// TIA Portal V18 program export: 2 tag tables, 0 data types, 2 data blocks, 5 code blocks (in call order from the OBs), 1 instance data blocks

VAR_GLOBAL   // PLC tag table "Default tag table"
   System_Byte AT %MB101 : Byte;
   FirstScan AT %M101.0 : Bool;
   DiagStatusUpdate AT %M101.1 : Bool;
   AlwaysTRUE AT %M101.2 : Bool;
   AlwaysFALSE AT %M101.3 : Bool;
   Clock_Byte AT %MB100 : Byte;
   Clock_10Hz AT %M100.0 : Bool;
   Clock_5Hz AT %M100.1 : Bool;
   "Clock_2.5Hz" AT %M100.2 : Bool;
   Clock_2Hz AT %M100.3 : Bool;
   "Clock_1.25Hz" AT %M100.4 : Bool;
   Clock_1Hz AT %M100.5 : Bool;
   "Clock_0.625Hz" AT %M100.6 : Bool;
   "Clock_0.5Hz" AT %M100.7 : Bool;
END_VAR

VAR_GLOBAL   // PLC tag table "PLC_Tags"
   FT3210_Bon3 AT %ID132 : Real;   // Cảm biến lưu lượng nước dosing vào Bồn 3
   FT3210_Bon3_HMI AT %MD764 : Real;   // Giá trị mô phỏng/HMI song song cho Cảm biến lưu lượng nước dosing vào Bồn 3
   FT3210_Bon3_Use_HMI AT %M421.0 : Bool;   // Chọn chế độ mô phỏng HMI cho Cảm biến lưu lượng nước dosing vào Bồn 3
   FT3210_Bon3_Sim_Req AT %M323.2 : Bool;   // Yêu cầu mô phỏng cảm biến cho Cảm biến lưu lượng nước dosing vào Bồn 3
   FT3210_Bon3_Sim_Active AT %M323.3 : Bool;   // Mô phỏng cảm biến đang hoạt động cho Cảm biến lưu lượng nước dosing vào Bồn 3
   FT3210_Bon3_Eff AT %MD768 : Real;   // Giá trị thực tế/mô phỏng hiệu dụng cho Cảm biến lưu lượng nước dosing vào Bồn 3
   FQ3210_Bon3 AT %ID136 : Real;   // Bộ đếm lưu lượng tích lũy Bồn 3
   FQ3210_Bon3_HMI AT %MD772 : Real;   // Giá trị mô phỏng/HMI song song cho Bộ đếm lưu lượng tích lũy Bồn 3
   FQ3210_Bon3_Use_HMI AT %M421.1 : Bool;   // Chọn chế độ mô phỏng HMI cho Bộ đếm lưu lượng tích lũy Bồn 3
   FQ3210_Bon3_Sim_Req AT %M323.4 : Bool;   // Yêu cầu mô phỏng cảm biến cho Bộ đếm lưu lượng tích lũy Bồn 3
   FQ3210_Bon3_Sim_Active AT %M323.5 : Bool;   // Mô phỏng cảm biến đang hoạt động cho Bộ đếm lưu lượng tích lũy Bồn 3
   FQ3210_Bon3_Eff AT %MD776 : Real;   // Giá trị thực tế/mô phỏng hiệu dụng cho Bộ đếm lưu lượng tích lũy Bồn 3
   LT3213_Bon3 AT %ID140 : Real;   // Cảm biến mức liên tục Bồn 3
   LT3213_Bon3_HMI AT %MD780 : Real;   // Giá trị mô phỏng/HMI song song cho Cảm biến mức liên tục Bồn 3
   LT3213_Bon3_Use_HMI AT %M421.2 : Bool;   // Chọn chế độ mô phỏng HMI cho Cảm biến mức liên tục Bồn 3
   LT3213_Bon3_Sim_Req AT %M323.6 : Bool;   // Yêu cầu mô phỏng cảm biến cho Cảm biến mức liên tục Bồn 3
   LT3213_Bon3_Sim_Active AT %M323.7 : Bool;   // Mô phỏng cảm biến đang hoạt động cho Cảm biến mức liên tục Bồn 3
   LT3213_Bon3_Eff AT %MD784 : Real;   // Giá trị thực tế/mô phỏng hiệu dụng cho Cảm biến mức liên tục Bồn 3
   TT3214_Bon3 AT %ID144 : Real;   // Cảm biến nhiệt độ Bồn 3
   TT3214_Bon3_HMI AT %MD788 : Real;   // Giá trị mô phỏng/HMI song song cho Cảm biến nhiệt độ Bồn 3
   TT3214_Bon3_Use_HMI AT %M421.3 : Bool;   // Chọn chế độ mô phỏng HMI cho Cảm biến nhiệt độ Bồn 3
   TT3214_Bon3_Sim_Req AT %M324.0 : Bool;   // Yêu cầu mô phỏng cảm biến cho Cảm biến nhiệt độ Bồn 3
   TT3214_Bon3_Sim_Active AT %M324.1 : Bool;   // Mô phỏng cảm biến đang hoạt động cho Cảm biến nhiệt độ Bồn 3
   TT3214_Bon3_Eff AT %MD792 : Real;   // Giá trị thực tế/mô phỏng hiệu dụng cho Cảm biến nhiệt độ Bồn 3
   FT3215_Bon4 AT %ID148 : Real;   // Cảm biến lưu lượng nước dosing vào Bồn 4
   FT3215_Bon4_HMI AT %MD796 : Real;   // Giá trị mô phỏng/HMI song song cho Cảm biến lưu lượng nước dosing vào Bồn 4
   FT3215_Bon4_Use_HMI AT %M421.4 : Bool;   // Chọn chế độ mô phỏng HMI cho Cảm biến lưu lượng nước dosing vào Bồn 4
   FT3215_Bon4_Sim_Req AT %M324.2 : Bool;   // Yêu cầu mô phỏng cảm biến cho Cảm biến lưu lượng nước dosing vào Bồn 4
   FT3215_Bon4_Sim_Active AT %M324.3 : Bool;   // Mô phỏng cảm biến đang hoạt động cho Cảm biến lưu lượng nước dosing vào Bồn 4
   FT3215_Bon4_Eff AT %MD800 : Real;   // Giá trị thực tế/mô phỏng hiệu dụng cho Cảm biến lưu lượng nước dosing vào Bồn 4
   FQ3215_Bon4 AT %ID152 : Real;   // Bộ đếm lưu lượng tích lũy Bồn 4
   FQ3215_Bon4_HMI AT %MD804 : Real;   // Giá trị mô phỏng/HMI song song cho Bộ đếm lưu lượng tích lũy Bồn 4
   FQ3215_Bon4_Use_HMI AT %M421.5 : Bool;   // Chọn chế độ mô phỏng HMI cho Bộ đếm lưu lượng tích lũy Bồn 4
   FQ3215_Bon4_Sim_Req AT %M324.4 : Bool;   // Yêu cầu mô phỏng cảm biến cho Bộ đếm lưu lượng tích lũy Bồn 4
   FQ3215_Bon4_Sim_Active AT %M324.5 : Bool;   // Mô phỏng cảm biến đang hoạt động cho Bộ đếm lưu lượng tích lũy Bồn 4
   FQ3215_Bon4_Eff AT %MD808 : Real;   // Giá trị thực tế/mô phỏng hiệu dụng cho Bộ đếm lưu lượng tích lũy Bồn 4
   LS3217_Bon4_Cao AT %I0.5 : Bool;   // Cảm biến mức cao Bồn 4
   LS3217_Bon4_Cao_HMI AT %M110.5 : Bool;   // Tín hiệu mô phỏng/HMI song song cho Cảm biến mức cao Bồn 4
   LS3217_Bon4_Cao_HMI_Gated AT %M324.6 : Bool;   // Tín hiệu HMI đã qua xử lý chế độ cho Cảm biến mức cao Bồn 4
   LS3217_Bon4_Cao_Eff AT %M324.7 : Bool;   // Tín hiệu thực tế/mô phỏng hiệu dụng cho Cảm biến mức cao Bồn 4
   LT3218_Bon4 AT %ID156 : Real;   // Cảm biến mức liên tục Bồn 4
   LT3218_Bon4_HMI AT %MD812 : Real;   // Giá trị mô phỏng/HMI song song cho Cảm biến mức liên tục Bồn 4
   LT3218_Bon4_Use_HMI AT %M421.6 : Bool;   // Chọn chế độ mô phỏng HMI cho Cảm biến mức liên tục Bồn 4
   LT3218_Bon4_Sim_Req AT %M325.0 : Bool;   // Yêu cầu mô phỏng cảm biến cho Cảm biến mức liên tục Bồn 4
   LT3218_Bon4_Sim_Active AT %M325.1 : Bool;   // Mô phỏng cảm biến đang hoạt động cho Cảm biến mức liên tục Bồn 4
   LT3218_Bon4_Eff AT %MD816 : Real;   // Giá trị thực tế/mô phỏng hiệu dụng cho Cảm biến mức liên tục Bồn 4
   TT3219_Bon4 AT %ID160 : Real;   // Cảm biến nhiệt độ Bồn 4
   TT3219_Bon4_HMI AT %MD820 : Real;   // Giá trị mô phỏng/HMI song song cho Cảm biến nhiệt độ Bồn 4
   TT3219_Bon4_Use_HMI AT %M421.7 : Bool;   // Chọn chế độ mô phỏng HMI cho Cảm biến nhiệt độ Bồn 4
   TT3219_Bon4_Sim_Req AT %M325.2 : Bool;   // Yêu cầu mô phỏng cảm biến cho Cảm biến nhiệt độ Bồn 4
   TT3219_Bon4_Sim_Active AT %M325.3 : Bool;   // Mô phỏng cảm biến đang hoạt động cho Cảm biến nhiệt độ Bồn 4
   TT3219_Bon4_Eff AT %MD824 : Real;   // Giá trị thực tế/mô phỏng hiệu dụng cho Cảm biến nhiệt độ Bồn 4
   V3240_Nuoc_Bon3 AT %Q1.4 : Bool;   // Van on/off cấp nước Bồn 3
   V3240_Nuoc_Bon3_M AT %M221.4 : Bool;   // Tag gương phản hồi HMI cho Van on/off cấp nước Bồn 3
   CV3211_Nuoc_Bon3 AT %QD116 : Real;   // Van tuyến tính cấp nước Bồn 3
   CV3211_Nuoc_Bon3_M AT %MD1216 : Real;   // Tag gương phản hồi HMI cho Van tuyến tính cấp nước Bồn 3
   AGTR3262_Khuay_Bon3 AT %Q1.5 : Bool;   // Động cơ khuấy Bồn 3
   AGTR3262_Khuay_Bon3_M AT %M221.5 : Bool;   // Tag gương phản hồi HMI cho Động cơ khuấy Bồn 3
   AGTR3262_Toc_Do_AO AT %QD120 : Real;   // Tín hiệu tốc độ khuấy Bồn 3
   AGTR3262_Toc_Do_AO_M AT %MD1220 : Real;   // Tag gương phản hồi HMI cho Tín hiệu tốc độ khuấy Bồn 3
   V3242_Xa_Bon3 AT %Q1.6 : Bool;   // Van xả đáy Bồn 3 số 1
   V3242_Xa_Bon3_M AT %M221.6 : Bool;   // Tag gương phản hồi HMI cho Van xả đáy Bồn 3 số 1
   V3243_Xa_Bon3 AT %Q1.7 : Bool;   // Van xả đáy Bồn 3 số 2
   V3243_Xa_Bon3_M AT %M221.7 : Bool;   // Tag gương phản hồi HMI cho Van xả đáy Bồn 3 số 2
   V3244_Xa_Bon3 AT %Q2.0 : Bool;   // Van xả đáy Bồn 3 số 3
   V3244_Xa_Bon3_M AT %M222.0 : Bool;   // Tag gương phản hồi HMI cho Van xả đáy Bồn 3 số 3
   V3245_Nuoc_Bon4 AT %Q2.1 : Bool;   // Van on/off cấp nước Bồn 4
   V3245_Nuoc_Bon4_M AT %M222.1 : Bool;   // Tag gương phản hồi HMI cho Van on/off cấp nước Bồn 4
   CV3216_Hoi_Bon4 AT %QD124 : Real;   // Van tuyến tính gia nhiệt mô phỏng Bồn 4
   CV3216_Hoi_Bon4_M AT %MD1224 : Real;   // Tag gương phản hồi HMI cho Van tuyến tính gia nhiệt mô phỏng Bồn 4
   AGTR3263_Khuay_Bon4 AT %Q2.2 : Bool;   // Động cơ khuấy Bồn 4
   AGTR3263_Khuay_Bon4_M AT %M222.2 : Bool;   // Tag gương phản hồi HMI cho Động cơ khuấy Bồn 4
   AGTR3263_Dao_Chieu AT %Q2.3 : Bool;   // Lệnh đảo chiều động cơ khuấy Bồn 4
   AGTR3263_Dao_Chieu_M AT %M222.3 : Bool;   // Tag gương phản hồi HMI cho Lệnh đảo chiều động cơ khuấy Bồn 4
   AGTR3263_Toc_Do_AO AT %QD128 : Real;   // Tốc độ đặt động cơ khuấy Bồn 4
   AGTR3263_Toc_Do_AO_M AT %MD1228 : Real;   // Tag gương phản hồi HMI cho Tốc độ đặt động cơ khuấy Bồn 4
   V3247_Xa_Bon4 AT %Q2.4 : Bool;   // Van xả đáy Bồn 4 số 1
   V3247_Xa_Bon4_M AT %M222.4 : Bool;   // Tag gương phản hồi HMI cho Van xả đáy Bồn 4 số 1
   V3248_Xa_Bon4 AT %Q2.5 : Bool;   // Van xả đáy Bồn 4 số 2
   V3248_Xa_Bon4_M AT %M222.5 : Bool;   // Tag gương phản hồi HMI cho Van xả đáy Bồn 4 số 2
   V3249_Xa_Bon4 AT %Q2.6 : Bool;   // Van xả đáy Bồn 4 số 3
   V3249_Xa_Bon4_M AT %M222.6 : Bool;   // Tag gương phản hồi HMI cho Van xả đáy Bồn 4 số 3
   Pump3265_Chuyen_Nhanh2 AT %Q2.7 : Bool;   // Bơm chuyển dung dịch Nhánh 2 xuống bồn chứa
   Pump3265_Chuyen_Nhanh2_M AT %M222.7 : Bool;   // Tag gương phản hồi HMI cho Bơm chuyển dung dịch Nhánh 2 xuống bồn chứa
   HMI_Operator_Login AT %M422.7 : Bool;   // Đăng nhập quyền Operator
   HMI_Engineer_Login AT %M423.0 : Bool;   // Đăng nhập quyền Engineer
   HMI_Admin_Login AT %M423.1 : Bool;   // Đăng nhập quyền Admin
   HMI_Che_Do_Manual AT %M423.2 : Bool;   // Cho phép điều khiển tay từng thiết bị
   HMI_Ack_Alarm AT %M423.3 : Bool;   // Xác nhận cảnh báo
   HMI_Reset_Alarm AT %M423.4 : Bool;   // Reset alarm bằng HMI
   Gia_Lap_Mat_Ket_Noi_HMI AT %M423.5 : Bool;   // Nút giả lập mất kết nối PLC
   HMI_User_Level AT %MW520 : Int;   // Mức quyền hiện tại: 1 Operator, 2 Engineer, 3 Admin
   HMI_Cho_Phep_Sua_Thong_So AT %M327.6 : Bool;   // Cờ cho phép sửa công thức và PID
   HMI_Alarm_Status AT %MW522 : Int;   // Mã cảnh báo tổng hợp cho WinCC TextList
   HMI_AnToan_Status AT %MW524 : Int;   // Mã chẩn đoán an toàn ưu tiên
   PLC2_Auto_Enable AT %M328.5 : Bool;   // Cho phép chạy Auto Nhánh 2 Bồn 3-4
   PLC2_EStop_Latch AT %M328.6 : Bool;   // Chốt dừng khẩn HMI/SCADA Nhánh 2 Bồn 3-4
   PLC2_Loi_Tong AT %M328.7 : Bool;   // Lỗi tổng khóa Auto Nhánh 2 Bồn 3-4
   PLC2_Loi_Dry_Run AT %M329.0 : Bool;   // Lỗi chạy khô bơm Nhánh 2 Bồn 3-4
   PLC2_Loi_Dosing AT %M329.1 : Bool;   // Lỗi quá thời gian dosing Nhánh 2 Bồn 3-4
   PLC2_Loi_Truyen_Thong AT %M329.2 : Bool;   // Lỗi truyền thông mô phỏng Nhánh 2 Bồn 3-4
   PLC2_State AT %MW528 : Int;   // Mã bước chu trình Nhánh 2 Bồn 3-4
   PLC2_Step_Bon3_Dosing AT %M331.0 : Bool;   // Bồn 3 đang dosing nước
   PLC2_Step_Bon3_Tip AT %M331.1 : Bool;   // Bồn 3 đang mô phỏng tip cốt tương đậu đậm đặc
   PLC2_Step_Bon3_Khuay AT %M331.2 : Bool;   // Bồn 3 đang khuấy ban đầu
   PLC2_Step_Bon3_Xa AT %M331.3 : Bool;   // Bồn 3 đang xả sang Bồn 4
   PLC2_Step_Bon4_Dosing AT %M331.4 : Bool;   // Bồn 4 đang dosing bổ sung
   PLC2_Step_Bon4_Tip AT %M331.5 : Bool;   // Bồn 4 đang tip phụ gia
   PLC2_Step_Bon4_Khuay_Thuan AT %M331.6 : Bool;   // Bồn 4 khuấy chiều thuận
   PLC2_Step_Bon4_Khuay_Nghich AT %M331.7 : Bool;   // Bồn 4 khuấy chiều ngược
   PLC2_Step_Bon4_PID_Mo_Phong AT %M332.0 : Bool;   // Bồn 4 chạy PID mô phỏng
   PLC2_Step_Bon4_Thanh_Trung AT %M332.1 : Bool;   // Bồn 4 giữ thời gian thanh trùng
   PLC2_Xa_Bon3_Xong AT %M332.2 : Bool;   // Bồn 3 đã xả hết
   PLC2_Xa_Bon4_Xong AT %M332.3 : Bool;   // Bồn 4 đã xả hết
   PLC2_Me_Nhanh2_Hoan_Thanh AT %M333.3 : Bool;   // Cờ hoàn thành Nhánh 2 gửi sang PLC1
   PLC2_Me_Nhanh2_Hoan_Thanh_M AT %M224.6 : Bool;   // Tag gương phản hồi HMI cho cờ hoàn thành Nhánh 2 gửi sang PLC1
   Pump3265_Chuyen_Nhanh2_Cmd_Nhan AT %M333.7 : Bool;   // Nhận lệnh chạy bơm chuyển Nhánh 2 từ PLC1
   Pump3265_Chuyen_Nhanh2_Cmd_Nhan_HMI AT %M111.1 : Bool;   // Tín hiệu mô phỏng/HMI song song cho lệnh chạy bơm chuyển Nhánh 2 từ PLC1
   Nut_Khoi_Dong_Nhan AT %M334.1 : Bool;   // nút khởi động nhận từ PLC1
   Nut_Khoi_Dong_Nhan_HMI AT %M111.2 : Bool;   // Tín hiệu mô phỏng/HMI song song cho nút khởi động nhận từ PLC1
   Nut_Khoi_Dong_Nhan_HMI_Gated AT %M334.2 : Bool;   // Tín hiệu HMI đã qua xử lý chế độ cho nút khởi động nhận từ PLC1
   Nut_Khoi_Dong_Nhan_Eff AT %M334.3 : Bool;   // Tín hiệu thực tế/mô phỏng hiệu dụng cho nút khởi động nhận từ PLC1
   Nut_Dung_Nhan AT %M334.4 : Bool;   // nút dừng nhận từ PLC1
   Nut_Dung_Nhan_HMI AT %M111.3 : Bool;   // Tín hiệu mô phỏng/HMI song song cho nút dừng nhận từ PLC1
   Nut_Dung_Nhan_HMI_Gated AT %M334.5 : Bool;   // Tín hiệu HMI đã qua xử lý chế độ cho nút dừng nhận từ PLC1
   Nut_Dung_Nhan_Eff AT %M334.6 : Bool;   // Tín hiệu thực tế/mô phỏng hiệu dụng cho nút dừng nhận từ PLC1
   Nut_Reset_Nhan AT %M334.7 : Bool;   // nút reset nhận từ PLC1
   Nut_Reset_Nhan_HMI AT %M111.4 : Bool;   // Tín hiệu mô phỏng/HMI song song cho nút reset nhận từ PLC1
   Nut_Reset_Nhan_HMI_Gated AT %M335.0 : Bool;   // Tín hiệu HMI đã qua xử lý chế độ cho nút reset nhận từ PLC1
   Nut_Reset_Nhan_Eff AT %M335.1 : Bool;   // Tín hiệu thực tế/mô phỏng hiệu dụng cho nút reset nhận từ PLC1
   Nut_EStop_Nhan AT %M335.2 : Bool;   // nút dừng khẩn nhận từ PLC1
   Nut_EStop_Nhan_HMI AT %M111.5 : Bool;   // Tín hiệu mô phỏng/HMI song song cho nút dừng khẩn nhận từ PLC1
   Nut_EStop_Nhan_HMI_Gated AT %M335.3 : Bool;   // Tín hiệu HMI đã qua xử lý chế độ cho nút dừng khẩn nhận từ PLC1
   Nut_EStop_Nhan_Eff AT %M335.4 : Bool;   // Tín hiệu thực tế/mô phỏng hiệu dụng cho nút dừng khẩn nhận từ PLC1
   Clock_1Hz AT %M100.5 : Bool;   // Clock 1Hz system memory bit
   FirstScan AT %M101.0 : Bool;   // First Scan system memory bit
   PLC2_Last_CmdSeq AT %MW80 : Int;   // Last processed command sequence
   PLC2_CmdSeq_New AT %M82.0 : Bool;   // New command sequence received
   MB_TCP_Server_Error AT %M82.1 : Bool;   // Modbus TCP Server Error
   MB_TCP_Server_Status AT %MW84 : Word;   // Modbus TCP Server Status
   MB_TCP_Server_NDR AT %M82.2 : Bool;   // Modbus TCP Server New Data Received
   MB_TCP_Server_DR AT %M82.3 : Bool;   // Modbus TCP Server Data Read
   PLC1_Tip_Bon1_Xong_HMI AT %M423.6 : Bool;   // Nút mô phỏng tip Bồn 1 đã hoàn tất
   PLC1_Khuay_Bon1_Xong_HMI AT %M423.7 : Bool;   // Nút mô phỏng hết thời gian khuấy Bồn 1
   PLC1_Tip_Bon2_Xong_HMI AT %M424.0 : Bool;   // Nút mô phỏng tip Bồn 2 đã hoàn tất
   PLC1_Khuay_Thuan_Bon2_Xong_HMI AT %M424.1 : Bool;   // Nút mô phỏng hết thời gian khuấy thuận Bồn 2
   PLC1_Khuay_Nghich_Bon2_Xong_HMI AT %M424.2 : Bool;   // Nút mô phỏng hết thời gian khuấy ngược Bồn 2
   PLC1_Thanh_Trung_Bon2_Xong_HMI AT %M424.3 : Bool;   // Nút mô phỏng hết thời gian thanh trùng Bồn 2
   PLC2_Tip_Bon3_Xong_HMI AT %M424.4 : Bool;   // Nút mô phỏng tip Bồn 3 đã hoàn tất
   PLC2_Khuay_Bon3_Xong_HMI AT %M424.5 : Bool;   // Nút mô phỏng hết thời gian khuấy Bồn 3
   PLC2_Tip_Bon4_Xong_HMI AT %M424.6 : Bool;   // Nút mô phỏng tip Bồn 4 đã hoàn tất
   PLC2_Khuay_Thuan_Bon4_Xong_HMI AT %M424.7 : Bool;   // Nút mô phỏng hết thời gian khuấy thuận Bồn 4
   PLC2_Khuay_Nghich_Bon4_Xong_HMI AT %M425.0 : Bool;   // Nút mô phỏng hết thời gian khuấy ngược Bồn 4
   PLC2_Thanh_Trung_Bon4_Xong_HMI AT %M425.1 : Bool;   // Nút mô phỏng hết thời gian thanh trùng Bồn 4
   BonChua_Nhan_Dich_Xong_HMI AT %M425.2 : Bool;   // Nút mô phỏng nhận dịch vào Bồn chứa 01 xong
   BonChua_Chuyen_Bon2_Xong_HMI AT %M425.3 : Bool;   // Nút mô phỏng chuyển sang Bồn chứa 02 xong
   HMI_SP_PLC1_Nuoc_Bon1 AT %MD896 : Real;   // Lượng nước dosing Bồn 1
   HMI_SP_PLC1_Nuoc_Bon2 AT %MD900 : Real;   // Lượng nước dosing bổ sung Bồn 2
   HMI_SP_PLC1_Toc_Do_Bon1 AT %MD904 : Real;   // Tốc độ khuấy Bồn 1
   HMI_SP_PLC1_Toc_Do_Bon2_Main AT %MD908 : Real;   // Tốc độ khuấy chính Bồn 2
   HMI_SP_PLC1_Nhiet_Do_Bon2 AT %MD912 : Real;   // Setpoint nhiệt/PID Bồn 2
   HMI_SP_PLC2_Nuoc_Bon3 AT %MD916 : Real;   // Lượng nước dosing Bồn 3
   HMI_SP_PLC2_Nuoc_Bon4 AT %MD920 : Real;   // Lượng nước dosing bổ sung Bồn 4
   HMI_SP_PLC2_Toc_Do_Bon3 AT %MD924 : Real;   // Tốc độ khuấy Bồn 3
   HMI_SP_PLC2_Toc_Do_Bon4_Main AT %MD928 : Real;   // Tốc độ khuấy chính Bồn 4
   HMI_SP_PLC2_Nhiet_Do_Bon4 AT %MD932 : Real;   // Setpoint nhiệt/PID mô phỏng Bồn 4
   HMI_SP_BonChua1_Nhiet_Giai_Nhiet AT %MD936 : Real;   // Nhiệt độ giải nhiệt đích Bồn chứa 01
   HMI_SP_Loc_Ap_Suat_Max AT %MD940 : Real;   // Ngưỡng áp suất cao trước màng lọc
   HMI_SP_Time_Khuay_Bon1 AT %MD944 : Time;   // Thời gian khuấy Bồn 1
   HMI_SP_Time_Khuay_Bon3 AT %MD948 : Time;   // Thời gian khuấy Bồn 3
   HMI_SP_Time_Fwd AT %MD952 : Time;   // Thời gian khuấy chiều thuận
   HMI_SP_Time_Rev AT %MD956 : Time;   // Thời gian khuấy chiều ngược
   HMI_SP_Time_Sterilize AT %MD960 : Time;   // Thời gian giữ nhiệt thanh trùng
   PLC1_Khuay_Bon1_Xong AT %M336.2 : Bool;   // Trạng thái tự động xong khuấy Bồn 1
   PLC1_Khuay_Thuan_Bon2_Xong AT %M336.3 : Bool;   // Trạng thái tự động xong khuấy thuận Bồn 2
   PLC1_Khuay_Nghich_Bon2_Xong AT %M336.4 : Bool;   // Trạng thái tự động xong khuấy ngược Bồn 2
   PLC1_Thanh_Trung_Bon2_Xong AT %M336.5 : Bool;   // Trạng thái tự động xong thanh trùng Bồn 2
   PLC2_Khuay_Bon3_Xong AT %M336.6 : Bool;   // Trạng thái tự động xong khuấy Bồn 3
   PLC2_Khuay_Thuan_Bon4_Xong AT %M336.7 : Bool;   // Trạng thái tự động xong khuấy thuận Bồn 4
   PLC2_Khuay_Nghich_Bon4_Xong AT %M337.0 : Bool;   // Trạng thái tự động xong khuấy ngược Bồn 4
   PLC2_Thanh_Trung_Bon4_Xong AT %M337.1 : Bool;   // Trạng thái tự động xong thanh trùng Bồn 4
   PLC1_Tip_Bon1_Auto_Done AT %M337.2 : Bool;   // Trạng thái tự động xong tip Bồn 1
   PLC1_Tip_Bon2_Auto_Done AT %M337.3 : Bool;   // Trạng thái tự động xong tip Bồn 2
   PLC2_Tip_Bon3_Auto_Done AT %M337.4 : Bool;   // Trạng thái tự động xong tip Bồn 3
   PLC2_Tip_Bon4_Auto_Done AT %M337.5 : Bool;   // Trạng thái tự động xong tip Bồn 4
   PLC1_Start_Edge_Old AT %M337.6 : Bool;   // Cờ nhớ cạnh lên nút Start PLC1
   PLC1_Start_Edge_Edge AT %M337.7 : Bool;   // Xung cạnh lên nút Start PLC1
   PLC2_Start_Edge_Old AT %M338.0 : Bool;   // Cờ nhớ cạnh lên nút Start PLC2
   PLC2_Start_Edge_Edge AT %M338.1 : Bool;   // Xung cạnh lên nút Start PLC2
   PID_Bon2_Enable AT %M338.2 : Bool;   // Cho phép PID Bồn 2
   PID_Bon2_ManualEnable AT %M338.3 : Bool;   // Chế độ manual PID Bồn 2
   PID_Bon2_Error AT %M338.4 : Bool;   // Lỗi khối PID Bồn 2
   PID_Bon4_Enable AT %M338.5 : Bool;   // Cho phép PID mô phỏng Bồn 4
   PID_Bon4_ManualEnable AT %M338.6 : Bool;   // Chế độ manual PID Bồn 4
   PID_Bon4_Error AT %M338.7 : Bool;   // Lỗi khối PID Bồn 4
   PID_Bon2_ErrorBits AT %MD964 : DWord;   // Mã lỗi DWORD PID Bồn 2
   PID_Bon4_ErrorBits AT %MD968 : DWord;   // Mã lỗi DWORD PID Bồn 4
   PID_Bon2_SP AT %MD972 : Real;   // Setpoint đưa vào PID Bồn 2
   PID_Bon2_Err AT %MD976 : Real;   // Sai lệch PID Bồn 2 = SP - PV
   PID_Bon2_CV AT %MD980 : Real;   // Giá trị điều khiển PID Bồn 2
   PID_Bon2_ManualValue AT %MD984 : Real;   // Giá trị manual PID Bồn 2
   PID_Bon4_SP AT %MD988 : Real;   // Setpoint đưa vào PID mô phỏng Bồn 4
   PID_Bon4_Err AT %MD992 : Real;   // Sai lệch PID mô phỏng Bồn 4 = SP - PV
   PID_Bon4_CV AT %MD996 : Real;   // Giá trị điều khiển PID mô phỏng Bồn 4
   PID_Bon4_ManualValue AT %MD1000 : Real;   // Giá trị manual PID Bồn 4
   TT3219_Bon4_Sim AT %MD1004 : Real;   // Nhiệt độ mô phỏng nội bộ cho PID Bồn 4
   PID_Bon2_Temp_Inc AT %MD1008 : Real;   // Mức tăng nhiệt mô phỏng Bồn 2
   PID_Bon4_Tang_Nhiet_Buoc AT %MD1012 : Real;   // Mức tăng nhiệt mô phỏng mỗi chu kỳ OB31
   TT3219_Bon4_Target AT %MD1016 : Real;   // Nhiệt độ đích mô phỏng bồn 4
   TT3219_Bon4_Sim_Pure AT %MD1020 : Real;   // Nhiệt độ mô phỏng chưa có nhiễu bồn 4
   PID_Bon4_Temp_Val_1 AT %MD1024 : Real;   // Biến tạm mô phỏng nhiệt độ 1
   PID_Bon4_Temp_Val_2 AT %MD1028 : Real;   // Biến tạm mô phỏng nhiệt độ 2
   PID_Bon4_Sim_Counter AT %MD1032 : Real;   // Đồng hồ chu kỳ mô phỏng
   PID_Bon4_Sim_Angle AT %MD1036 : Real;   // Góc lượng giác nhiễu
   PID_Bon4_Sim_Sin AT %MD1040 : Real;   // Giá trị hình sin nhiễu
   PID_Bon4_Sim_Noise AT %MD1044 : Real;   // Giá trị nhiễu nhiệt độ
   PLC1_Tip_Bon1_Timer AT %MD1048 : Real;   // Bộ đếm thời gian mô phỏng tip bồn 1
   PLC1_Tip_Bon2_Timer AT %MD1052 : Real;   // Bộ đếm thời gian mô phỏng tip bồn 2
   PLC2_Tip_Bon3_Timer AT %MD1056 : Real;   // Bộ đếm thời gian mô phỏng tip bồn 3
   PLC2_Tip_Bon4_Timer AT %MD1060 : Real;   // Bộ đếm thời gian mô phỏng tip bồn 4
   PID_Bon4_State AT %MW536 : Int;   // Trạng thái khối PID Bồn 4
   PLC2_Stop_Active AT %M339.1 : Bool;   // Tín hiệu dừng active PLC2
   AGTR3263_Khuay_Active AT %M339.4 : Bool;   // Trạng thái khuấy Bồn 4 active
   AGTR3263_Should_Run AT %M339.5 : Bool;   // Yêu cầu chạy động cơ Bồn 4
   HMI_Use_Sim_Input_PLC2 AT %M339.7 : Bool;   // Cho phép sử dụng đầu vào mô phỏng PLC2
   Pump3265_Chuyen_Nhanh2_Cmd_Nhan_Eff AT %M340.2 : Bool;   // Lệnh chạy bơm chuyển Nhánh 2 nhận được hiệu dụng
   Pump3265_Chuyen_Nhanh2_Cmd_Nhan_HMI_Gated AT %M340.4 : Bool;   // Lệnh chạy bơm chuyển Nhánh 2 HMI gated
   PLC2_SP_Valid AT %M340.6 : Bool;   // Setpoint PLC2 hợp lệ
   PLC2_Loi_Setpoint AT %M341.1 : Bool;   // Lỗi Setpoint PLC2
   Init_Defaults_Done_PLC2 AT %M341.4 : Bool;   // Khởi tạo Setpoint mặc định PLC2 hoàn tất
   Init_Trigger_PLC2 AT %M341.7 : Bool;   // Cờ kích hoạt nạp recipe mặc định PLC2
   HMI_Load_Default_Recipe AT %M342.1 : Bool;   // Yêu cầu nạp lại Recipe mặc định từ HMI
   PLC2_Load_Default_Cmd_Nhan AT %M342.3 : Bool;   // Nhận lệnh nạp recipe mặc định từ PLC1
   PLC2_Load_Default_Cmd_Nhan_HMI AT %M111.6 : Bool;   // Tín hiệu mô phỏng/HMI cho nhận lệnh nạp recipe
   PLC2_Load_Default_Cmd_Nhan_HMI_Gated AT %M342.4 : Bool;   // Tín hiệu nhận lệnh nạp recipe HMI gated
   PLC2_Load_Default_Cmd_Nhan_Eff AT %M342.5 : Bool;   // Tín hiệu nhận lệnh nạp recipe hiệu dụng
   PLC2_Load_Default_Done AT %M342.6 : Bool;   // Báo nạp recipe mặc định xong gửi sang PLC1
   PLC2_Load_Default_Done_M AT %M225.1 : Bool;   // Tag gương phản hồi HMI cho báo nạp recipe xong PLC2
   HMI_Sim_Mode AT %M343.2 : Bool;   // Cho phép toàn bộ tín hiệu mô phỏng HMI tác động vào input hiệu dụng
   HMI_Run_Enable AT %M343.3 : Bool;   // Cho phép vận hành từ HMI ở chế độ thật
   System_Mode_Real AT %M343.4 : Bool;   // Hệ thống đang hoạt động ở chế độ thực tế
   System_Mode_Sim AT %M343.5 : Bool;   // Hệ thống đang hoạt động ở chế độ mô phỏng
   HMI_Sim_Active_Warning AT %M343.6 : Bool;   // Cảnh báo chế độ mô phỏng HMI đang hoạt động
   PID_Bon4_Kp_HMI AT %MD1072 : Real;   // HMI parameter for Kp PID Bồn 4
   PID_Bon4_Ti_HMI AT %MD1076 : Real;   // HMI parameter for Ti PID Bồn 4
   Clock_1Hz_Last AT %M344.1 : Bool;   // Trạng thái Clock 1Hz chu kỳ trước
   Clock_1Hz_Edge AT %M344.2 : Bool;   // Xung cạnh lên của Clock 1Hz
   PLC1_Heartbeat_Last AT %MW538 : Int;   // Heartbeat PLC1 chu kỳ trước
   PLC1_Heartbeat_Changed AT %M344.3 : Bool;   // Cờ heartbeat PLC1 thay đổi
   PLC2_Heartbeat_Timeout AT %M344.4 : Bool;   // Lỗi timeout heartbeat PLC1
END_VAR

DATA_BLOCK "DB_Modbus_Holding_Register_DB"   // DB20
TITLE = DB_Modbus_Holding_Register_DB
{ S7_Optimized_Access := 'FALSE' }
VERSION : 0.1
// DB communication via Modbus TCP
// stored: AutoNumber false, DBAccessibleFromOPCUA true, IsOnlyStoredInLoadMemory false, IsWriteProtectedInAS false
   VAR
      CmdSeq : Int;
      Cmd_Start : Bool;
      Cmd_Stop : Bool;
      Cmd_Reset : Bool;
      Cmd_EStop : Bool;
      Cmd_Pump_Branch2_To_SubTanks : Bool;
      Cmd_Load_Recipe : Bool;
      Heartbeat_Client : Int;
      AckSeq : Int;
      Done_Branch2 : Bool;
      Done_Recipe : Bool;
      Alarm : Bool;
      State : Int;
      PID_Bon4_SP : Real;
      PID_Bon4_PV : Real;
      PID_Bon4_CV : Real;
      Done_Discharge2 : Bool;
      Heartbeat_Server : Int;
   END_VAR
BEGIN
END_DATA_BLOCK

DATA_BLOCK "Timers_PLC2"   // DB1
TITLE = Timers_PLC2
{ S7_Optimized_Access := 'TRUE' }
VERSION : 0.1
// Global DB containing all timers and PID instances
// stored: AutoNumber true, DBAccessibleFromOPCUA true, IsOnlyStoredInLoadMemory false, IsRetainMemResEnabled false, IsWriteProtectedInAS false, MemoryReserve 100
   VAR
      Timer_Dosing_Bon3 : IEC_TIMER;
      Timer_Tip_Bon3 : IEC_TIMER;
      Timer_Dosing_Bon4 : IEC_TIMER;
      Timer_Tip_Bon4 : IEC_TIMER;
      Timer_Khuay_Bon3 : IEC_TIMER;
      Timer_Khuay_Thuan_Bon4 : IEC_TIMER;
      Timer_Khuay_Nghich_Bon4 : IEC_TIMER;
      Timer_Thanh_Trung_Bon4 : IEC_TIMER;
      Timer_DryRun_Bon4 : IEC_TIMER;
      Timer_Heartbeat_PLC2 : IEC_TIMER;
   END_VAR
BEGIN
END_DATA_BLOCK

ORGANIZATION_BLOCK "Main"   // OB1, LAD, ProgramCycle
TITLE = "Main Program Sweep (Cycle)"
{ S7_Optimized_Access := 'TRUE' }
VERSION : 0.1
// stored: AutoNumber true, IsIECCheckEnabled false, SetENOAutomatically false
   VAR_INPUT
      Initial_Call : Bool;   // Initial call of this OB
      Remanence : Bool;   // =True, if remanent data are available
   END_VAR
BEGIN

REGION Network 1: Clock 1Hz Edge Detection
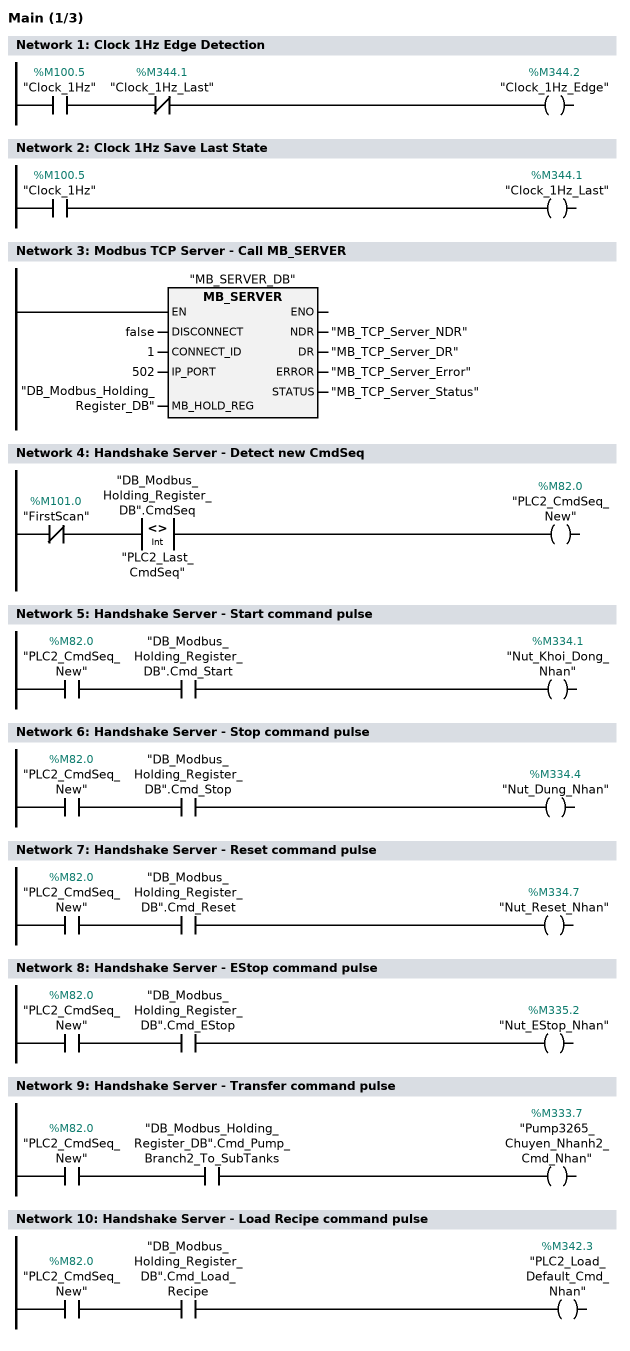
   RUNG wire#powerrail
      Contact( "Clock_1Hz" )
      I_Contact( "Clock_1Hz_Last" )
      Coil( "Clock_1Hz_Edge" )
   END_RUNG
   // the same network as SCL:
   "Clock_1Hz_Edge" := "Clock_1Hz" AND NOT "Clock_1Hz_Last";
END_REGION

REGION Network 2: Clock 1Hz Save Last State
   RUNG wire#powerrail
      Contact( "Clock_1Hz" )
      Coil( "Clock_1Hz_Last" )
   END_RUNG
   // the same network as SCL:
   "Clock_1Hz_Last" := "Clock_1Hz";
END_REGION

REGION Network 3: Modbus TCP Server - Call MB_SERVER
   RUNG wire#powerrail
      { S7_Templates := "[card1200 := 1, card1500 := 0]" } "MB_SERVER_DB".MB_SERVER(DISCONNECT := false, CONNECT_ID := 1, IP_PORT := 502, MB_HOLD_REG := "DB_Modbus_Holding_Register_DB", NDR => "MB_TCP_Server_NDR", DR => "MB_TCP_Server_DR", ERROR => "MB_TCP_Server_Error", STATUS => "MB_TCP_Server_Status")
   END_RUNG
   // the same network as SCL:
   "MB_SERVER_DB"(DISCONNECT := false,   // MB_SERVER
                  CONNECT_ID := 1,
                  IP_PORT := 502,
                  MB_HOLD_REG := "DB_Modbus_Holding_Register_DB",
                  NDR => "MB_TCP_Server_NDR",
                  DR => "MB_TCP_Server_DR",
                  ERROR => "MB_TCP_Server_Error",
                  STATUS => "MB_TCP_Server_Status");
END_REGION

REGION Network 4: Handshake Server - Detect new CmdSeq
   RUNG wire#powerrail
      I_Contact( "FirstScan" )
      { S7_Templates := "SrcType := Int" } NE_Contact(in1 := "DB_Modbus_Holding_Register_DB".CmdSeq, in2 := "PLC2_Last_CmdSeq")
      Coil( "PLC2_CmdSeq_New" )
   END_RUNG
   // the same network as SCL:
   "PLC2_CmdSeq_New" := NOT "FirstScan" AND ("DB_Modbus_Holding_Register_DB".CmdSeq <> "PLC2_Last_CmdSeq");
END_REGION

REGION Network 5: Handshake Server - Start command pulse
   RUNG wire#powerrail
      Contact( "PLC2_CmdSeq_New" )
      Contact( "DB_Modbus_Holding_Register_DB".Cmd_Start )
      Coil( "Nut_Khoi_Dong_Nhan" )
   END_RUNG
   // the same network as SCL:
   "Nut_Khoi_Dong_Nhan" := "PLC2_CmdSeq_New" AND "DB_Modbus_Holding_Register_DB".Cmd_Start;
END_REGION

REGION Network 6: Handshake Server - Stop command pulse
   RUNG wire#powerrail
      Contact( "PLC2_CmdSeq_New" )
      Contact( "DB_Modbus_Holding_Register_DB".Cmd_Stop )
      Coil( "Nut_Dung_Nhan" )
   END_RUNG
   // the same network as SCL:
   "Nut_Dung_Nhan" := "PLC2_CmdSeq_New" AND "DB_Modbus_Holding_Register_DB".Cmd_Stop;
END_REGION

REGION Network 7: Handshake Server - Reset command pulse
   RUNG wire#powerrail
      Contact( "PLC2_CmdSeq_New" )
      Contact( "DB_Modbus_Holding_Register_DB".Cmd_Reset )
      Coil( "Nut_Reset_Nhan" )
   END_RUNG
   // the same network as SCL:
   "Nut_Reset_Nhan" := "PLC2_CmdSeq_New" AND "DB_Modbus_Holding_Register_DB".Cmd_Reset;
END_REGION

REGION Network 8: Handshake Server - EStop command pulse
   RUNG wire#powerrail
      Contact( "PLC2_CmdSeq_New" )
      Contact( "DB_Modbus_Holding_Register_DB".Cmd_EStop )
      Coil( "Nut_EStop_Nhan" )
   END_RUNG
   // the same network as SCL:
   "Nut_EStop_Nhan" := "PLC2_CmdSeq_New" AND "DB_Modbus_Holding_Register_DB".Cmd_EStop;
END_REGION

REGION Network 9: Handshake Server - Transfer command pulse
   RUNG wire#powerrail
      Contact( "PLC2_CmdSeq_New" )
      Contact( "DB_Modbus_Holding_Register_DB".Cmd_Pump_Branch2_To_SubTanks )
      Coil( "Pump3265_Chuyen_Nhanh2_Cmd_Nhan" )
   END_RUNG
   // the same network as SCL:
   "Pump3265_Chuyen_Nhanh2_Cmd_Nhan" := "PLC2_CmdSeq_New" AND "DB_Modbus_Holding_Register_DB".Cmd_Pump_Branch2_To_SubTanks;
END_REGION

REGION Network 10: Handshake Server - Load Recipe command pulse
   RUNG wire#powerrail
      Contact( "PLC2_CmdSeq_New" )
      Contact( "DB_Modbus_Holding_Register_DB".Cmd_Load_Recipe )
      Coil( "PLC2_Load_Default_Cmd_Nhan" )
   END_RUNG
   // the same network as SCL:
   "PLC2_Load_Default_Cmd_Nhan" := "PLC2_CmdSeq_New" AND "DB_Modbus_Holding_Register_DB".Cmd_Load_Recipe;
END_REGION

REGION Network 11: PLC2 - Gọi logic khởi tạo recipe mặc định PLC2
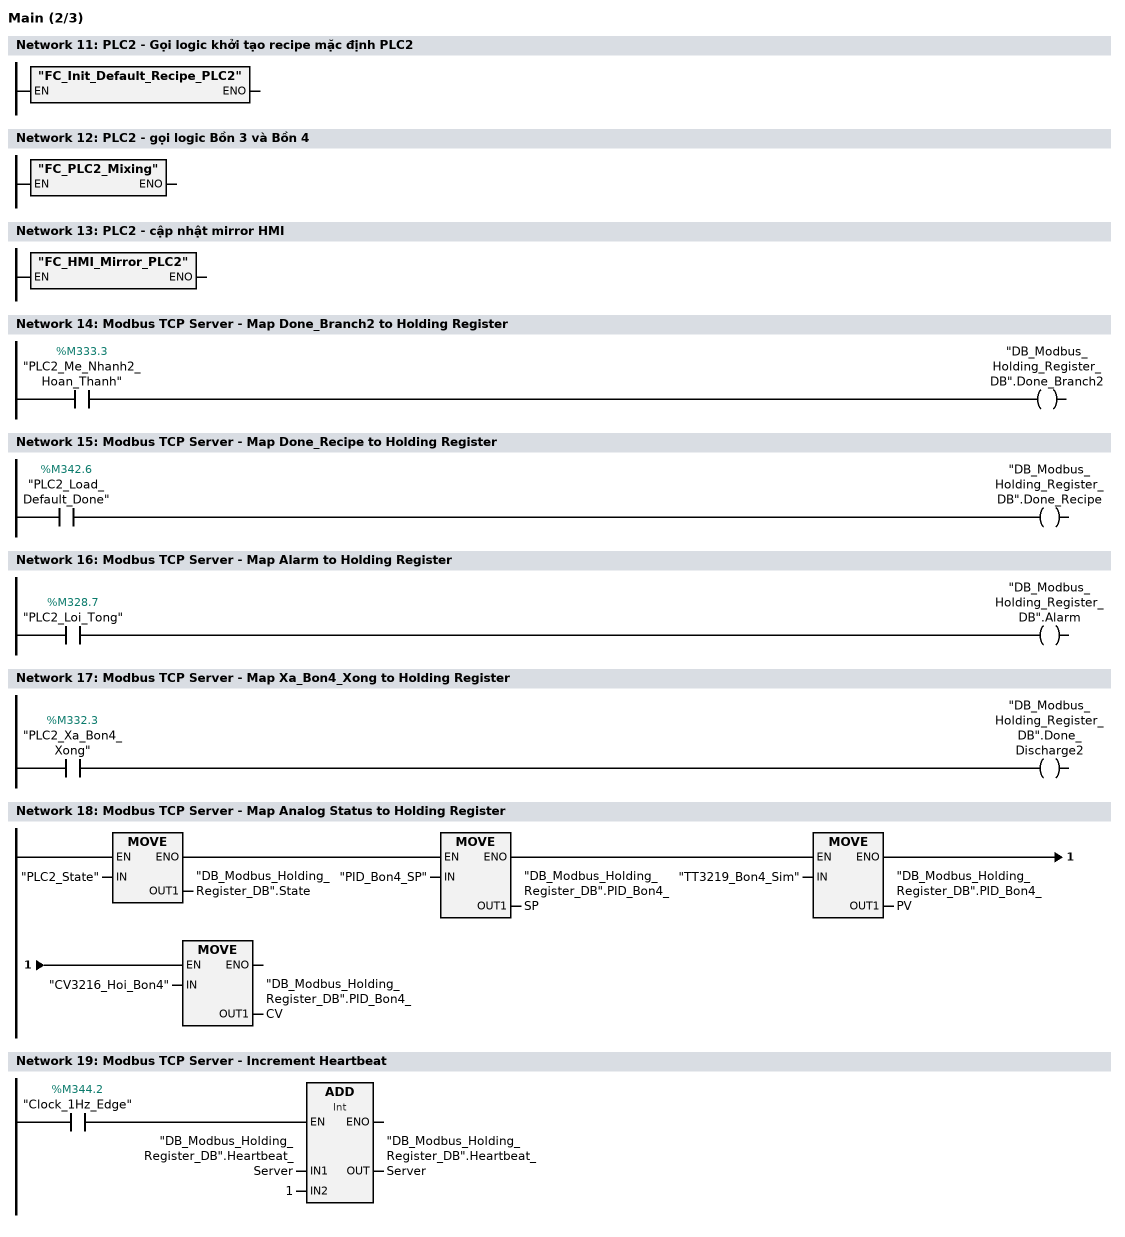
   RUNG wire#powerrail
      "FC_Init_Default_Recipe_PLC2"()
   END_RUNG
   // the same network as SCL:
   "FC_Init_Default_Recipe_PLC2"();
END_REGION

REGION Network 12: PLC2 - gọi logic Bồn 3 và Bồn 4
   RUNG wire#powerrail
      "FC_PLC2_Mixing"()
   END_RUNG
   // the same network as SCL:
   "FC_PLC2_Mixing"();
END_REGION

REGION Network 13: PLC2 - cập nhật mirror HMI
   RUNG wire#powerrail
      "FC_HMI_Mirror_PLC2"()
   END_RUNG
   // the same network as SCL:
   "FC_HMI_Mirror_PLC2"();
END_REGION

REGION Network 14: Modbus TCP Server - Map Done_Branch2 to Holding Register
   RUNG wire#powerrail
      Contact( "PLC2_Me_Nhanh2_Hoan_Thanh" )
      Coil( "DB_Modbus_Holding_Register_DB".Done_Branch2 )
   END_RUNG
   // the same network as SCL:
   "DB_Modbus_Holding_Register_DB".Done_Branch2 := "PLC2_Me_Nhanh2_Hoan_Thanh";
END_REGION

REGION Network 15: Modbus TCP Server - Map Done_Recipe to Holding Register
   RUNG wire#powerrail
      Contact( "PLC2_Load_Default_Done" )
      Coil( "DB_Modbus_Holding_Register_DB".Done_Recipe )
   END_RUNG
   // the same network as SCL:
   "DB_Modbus_Holding_Register_DB".Done_Recipe := "PLC2_Load_Default_Done";
END_REGION

REGION Network 16: Modbus TCP Server - Map Alarm to Holding Register
   RUNG wire#powerrail
      Contact( "PLC2_Loi_Tong" )
      Coil( "DB_Modbus_Holding_Register_DB".Alarm )
   END_RUNG
   // the same network as SCL:
   "DB_Modbus_Holding_Register_DB".Alarm := "PLC2_Loi_Tong";
END_REGION

REGION Network 17: Modbus TCP Server - Map Xa_Bon4_Xong to Holding Register
   RUNG wire#powerrail
      Contact( "PLC2_Xa_Bon4_Xong" )
      Coil( "DB_Modbus_Holding_Register_DB".Done_Discharge2 )
   END_RUNG
   // the same network as SCL:
   "DB_Modbus_Holding_Register_DB".Done_Discharge2 := "PLC2_Xa_Bon4_Xong";
END_REGION

REGION Network 18: Modbus TCP Server - Map Analog Status to Holding Register
   RUNG wire#powerrail
      { S7_GenerateENO := "TRUE" } Move(in := "PLC2_State", out1 => "DB_Modbus_Holding_Register_DB".State)
      { S7_GenerateENO := "TRUE" } Move(in := "PID_Bon4_SP", out1 => "DB_Modbus_Holding_Register_DB".PID_Bon4_SP)
      { S7_GenerateENO := "TRUE" } Move(in := "TT3219_Bon4_Sim", out1 => "DB_Modbus_Holding_Register_DB".PID_Bon4_PV)
      { S7_GenerateENO := "TRUE" } Move(in := "CV3216_Hoi_Bon4", out1 => "DB_Modbus_Holding_Register_DB".PID_Bon4_CV)
   END_RUNG
   // the same network as SCL:
   // ENO of a box is taken as its EN; it also drops when the box reports an error
   "DB_Modbus_Holding_Register_DB".State := "PLC2_State";
   "DB_Modbus_Holding_Register_DB".PID_Bon4_SP := "PID_Bon4_SP";
   "DB_Modbus_Holding_Register_DB".PID_Bon4_PV := "TT3219_Bon4_Sim";
   "DB_Modbus_Holding_Register_DB".PID_Bon4_CV := "CV3216_Hoi_Bon4";
END_REGION

REGION Network 19: Modbus TCP Server - Increment Heartbeat
   RUNG wire#powerrail
      Contact( "Clock_1Hz_Edge" )
      { S7_Templates := "SrcType := Int"; S7_GenerateENO := "TRUE" } Add(in1 := "DB_Modbus_Holding_Register_DB".Heartbeat_Server, in2 := 1, out => "DB_Modbus_Holding_Register_DB".Heartbeat_Server)
   END_RUNG
   // the same network as SCL:
   IF "Clock_1Hz_Edge" THEN
       "DB_Modbus_Holding_Register_DB".Heartbeat_Server := "DB_Modbus_Holding_Register_DB".Heartbeat_Server + 1;
   END_IF;
END_REGION

REGION Network 20: Modbus TCP Server - Monitor Heartbeat Change
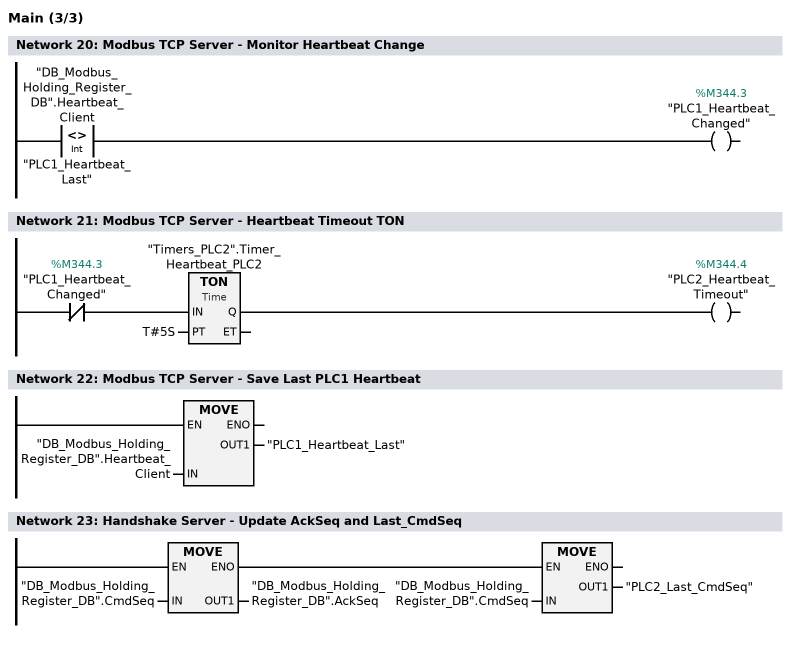
   RUNG wire#powerrail
      { S7_Templates := "SrcType := Int" } NE_Contact(in1 := "DB_Modbus_Holding_Register_DB".Heartbeat_Client, in2 := "PLC1_Heartbeat_Last")
      Coil( "PLC1_Heartbeat_Changed" )
   END_RUNG
   // the same network as SCL:
   "PLC1_Heartbeat_Changed" := "DB_Modbus_Holding_Register_DB".Heartbeat_Client <> "PLC1_Heartbeat_Last";
END_REGION

REGION Network 21: Modbus TCP Server - Heartbeat Timeout TON
   RUNG wire#powerrail
      I_Contact( "PLC1_Heartbeat_Changed" )
      { S7_Templates := "time_type := Time" } "Timers_PLC2".Timer_Heartbeat_PLC2.TON(pt := T#5S, et =>)
      Coil( "PLC2_Heartbeat_Timeout" )
   END_RUNG
   // the same network as SCL:
   "Timers_PLC2".Timer_Heartbeat_PLC2.TON(IN := NOT "PLC1_Heartbeat_Changed", PT := T#5S);
   "PLC2_Heartbeat_Timeout" := "Timers_PLC2".Timer_Heartbeat_PLC2.Q;
END_REGION

REGION Network 22: Modbus TCP Server - Save Last PLC1 Heartbeat
   RUNG wire#powerrail
      { S7_GenerateENO := "TRUE" } Move(in := "DB_Modbus_Holding_Register_DB".Heartbeat_Client, out1 => "PLC1_Heartbeat_Last")
   END_RUNG
   // the same network as SCL:
   "PLC1_Heartbeat_Last" := "DB_Modbus_Holding_Register_DB".Heartbeat_Client;
END_REGION

REGION Network 23: Handshake Server - Update AckSeq and Last_CmdSeq
   RUNG wire#powerrail
      { S7_GenerateENO := "TRUE" } Move(in := "DB_Modbus_Holding_Register_DB".CmdSeq, out1 => "DB_Modbus_Holding_Register_DB".AckSeq)
      { S7_GenerateENO := "TRUE" } Move(in := "DB_Modbus_Holding_Register_DB".CmdSeq, out1 => "PLC2_Last_CmdSeq")
   END_RUNG
   // the same network as SCL:
   // ENO of a box is taken as its EN; it also drops when the box reports an error
   "DB_Modbus_Holding_Register_DB".AckSeq := "DB_Modbus_Holding_Register_DB".CmdSeq;
   "PLC2_Last_CmdSeq" := "DB_Modbus_Holding_Register_DB".CmdSeq;
END_REGION
END_ORGANIZATION_BLOCK

FUNCTION "FC_Init_Default_Recipe_PLC2" : Void   // FC51, LAD
{ S7_Optimized_Access := 'TRUE' }
VERSION : 0.1
// stored: AutoNumber true, IsIECCheckEnabled false, SetENOAutomatically false, UDAEnableTagReadback false
BEGIN

REGION Network 1: Kích hoạt nạp recipe mặc định lần đầu scan PLC2
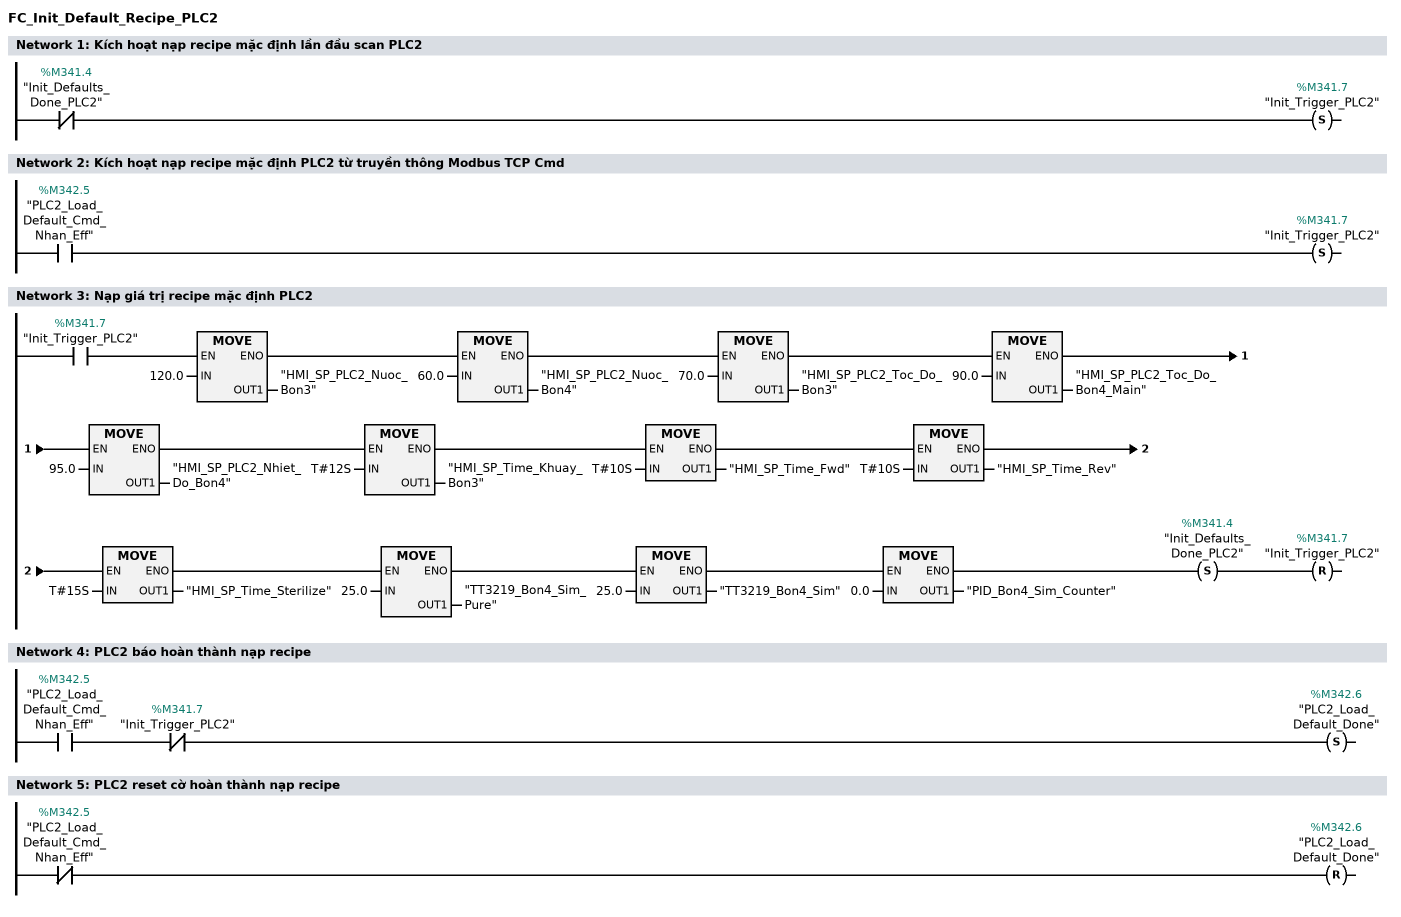
   RUNG wire#powerrail
      I_Contact( "Init_Defaults_Done_PLC2" )
      S_Coil( "Init_Trigger_PLC2" )
   END_RUNG
   // the same network as SCL:
   IF NOT "Init_Defaults_Done_PLC2" THEN "Init_Trigger_PLC2" := TRUE; END_IF;
END_REGION

REGION Network 2: Kích hoạt nạp recipe mặc định PLC2 từ truyền thông Modbus TCP Cmd
   RUNG wire#powerrail
      Contact( "PLC2_Load_Default_Cmd_Nhan_Eff" )
      S_Coil( "Init_Trigger_PLC2" )
   END_RUNG
   // the same network as SCL:
   IF "PLC2_Load_Default_Cmd_Nhan_Eff" THEN "Init_Trigger_PLC2" := TRUE; END_IF;
END_REGION

REGION Network 3: Nạp giá trị recipe mặc định PLC2
   RUNG wire#powerrail
      Contact( "Init_Trigger_PLC2" )
      { S7_GenerateENO := "TRUE" } Move(in := 120.0, out1 => "HMI_SP_PLC2_Nuoc_Bon3")
      { S7_GenerateENO := "TRUE" } Move(in := 60.0, out1 => "HMI_SP_PLC2_Nuoc_Bon4")
      { S7_GenerateENO := "TRUE" } Move(in := 70.0, out1 => "HMI_SP_PLC2_Toc_Do_Bon3")
      { S7_GenerateENO := "TRUE" } Move(in := 90.0, out1 => "HMI_SP_PLC2_Toc_Do_Bon4_Main")
      { S7_GenerateENO := "TRUE" } Move(in := 95.0, out1 => "HMI_SP_PLC2_Nhiet_Do_Bon4")
      { S7_GenerateENO := "TRUE" } Move(in := T#12S, out1 => "HMI_SP_Time_Khuay_Bon3")
      { S7_GenerateENO := "TRUE" } Move(in := T#10S, out1 => "HMI_SP_Time_Fwd")
      { S7_GenerateENO := "TRUE" } Move(in := T#10S, out1 => "HMI_SP_Time_Rev")
      { S7_GenerateENO := "TRUE" } Move(in := T#15S, out1 => "HMI_SP_Time_Sterilize")
      { S7_GenerateENO := "TRUE" } Move(in := 25.0, out1 => "TT3219_Bon4_Sim_Pure")
      { S7_GenerateENO := "TRUE" } Move(in := 25.0, out1 => "TT3219_Bon4_Sim")
      { S7_GenerateENO := "TRUE" } Move(in := 0.0, out1 => "PID_Bon4_Sim_Counter")
      S_Coil( "Init_Defaults_Done_PLC2" )
      R_Coil( "Init_Trigger_PLC2" )
   END_RUNG
   // the same network as SCL:
   // ENO of a box is taken as its EN; it also drops when the box reports an error
   IF "Init_Trigger_PLC2" THEN
       "HMI_SP_PLC2_Nuoc_Bon3" := 120.0;
       "HMI_SP_PLC2_Nuoc_Bon4" := 60.0;
       "HMI_SP_PLC2_Toc_Do_Bon3" := 70.0;
       "HMI_SP_PLC2_Toc_Do_Bon4_Main" := 90.0;
       "HMI_SP_PLC2_Nhiet_Do_Bon4" := 95.0;
       "HMI_SP_Time_Khuay_Bon3" := T#12S;
       "HMI_SP_Time_Fwd" := T#10S;
       "HMI_SP_Time_Rev" := T#10S;
       "HMI_SP_Time_Sterilize" := T#15S;
       "TT3219_Bon4_Sim_Pure" := 25.0;
       "TT3219_Bon4_Sim" := 25.0;
       "PID_Bon4_Sim_Counter" := 0.0;
       "Init_Defaults_Done_PLC2" := TRUE;
       "Init_Trigger_PLC2" := FALSE;
   END_IF;
END_REGION

REGION Network 4: PLC2 báo hoàn thành nạp recipe
   RUNG wire#powerrail
      Contact( "PLC2_Load_Default_Cmd_Nhan_Eff" )
      I_Contact( "Init_Trigger_PLC2" )
      S_Coil( "PLC2_Load_Default_Done" )
   END_RUNG
   // the same network as SCL:
   IF "PLC2_Load_Default_Cmd_Nhan_Eff" AND NOT "Init_Trigger_PLC2" THEN
       "PLC2_Load_Default_Done" := TRUE;
   END_IF;
END_REGION

REGION Network 5: PLC2 reset cờ hoàn thành nạp recipe
   RUNG wire#powerrail
      I_Contact( "PLC2_Load_Default_Cmd_Nhan_Eff" )
      R_Coil( "PLC2_Load_Default_Done" )
   END_RUNG
   // the same network as SCL:
   IF NOT "PLC2_Load_Default_Cmd_Nhan_Eff" THEN "PLC2_Load_Default_Done" := FALSE; END_IF;
END_REGION
END_FUNCTION

FUNCTION "FC_PLC2_Mixing" : Void   // FC20, LAD
{ S7_Optimized_Access := 'TRUE' }
VERSION : 0.1
// stored: AutoNumber true, IsIECCheckEnabled false, SetENOAutomatically false, UDAEnableTagReadback false
   VAR_TEMP   // added for the SCL form of the ladder/FBD networks
      _w1 : Bool;
   END_VAR
BEGIN

REGION Network 1: Khóa nút nhấn Start HMI qua Run Enable PLC2
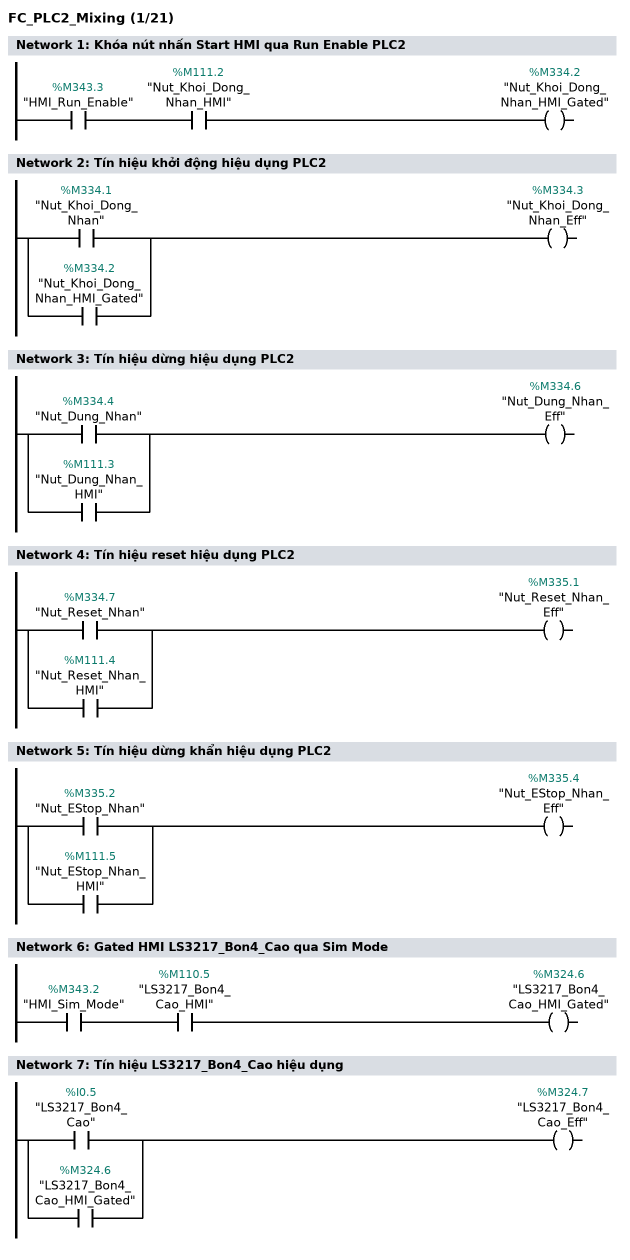
   RUNG wire#powerrail
      Contact( "HMI_Run_Enable" )
      Contact( "Nut_Khoi_Dong_Nhan_HMI" )
      Coil( "Nut_Khoi_Dong_Nhan_HMI_Gated" )
   END_RUNG
   // the same network as SCL:
   "Nut_Khoi_Dong_Nhan_HMI_Gated" := "HMI_Run_Enable" AND "Nut_Khoi_Dong_Nhan_HMI";
END_REGION

REGION Network 2: Tín hiệu khởi động hiệu dụng PLC2
   RUNG wire#powerrail
      Contact( "Nut_Khoi_Dong_Nhan" )
      wire#w1
      Coil( "Nut_Khoi_Dong_Nhan_Eff" )
   END_RUNG
   RUNG wire#powerrail
      Contact( "Nut_Khoi_Dong_Nhan_HMI_Gated" )
   END_RUNG wire#w1
   // the same network as SCL:
   "Nut_Khoi_Dong_Nhan_Eff" := "Nut_Khoi_Dong_Nhan" OR "Nut_Khoi_Dong_Nhan_HMI_Gated";
END_REGION

REGION Network 3: Tín hiệu dừng hiệu dụng PLC2
   RUNG wire#powerrail
      Contact( "Nut_Dung_Nhan" )
      wire#w1
      Coil( "Nut_Dung_Nhan_Eff" )
   END_RUNG
   RUNG wire#powerrail
      Contact( "Nut_Dung_Nhan_HMI" )
   END_RUNG wire#w1
   // the same network as SCL:
   "Nut_Dung_Nhan_Eff" := "Nut_Dung_Nhan" OR "Nut_Dung_Nhan_HMI";
END_REGION

REGION Network 4: Tín hiệu reset hiệu dụng PLC2
   RUNG wire#powerrail
      Contact( "Nut_Reset_Nhan" )
      wire#w1
      Coil( "Nut_Reset_Nhan_Eff" )
   END_RUNG
   RUNG wire#powerrail
      Contact( "Nut_Reset_Nhan_HMI" )
   END_RUNG wire#w1
   // the same network as SCL:
   "Nut_Reset_Nhan_Eff" := "Nut_Reset_Nhan" OR "Nut_Reset_Nhan_HMI";
END_REGION

REGION Network 5: Tín hiệu dừng khẩn hiệu dụng PLC2
   RUNG wire#powerrail
      Contact( "Nut_EStop_Nhan" )
      wire#w1
      Coil( "Nut_EStop_Nhan_Eff" )
   END_RUNG
   RUNG wire#powerrail
      Contact( "Nut_EStop_Nhan_HMI" )
   END_RUNG wire#w1
   // the same network as SCL:
   "Nut_EStop_Nhan_Eff" := "Nut_EStop_Nhan" OR "Nut_EStop_Nhan_HMI";
END_REGION

REGION Network 6: Gated HMI LS3217_Bon4_Cao qua Sim Mode
   RUNG wire#powerrail
      Contact( "HMI_Sim_Mode" )
      Contact( "LS3217_Bon4_Cao_HMI" )
      Coil( "LS3217_Bon4_Cao_HMI_Gated" )
   END_RUNG
   // the same network as SCL:
   "LS3217_Bon4_Cao_HMI_Gated" := "HMI_Sim_Mode" AND "LS3217_Bon4_Cao_HMI";
END_REGION

REGION Network 7: Tín hiệu LS3217_Bon4_Cao hiệu dụng
   RUNG wire#powerrail
      Contact( "LS3217_Bon4_Cao" )
      wire#w1
      Coil( "LS3217_Bon4_Cao_Eff" )
   END_RUNG
   RUNG wire#powerrail
      Contact( "LS3217_Bon4_Cao_HMI_Gated" )
   END_RUNG wire#w1
   // the same network as SCL:
   "LS3217_Bon4_Cao_Eff" := "LS3217_Bon4_Cao" OR "LS3217_Bon4_Cao_HMI_Gated";
END_REGION

REGION Network 8: Gated HMI Pump3265_Chuyen_Nhanh2_Cmd_Nhan qua Sim Mode
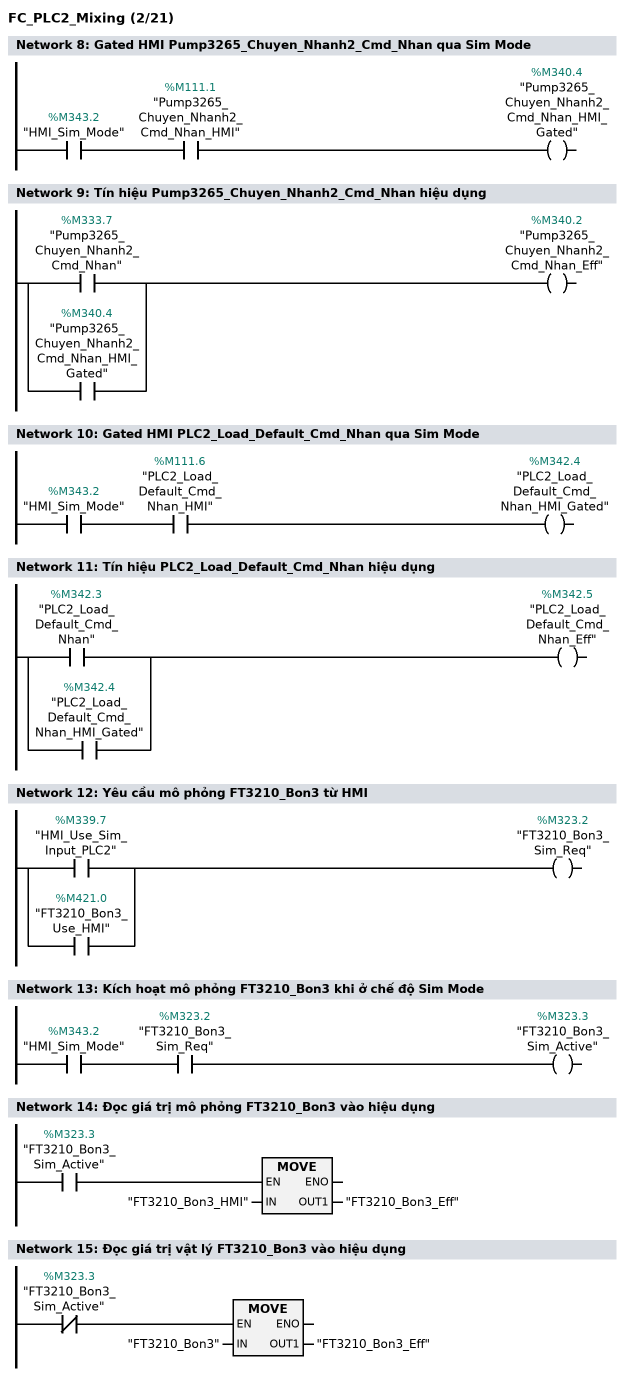
   RUNG wire#powerrail
      Contact( "HMI_Sim_Mode" )
      Contact( "Pump3265_Chuyen_Nhanh2_Cmd_Nhan_HMI" )
      Coil( "Pump3265_Chuyen_Nhanh2_Cmd_Nhan_HMI_Gated" )
   END_RUNG
   // the same network as SCL:
   "Pump3265_Chuyen_Nhanh2_Cmd_Nhan_HMI_Gated" := "HMI_Sim_Mode" AND "Pump3265_Chuyen_Nhanh2_Cmd_Nhan_HMI";
END_REGION

REGION Network 9: Tín hiệu Pump3265_Chuyen_Nhanh2_Cmd_Nhan hiệu dụng
   RUNG wire#powerrail
      Contact( "Pump3265_Chuyen_Nhanh2_Cmd_Nhan" )
      wire#w1
      Coil( "Pump3265_Chuyen_Nhanh2_Cmd_Nhan_Eff" )
   END_RUNG
   RUNG wire#powerrail
      Contact( "Pump3265_Chuyen_Nhanh2_Cmd_Nhan_HMI_Gated" )
   END_RUNG wire#w1
   // the same network as SCL:
   "Pump3265_Chuyen_Nhanh2_Cmd_Nhan_Eff" := "Pump3265_Chuyen_Nhanh2_Cmd_Nhan" OR "Pump3265_Chuyen_Nhanh2_Cmd_Nhan_HMI_Gated";
END_REGION

REGION Network 10: Gated HMI PLC2_Load_Default_Cmd_Nhan qua Sim Mode
   RUNG wire#powerrail
      Contact( "HMI_Sim_Mode" )
      Contact( "PLC2_Load_Default_Cmd_Nhan_HMI" )
      Coil( "PLC2_Load_Default_Cmd_Nhan_HMI_Gated" )
   END_RUNG
   // the same network as SCL:
   "PLC2_Load_Default_Cmd_Nhan_HMI_Gated" := "HMI_Sim_Mode" AND "PLC2_Load_Default_Cmd_Nhan_HMI";
END_REGION

REGION Network 11: Tín hiệu PLC2_Load_Default_Cmd_Nhan hiệu dụng
   RUNG wire#powerrail
      Contact( "PLC2_Load_Default_Cmd_Nhan" )
      wire#w1
      Coil( "PLC2_Load_Default_Cmd_Nhan_Eff" )
   END_RUNG
   RUNG wire#powerrail
      Contact( "PLC2_Load_Default_Cmd_Nhan_HMI_Gated" )
   END_RUNG wire#w1
   // the same network as SCL:
   "PLC2_Load_Default_Cmd_Nhan_Eff" := "PLC2_Load_Default_Cmd_Nhan" OR "PLC2_Load_Default_Cmd_Nhan_HMI_Gated";
END_REGION

REGION Network 12: Yêu cầu mô phỏng FT3210_Bon3 từ HMI
   RUNG wire#powerrail
      Contact( "HMI_Use_Sim_Input_PLC2" )
      wire#w1
      Coil( "FT3210_Bon3_Sim_Req" )
   END_RUNG
   RUNG wire#powerrail
      Contact( "FT3210_Bon3_Use_HMI" )
   END_RUNG wire#w1
   // the same network as SCL:
   "FT3210_Bon3_Sim_Req" := "HMI_Use_Sim_Input_PLC2" OR "FT3210_Bon3_Use_HMI";
END_REGION

REGION Network 13: Kích hoạt mô phỏng FT3210_Bon3 khi ở chế độ Sim Mode
   RUNG wire#powerrail
      Contact( "HMI_Sim_Mode" )
      Contact( "FT3210_Bon3_Sim_Req" )
      Coil( "FT3210_Bon3_Sim_Active" )
   END_RUNG
   // the same network as SCL:
   "FT3210_Bon3_Sim_Active" := "HMI_Sim_Mode" AND "FT3210_Bon3_Sim_Req";
END_REGION

REGION Network 14: Đọc giá trị mô phỏng FT3210_Bon3 vào hiệu dụng
   RUNG wire#powerrail
      Contact( "FT3210_Bon3_Sim_Active" )
      { S7_GenerateENO := "TRUE" } Move(in := "FT3210_Bon3_HMI", out1 => "FT3210_Bon3_Eff")
   END_RUNG
   // the same network as SCL:
   IF "FT3210_Bon3_Sim_Active" THEN "FT3210_Bon3_Eff" := "FT3210_Bon3_HMI"; END_IF;
END_REGION

REGION Network 15: Đọc giá trị vật lý FT3210_Bon3 vào hiệu dụng
   RUNG wire#powerrail
      I_Contact( "FT3210_Bon3_Sim_Active" )
      { S7_GenerateENO := "TRUE" } Move(in := "FT3210_Bon3", out1 => "FT3210_Bon3_Eff")
   END_RUNG
   // the same network as SCL:
   IF NOT "FT3210_Bon3_Sim_Active" THEN "FT3210_Bon3_Eff" := "FT3210_Bon3"; END_IF;
END_REGION

REGION Network 16: Yêu cầu mô phỏng FQ3210_Bon3 từ HMI
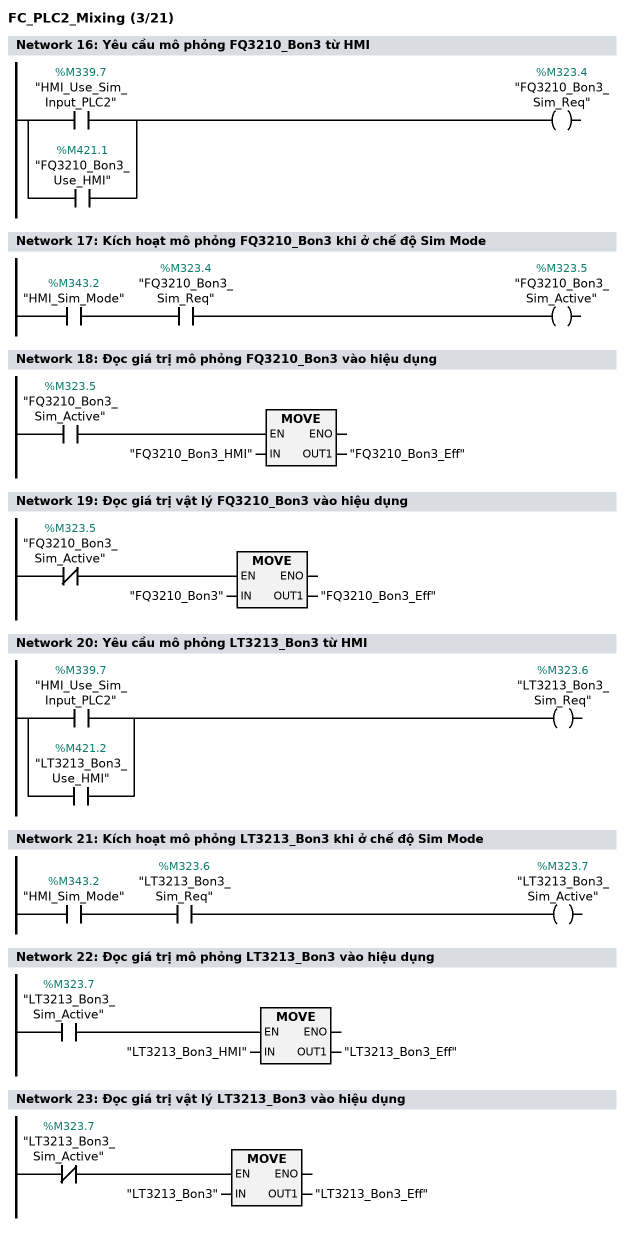
   RUNG wire#powerrail
      Contact( "HMI_Use_Sim_Input_PLC2" )
      wire#w1
      Coil( "FQ3210_Bon3_Sim_Req" )
   END_RUNG
   RUNG wire#powerrail
      Contact( "FQ3210_Bon3_Use_HMI" )
   END_RUNG wire#w1
   // the same network as SCL:
   "FQ3210_Bon3_Sim_Req" := "HMI_Use_Sim_Input_PLC2" OR "FQ3210_Bon3_Use_HMI";
END_REGION

REGION Network 17: Kích hoạt mô phỏng FQ3210_Bon3 khi ở chế độ Sim Mode
   RUNG wire#powerrail
      Contact( "HMI_Sim_Mode" )
      Contact( "FQ3210_Bon3_Sim_Req" )
      Coil( "FQ3210_Bon3_Sim_Active" )
   END_RUNG
   // the same network as SCL:
   "FQ3210_Bon3_Sim_Active" := "HMI_Sim_Mode" AND "FQ3210_Bon3_Sim_Req";
END_REGION

REGION Network 18: Đọc giá trị mô phỏng FQ3210_Bon3 vào hiệu dụng
   RUNG wire#powerrail
      Contact( "FQ3210_Bon3_Sim_Active" )
      { S7_GenerateENO := "TRUE" } Move(in := "FQ3210_Bon3_HMI", out1 => "FQ3210_Bon3_Eff")
   END_RUNG
   // the same network as SCL:
   IF "FQ3210_Bon3_Sim_Active" THEN "FQ3210_Bon3_Eff" := "FQ3210_Bon3_HMI"; END_IF;
END_REGION

REGION Network 19: Đọc giá trị vật lý FQ3210_Bon3 vào hiệu dụng
   RUNG wire#powerrail
      I_Contact( "FQ3210_Bon3_Sim_Active" )
      { S7_GenerateENO := "TRUE" } Move(in := "FQ3210_Bon3", out1 => "FQ3210_Bon3_Eff")
   END_RUNG
   // the same network as SCL:
   IF NOT "FQ3210_Bon3_Sim_Active" THEN "FQ3210_Bon3_Eff" := "FQ3210_Bon3"; END_IF;
END_REGION

REGION Network 20: Yêu cầu mô phỏng LT3213_Bon3 từ HMI
   RUNG wire#powerrail
      Contact( "HMI_Use_Sim_Input_PLC2" )
      wire#w1
      Coil( "LT3213_Bon3_Sim_Req" )
   END_RUNG
   RUNG wire#powerrail
      Contact( "LT3213_Bon3_Use_HMI" )
   END_RUNG wire#w1
   // the same network as SCL:
   "LT3213_Bon3_Sim_Req" := "HMI_Use_Sim_Input_PLC2" OR "LT3213_Bon3_Use_HMI";
END_REGION

REGION Network 21: Kích hoạt mô phỏng LT3213_Bon3 khi ở chế độ Sim Mode
   RUNG wire#powerrail
      Contact( "HMI_Sim_Mode" )
      Contact( "LT3213_Bon3_Sim_Req" )
      Coil( "LT3213_Bon3_Sim_Active" )
   END_RUNG
   // the same network as SCL:
   "LT3213_Bon3_Sim_Active" := "HMI_Sim_Mode" AND "LT3213_Bon3_Sim_Req";
END_REGION

REGION Network 22: Đọc giá trị mô phỏng LT3213_Bon3 vào hiệu dụng
   RUNG wire#powerrail
      Contact( "LT3213_Bon3_Sim_Active" )
      { S7_GenerateENO := "TRUE" } Move(in := "LT3213_Bon3_HMI", out1 => "LT3213_Bon3_Eff")
   END_RUNG
   // the same network as SCL:
   IF "LT3213_Bon3_Sim_Active" THEN "LT3213_Bon3_Eff" := "LT3213_Bon3_HMI"; END_IF;
END_REGION

REGION Network 23: Đọc giá trị vật lý LT3213_Bon3 vào hiệu dụng
   RUNG wire#powerrail
      I_Contact( "LT3213_Bon3_Sim_Active" )
      { S7_GenerateENO := "TRUE" } Move(in := "LT3213_Bon3", out1 => "LT3213_Bon3_Eff")
   END_RUNG
   // the same network as SCL:
   IF NOT "LT3213_Bon3_Sim_Active" THEN "LT3213_Bon3_Eff" := "LT3213_Bon3"; END_IF;
END_REGION

REGION Network 24: Yêu cầu mô phỏng TT3214_Bon3 từ HMI
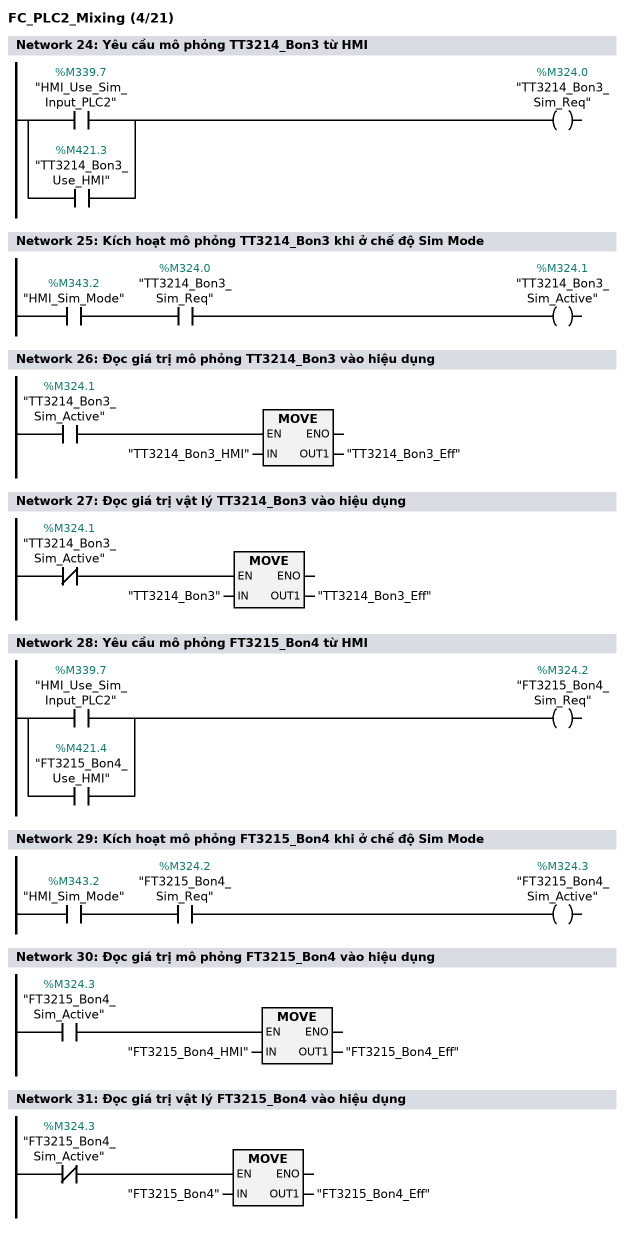
   RUNG wire#powerrail
      Contact( "HMI_Use_Sim_Input_PLC2" )
      wire#w1
      Coil( "TT3214_Bon3_Sim_Req" )
   END_RUNG
   RUNG wire#powerrail
      Contact( "TT3214_Bon3_Use_HMI" )
   END_RUNG wire#w1
   // the same network as SCL:
   "TT3214_Bon3_Sim_Req" := "HMI_Use_Sim_Input_PLC2" OR "TT3214_Bon3_Use_HMI";
END_REGION

REGION Network 25: Kích hoạt mô phỏng TT3214_Bon3 khi ở chế độ Sim Mode
   RUNG wire#powerrail
      Contact( "HMI_Sim_Mode" )
      Contact( "TT3214_Bon3_Sim_Req" )
      Coil( "TT3214_Bon3_Sim_Active" )
   END_RUNG
   // the same network as SCL:
   "TT3214_Bon3_Sim_Active" := "HMI_Sim_Mode" AND "TT3214_Bon3_Sim_Req";
END_REGION

REGION Network 26: Đọc giá trị mô phỏng TT3214_Bon3 vào hiệu dụng
   RUNG wire#powerrail
      Contact( "TT3214_Bon3_Sim_Active" )
      { S7_GenerateENO := "TRUE" } Move(in := "TT3214_Bon3_HMI", out1 => "TT3214_Bon3_Eff")
   END_RUNG
   // the same network as SCL:
   IF "TT3214_Bon3_Sim_Active" THEN "TT3214_Bon3_Eff" := "TT3214_Bon3_HMI"; END_IF;
END_REGION

REGION Network 27: Đọc giá trị vật lý TT3214_Bon3 vào hiệu dụng
   RUNG wire#powerrail
      I_Contact( "TT3214_Bon3_Sim_Active" )
      { S7_GenerateENO := "TRUE" } Move(in := "TT3214_Bon3", out1 => "TT3214_Bon3_Eff")
   END_RUNG
   // the same network as SCL:
   IF NOT "TT3214_Bon3_Sim_Active" THEN "TT3214_Bon3_Eff" := "TT3214_Bon3"; END_IF;
END_REGION

REGION Network 28: Yêu cầu mô phỏng FT3215_Bon4 từ HMI
   RUNG wire#powerrail
      Contact( "HMI_Use_Sim_Input_PLC2" )
      wire#w1
      Coil( "FT3215_Bon4_Sim_Req" )
   END_RUNG
   RUNG wire#powerrail
      Contact( "FT3215_Bon4_Use_HMI" )
   END_RUNG wire#w1
   // the same network as SCL:
   "FT3215_Bon4_Sim_Req" := "HMI_Use_Sim_Input_PLC2" OR "FT3215_Bon4_Use_HMI";
END_REGION

REGION Network 29: Kích hoạt mô phỏng FT3215_Bon4 khi ở chế độ Sim Mode
   RUNG wire#powerrail
      Contact( "HMI_Sim_Mode" )
      Contact( "FT3215_Bon4_Sim_Req" )
      Coil( "FT3215_Bon4_Sim_Active" )
   END_RUNG
   // the same network as SCL:
   "FT3215_Bon4_Sim_Active" := "HMI_Sim_Mode" AND "FT3215_Bon4_Sim_Req";
END_REGION

REGION Network 30: Đọc giá trị mô phỏng FT3215_Bon4 vào hiệu dụng
   RUNG wire#powerrail
      Contact( "FT3215_Bon4_Sim_Active" )
      { S7_GenerateENO := "TRUE" } Move(in := "FT3215_Bon4_HMI", out1 => "FT3215_Bon4_Eff")
   END_RUNG
   // the same network as SCL:
   IF "FT3215_Bon4_Sim_Active" THEN "FT3215_Bon4_Eff" := "FT3215_Bon4_HMI"; END_IF;
END_REGION

REGION Network 31: Đọc giá trị vật lý FT3215_Bon4 vào hiệu dụng
   RUNG wire#powerrail
      I_Contact( "FT3215_Bon4_Sim_Active" )
      { S7_GenerateENO := "TRUE" } Move(in := "FT3215_Bon4", out1 => "FT3215_Bon4_Eff")
   END_RUNG
   // the same network as SCL:
   IF NOT "FT3215_Bon4_Sim_Active" THEN "FT3215_Bon4_Eff" := "FT3215_Bon4"; END_IF;
END_REGION

REGION Network 32: Yêu cầu mô phỏng FQ3215_Bon4 từ HMI
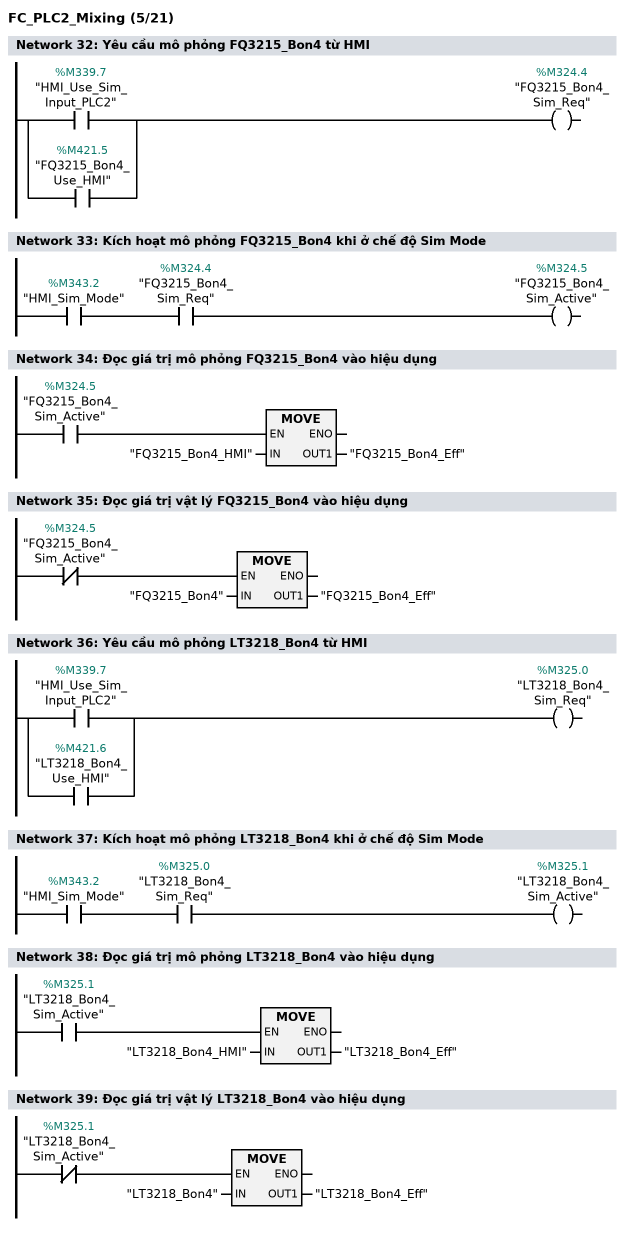
   RUNG wire#powerrail
      Contact( "HMI_Use_Sim_Input_PLC2" )
      wire#w1
      Coil( "FQ3215_Bon4_Sim_Req" )
   END_RUNG
   RUNG wire#powerrail
      Contact( "FQ3215_Bon4_Use_HMI" )
   END_RUNG wire#w1
   // the same network as SCL:
   "FQ3215_Bon4_Sim_Req" := "HMI_Use_Sim_Input_PLC2" OR "FQ3215_Bon4_Use_HMI";
END_REGION

REGION Network 33: Kích hoạt mô phỏng FQ3215_Bon4 khi ở chế độ Sim Mode
   RUNG wire#powerrail
      Contact( "HMI_Sim_Mode" )
      Contact( "FQ3215_Bon4_Sim_Req" )
      Coil( "FQ3215_Bon4_Sim_Active" )
   END_RUNG
   // the same network as SCL:
   "FQ3215_Bon4_Sim_Active" := "HMI_Sim_Mode" AND "FQ3215_Bon4_Sim_Req";
END_REGION

REGION Network 34: Đọc giá trị mô phỏng FQ3215_Bon4 vào hiệu dụng
   RUNG wire#powerrail
      Contact( "FQ3215_Bon4_Sim_Active" )
      { S7_GenerateENO := "TRUE" } Move(in := "FQ3215_Bon4_HMI", out1 => "FQ3215_Bon4_Eff")
   END_RUNG
   // the same network as SCL:
   IF "FQ3215_Bon4_Sim_Active" THEN "FQ3215_Bon4_Eff" := "FQ3215_Bon4_HMI"; END_IF;
END_REGION

REGION Network 35: Đọc giá trị vật lý FQ3215_Bon4 vào hiệu dụng
   RUNG wire#powerrail
      I_Contact( "FQ3215_Bon4_Sim_Active" )
      { S7_GenerateENO := "TRUE" } Move(in := "FQ3215_Bon4", out1 => "FQ3215_Bon4_Eff")
   END_RUNG
   // the same network as SCL:
   IF NOT "FQ3215_Bon4_Sim_Active" THEN "FQ3215_Bon4_Eff" := "FQ3215_Bon4"; END_IF;
END_REGION

REGION Network 36: Yêu cầu mô phỏng LT3218_Bon4 từ HMI
   RUNG wire#powerrail
      Contact( "HMI_Use_Sim_Input_PLC2" )
      wire#w1
      Coil( "LT3218_Bon4_Sim_Req" )
   END_RUNG
   RUNG wire#powerrail
      Contact( "LT3218_Bon4_Use_HMI" )
   END_RUNG wire#w1
   // the same network as SCL:
   "LT3218_Bon4_Sim_Req" := "HMI_Use_Sim_Input_PLC2" OR "LT3218_Bon4_Use_HMI";
END_REGION

REGION Network 37: Kích hoạt mô phỏng LT3218_Bon4 khi ở chế độ Sim Mode
   RUNG wire#powerrail
      Contact( "HMI_Sim_Mode" )
      Contact( "LT3218_Bon4_Sim_Req" )
      Coil( "LT3218_Bon4_Sim_Active" )
   END_RUNG
   // the same network as SCL:
   "LT3218_Bon4_Sim_Active" := "HMI_Sim_Mode" AND "LT3218_Bon4_Sim_Req";
END_REGION

REGION Network 38: Đọc giá trị mô phỏng LT3218_Bon4 vào hiệu dụng
   RUNG wire#powerrail
      Contact( "LT3218_Bon4_Sim_Active" )
      { S7_GenerateENO := "TRUE" } Move(in := "LT3218_Bon4_HMI", out1 => "LT3218_Bon4_Eff")
   END_RUNG
   // the same network as SCL:
   IF "LT3218_Bon4_Sim_Active" THEN "LT3218_Bon4_Eff" := "LT3218_Bon4_HMI"; END_IF;
END_REGION

REGION Network 39: Đọc giá trị vật lý LT3218_Bon4 vào hiệu dụng
   RUNG wire#powerrail
      I_Contact( "LT3218_Bon4_Sim_Active" )
      { S7_GenerateENO := "TRUE" } Move(in := "LT3218_Bon4", out1 => "LT3218_Bon4_Eff")
   END_RUNG
   // the same network as SCL:
   IF NOT "LT3218_Bon4_Sim_Active" THEN "LT3218_Bon4_Eff" := "LT3218_Bon4"; END_IF;
END_REGION

REGION Network 40: Yêu cầu mô phỏng TT3219_Bon4 từ HMI
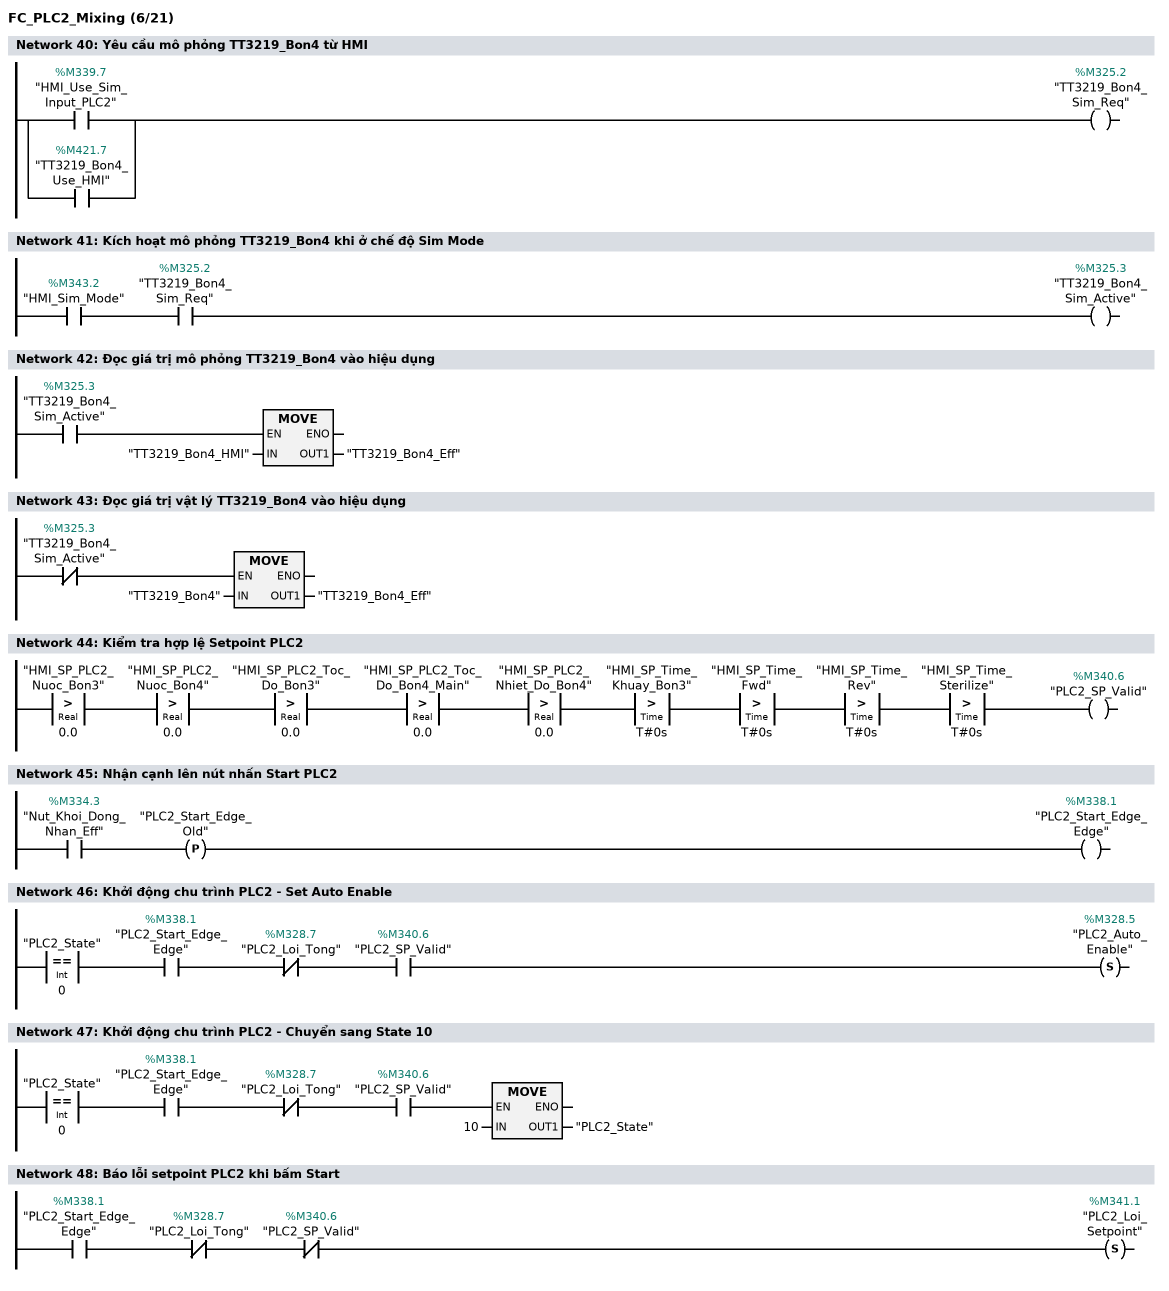
   RUNG wire#powerrail
      Contact( "HMI_Use_Sim_Input_PLC2" )
      wire#w1
      Coil( "TT3219_Bon4_Sim_Req" )
   END_RUNG
   RUNG wire#powerrail
      Contact( "TT3219_Bon4_Use_HMI" )
   END_RUNG wire#w1
   // the same network as SCL:
   "TT3219_Bon4_Sim_Req" := "HMI_Use_Sim_Input_PLC2" OR "TT3219_Bon4_Use_HMI";
END_REGION

REGION Network 41: Kích hoạt mô phỏng TT3219_Bon4 khi ở chế độ Sim Mode
   RUNG wire#powerrail
      Contact( "HMI_Sim_Mode" )
      Contact( "TT3219_Bon4_Sim_Req" )
      Coil( "TT3219_Bon4_Sim_Active" )
   END_RUNG
   // the same network as SCL:
   "TT3219_Bon4_Sim_Active" := "HMI_Sim_Mode" AND "TT3219_Bon4_Sim_Req";
END_REGION

REGION Network 42: Đọc giá trị mô phỏng TT3219_Bon4 vào hiệu dụng
   RUNG wire#powerrail
      Contact( "TT3219_Bon4_Sim_Active" )
      { S7_GenerateENO := "TRUE" } Move(in := "TT3219_Bon4_HMI", out1 => "TT3219_Bon4_Eff")
   END_RUNG
   // the same network as SCL:
   IF "TT3219_Bon4_Sim_Active" THEN "TT3219_Bon4_Eff" := "TT3219_Bon4_HMI"; END_IF;
END_REGION

REGION Network 43: Đọc giá trị vật lý TT3219_Bon4 vào hiệu dụng
   RUNG wire#powerrail
      I_Contact( "TT3219_Bon4_Sim_Active" )
      { S7_GenerateENO := "TRUE" } Move(in := "TT3219_Bon4", out1 => "TT3219_Bon4_Eff")
   END_RUNG
   // the same network as SCL:
   IF NOT "TT3219_Bon4_Sim_Active" THEN "TT3219_Bon4_Eff" := "TT3219_Bon4"; END_IF;
END_REGION

REGION Network 44: Kiểm tra hợp lệ Setpoint PLC2
   RUNG wire#powerrail
      { S7_Templates := "SrcType := Real" } GT_Contact(in1 := "HMI_SP_PLC2_Nuoc_Bon3", in2 := 0.0)
      { S7_Templates := "SrcType := Real" } GT_Contact(in1 := "HMI_SP_PLC2_Nuoc_Bon4", in2 := 0.0)
      { S7_Templates := "SrcType := Real" } GT_Contact(in1 := "HMI_SP_PLC2_Toc_Do_Bon3", in2 := 0.0)
      { S7_Templates := "SrcType := Real" } GT_Contact(in1 := "HMI_SP_PLC2_Toc_Do_Bon4_Main", in2 := 0.0)
      { S7_Templates := "SrcType := Real" } GT_Contact(in1 := "HMI_SP_PLC2_Nhiet_Do_Bon4", in2 := 0.0)
      { S7_Templates := "SrcType := Time" } GT_Contact(in1 := "HMI_SP_Time_Khuay_Bon3", in2 := T#0s)
      { S7_Templates := "SrcType := Time" } GT_Contact(in1 := "HMI_SP_Time_Fwd", in2 := T#0s)
      { S7_Templates := "SrcType := Time" } GT_Contact(in1 := "HMI_SP_Time_Rev", in2 := T#0s)
      { S7_Templates := "SrcType := Time" } GT_Contact(in1 := "HMI_SP_Time_Sterilize", in2 := T#0s)
      Coil( "PLC2_SP_Valid" )
   END_RUNG
   // the same network as SCL:
   "PLC2_SP_Valid" := ("HMI_SP_PLC2_Nuoc_Bon3" > 0.0) AND ("HMI_SP_PLC2_Nuoc_Bon4" > 0.0) AND ("HMI_SP_PLC2_Toc_Do_Bon3" > 0.0) AND ("HMI_SP_PLC2_Toc_Do_Bon4_Main" > 0.0) AND ("HMI_SP_PLC2_Nhiet_Do_Bon4" > 0.0) AND ("HMI_SP_Time_Khuay_Bon3" > T#0s) AND ("HMI_SP_Time_Fwd" > T#0s) AND ("HMI_SP_Time_Rev" > T#0s) AND ("HMI_SP_Time_Sterilize" > T#0s);
END_REGION

REGION Network 45: Nhận cạnh lên nút nhấn Start PLC2
   RUNG wire#powerrail
      Contact( "Nut_Khoi_Dong_Nhan_Eff" )
      P_Trig( "PLC2_Start_Edge_Old" )
      Coil( "PLC2_Start_Edge_Edge" )
   END_RUNG
   // the same network as SCL:
   #_w1 := "Nut_Khoi_Dong_Nhan_Eff" AND NOT "PLC2_Start_Edge_Old";   // rising edge
   "PLC2_Start_Edge_Old" := "Nut_Khoi_Dong_Nhan_Eff";
   "PLC2_Start_Edge_Edge" := #_w1;
END_REGION

REGION Network 46: Khởi động chu trình PLC2 - Set Auto Enable
   RUNG wire#powerrail
      { S7_Templates := "SrcType := Int" } EQ_Contact(in1 := "PLC2_State", in2 := 0)
      Contact( "PLC2_Start_Edge_Edge" )
      I_Contact( "PLC2_Loi_Tong" )
      Contact( "PLC2_SP_Valid" )
      S_Coil( "PLC2_Auto_Enable" )
   END_RUNG
   // the same network as SCL:
   IF ("PLC2_State" = 0) AND "PLC2_Start_Edge_Edge" AND NOT "PLC2_Loi_Tong" AND "PLC2_SP_Valid" THEN
       "PLC2_Auto_Enable" := TRUE;
   END_IF;
END_REGION

REGION Network 47: Khởi động chu trình PLC2 - Chuyển sang State 10
   RUNG wire#powerrail
      { S7_Templates := "SrcType := Int" } EQ_Contact(in1 := "PLC2_State", in2 := 0)
      Contact( "PLC2_Start_Edge_Edge" )
      I_Contact( "PLC2_Loi_Tong" )
      Contact( "PLC2_SP_Valid" )
      { S7_GenerateENO := "TRUE" } Move(in := 10, out1 => "PLC2_State")
   END_RUNG
   // the same network as SCL:
   IF ("PLC2_State" = 0) AND "PLC2_Start_Edge_Edge" AND NOT "PLC2_Loi_Tong" AND "PLC2_SP_Valid" THEN
       "PLC2_State" := 10;
   END_IF;
END_REGION

REGION Network 48: Báo lỗi setpoint PLC2 khi bấm Start
   RUNG wire#powerrail
      Contact( "PLC2_Start_Edge_Edge" )
      I_Contact( "PLC2_Loi_Tong" )
      I_Contact( "PLC2_SP_Valid" )
      S_Coil( "PLC2_Loi_Setpoint" )
   END_RUNG
   // the same network as SCL:
   IF "PLC2_Start_Edge_Edge" AND NOT "PLC2_Loi_Tong" AND NOT "PLC2_SP_Valid" THEN
       "PLC2_Loi_Setpoint" := TRUE;
   END_IF;
END_REGION

REGION Network 49: Stop PLC2 từ HMI dùng chung
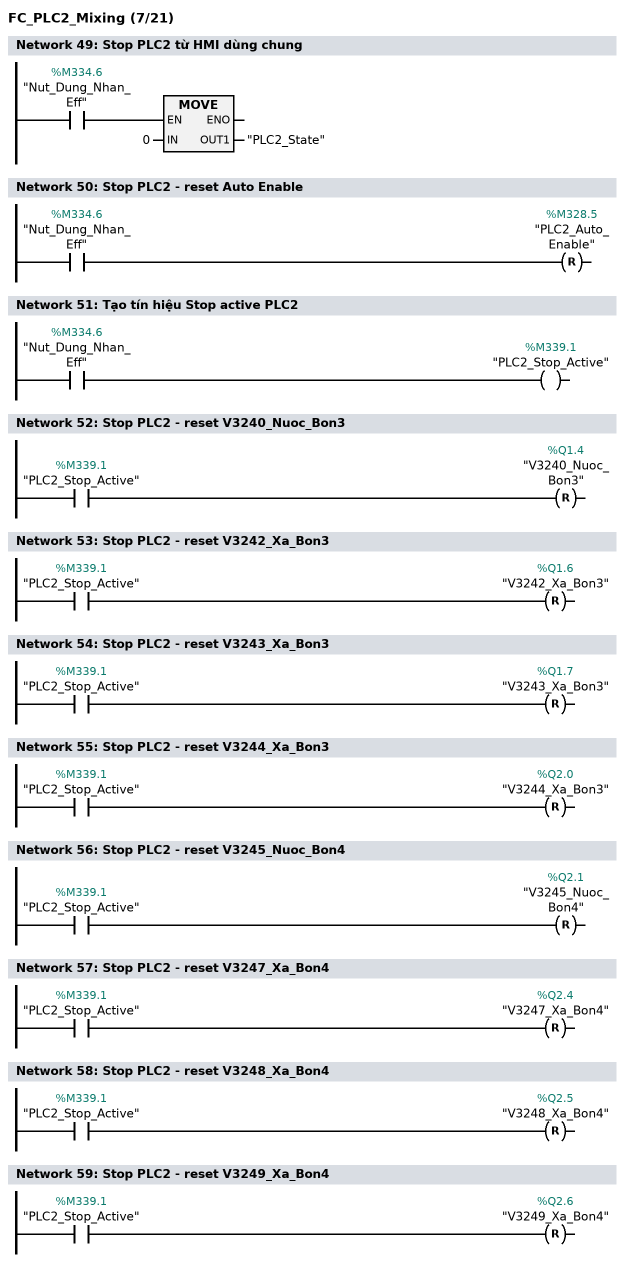
   RUNG wire#powerrail
      Contact( "Nut_Dung_Nhan_Eff" )
      { S7_GenerateENO := "TRUE" } Move(in := 0, out1 => "PLC2_State")
   END_RUNG
   // the same network as SCL:
   IF "Nut_Dung_Nhan_Eff" THEN "PLC2_State" := 0; END_IF;
END_REGION

REGION Network 50: Stop PLC2 - reset Auto Enable
   RUNG wire#powerrail
      Contact( "Nut_Dung_Nhan_Eff" )
      R_Coil( "PLC2_Auto_Enable" )
   END_RUNG
   // the same network as SCL:
   IF "Nut_Dung_Nhan_Eff" THEN "PLC2_Auto_Enable" := FALSE; END_IF;
END_REGION

REGION Network 51: Tạo tín hiệu Stop active PLC2
   RUNG wire#powerrail
      Contact( "Nut_Dung_Nhan_Eff" )
      Coil( "PLC2_Stop_Active" )
   END_RUNG
   // the same network as SCL:
   "PLC2_Stop_Active" := "Nut_Dung_Nhan_Eff";
END_REGION

REGION Network 52: Stop PLC2 - reset V3240_Nuoc_Bon3
   RUNG wire#powerrail
      Contact( "PLC2_Stop_Active" )
      R_Coil( "V3240_Nuoc_Bon3" )
   END_RUNG
   // the same network as SCL:
   IF "PLC2_Stop_Active" THEN "V3240_Nuoc_Bon3" := FALSE; END_IF;
END_REGION

REGION Network 53: Stop PLC2 - reset V3242_Xa_Bon3
   RUNG wire#powerrail
      Contact( "PLC2_Stop_Active" )
      R_Coil( "V3242_Xa_Bon3" )
   END_RUNG
   // the same network as SCL:
   IF "PLC2_Stop_Active" THEN "V3242_Xa_Bon3" := FALSE; END_IF;
END_REGION

REGION Network 54: Stop PLC2 - reset V3243_Xa_Bon3
   RUNG wire#powerrail
      Contact( "PLC2_Stop_Active" )
      R_Coil( "V3243_Xa_Bon3" )
   END_RUNG
   // the same network as SCL:
   IF "PLC2_Stop_Active" THEN "V3243_Xa_Bon3" := FALSE; END_IF;
END_REGION

REGION Network 55: Stop PLC2 - reset V3244_Xa_Bon3
   RUNG wire#powerrail
      Contact( "PLC2_Stop_Active" )
      R_Coil( "V3244_Xa_Bon3" )
   END_RUNG
   // the same network as SCL:
   IF "PLC2_Stop_Active" THEN "V3244_Xa_Bon3" := FALSE; END_IF;
END_REGION

REGION Network 56: Stop PLC2 - reset V3245_Nuoc_Bon4
   RUNG wire#powerrail
      Contact( "PLC2_Stop_Active" )
      R_Coil( "V3245_Nuoc_Bon4" )
   END_RUNG
   // the same network as SCL:
   IF "PLC2_Stop_Active" THEN "V3245_Nuoc_Bon4" := FALSE; END_IF;
END_REGION

REGION Network 57: Stop PLC2 - reset V3247_Xa_Bon4
   RUNG wire#powerrail
      Contact( "PLC2_Stop_Active" )
      R_Coil( "V3247_Xa_Bon4" )
   END_RUNG
   // the same network as SCL:
   IF "PLC2_Stop_Active" THEN "V3247_Xa_Bon4" := FALSE; END_IF;
END_REGION

REGION Network 58: Stop PLC2 - reset V3248_Xa_Bon4
   RUNG wire#powerrail
      Contact( "PLC2_Stop_Active" )
      R_Coil( "V3248_Xa_Bon4" )
   END_RUNG
   // the same network as SCL:
   IF "PLC2_Stop_Active" THEN "V3248_Xa_Bon4" := FALSE; END_IF;
END_REGION

REGION Network 59: Stop PLC2 - reset V3249_Xa_Bon4
   RUNG wire#powerrail
      Contact( "PLC2_Stop_Active" )
      R_Coil( "V3249_Xa_Bon4" )
   END_RUNG
   // the same network as SCL:
   IF "PLC2_Stop_Active" THEN "V3249_Xa_Bon4" := FALSE; END_IF;
END_REGION

REGION Network 60: Stop PLC2 - reset PID Enable
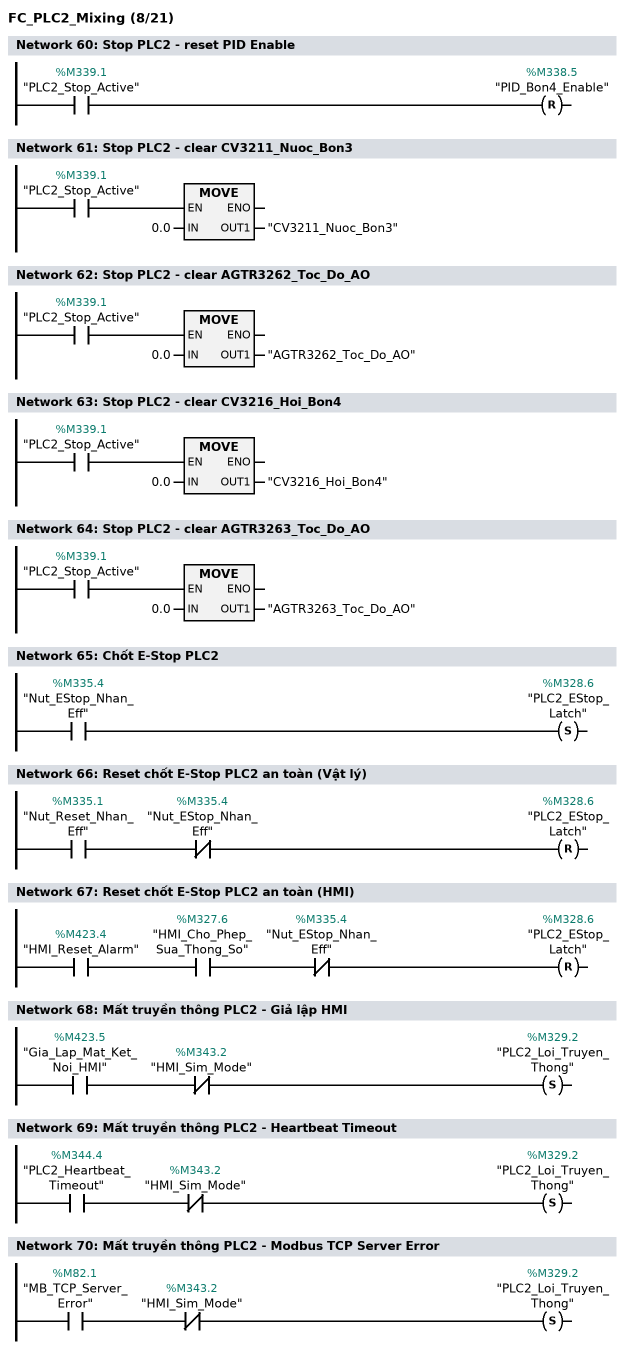
   RUNG wire#powerrail
      Contact( "PLC2_Stop_Active" )
      R_Coil( "PID_Bon4_Enable" )
   END_RUNG
   // the same network as SCL:
   IF "PLC2_Stop_Active" THEN "PID_Bon4_Enable" := FALSE; END_IF;
END_REGION

REGION Network 61: Stop PLC2 - clear CV3211_Nuoc_Bon3
   RUNG wire#powerrail
      Contact( "PLC2_Stop_Active" )
      { S7_GenerateENO := "TRUE" } Move(in := 0.0, out1 => "CV3211_Nuoc_Bon3")
   END_RUNG
   // the same network as SCL:
   IF "PLC2_Stop_Active" THEN "CV3211_Nuoc_Bon3" := 0.0; END_IF;
END_REGION

REGION Network 62: Stop PLC2 - clear AGTR3262_Toc_Do_AO
   RUNG wire#powerrail
      Contact( "PLC2_Stop_Active" )
      { S7_GenerateENO := "TRUE" } Move(in := 0.0, out1 => "AGTR3262_Toc_Do_AO")
   END_RUNG
   // the same network as SCL:
   IF "PLC2_Stop_Active" THEN "AGTR3262_Toc_Do_AO" := 0.0; END_IF;
END_REGION

REGION Network 63: Stop PLC2 - clear CV3216_Hoi_Bon4
   RUNG wire#powerrail
      Contact( "PLC2_Stop_Active" )
      { S7_GenerateENO := "TRUE" } Move(in := 0.0, out1 => "CV3216_Hoi_Bon4")
   END_RUNG
   // the same network as SCL:
   IF "PLC2_Stop_Active" THEN "CV3216_Hoi_Bon4" := 0.0; END_IF;
END_REGION

REGION Network 64: Stop PLC2 - clear AGTR3263_Toc_Do_AO
   RUNG wire#powerrail
      Contact( "PLC2_Stop_Active" )
      { S7_GenerateENO := "TRUE" } Move(in := 0.0, out1 => "AGTR3263_Toc_Do_AO")
   END_RUNG
   // the same network as SCL:
   IF "PLC2_Stop_Active" THEN "AGTR3263_Toc_Do_AO" := 0.0; END_IF;
END_REGION

REGION Network 65: Chốt E-Stop PLC2
   RUNG wire#powerrail
      Contact( "Nut_EStop_Nhan_Eff" )
      S_Coil( "PLC2_EStop_Latch" )
   END_RUNG
   // the same network as SCL:
   IF "Nut_EStop_Nhan_Eff" THEN "PLC2_EStop_Latch" := TRUE; END_IF;
END_REGION

REGION Network 66: Reset chốt E-Stop PLC2 an toàn (Vật lý)
   RUNG wire#powerrail
      Contact( "Nut_Reset_Nhan_Eff" )
      I_Contact( "Nut_EStop_Nhan_Eff" )
      R_Coil( "PLC2_EStop_Latch" )
   END_RUNG
   // the same network as SCL:
   IF "Nut_Reset_Nhan_Eff" AND NOT "Nut_EStop_Nhan_Eff" THEN "PLC2_EStop_Latch" := FALSE; END_IF;
END_REGION

REGION Network 67: Reset chốt E-Stop PLC2 an toàn (HMI)
   RUNG wire#powerrail
      Contact( "HMI_Reset_Alarm" )
      Contact( "HMI_Cho_Phep_Sua_Thong_So" )
      I_Contact( "Nut_EStop_Nhan_Eff" )
      R_Coil( "PLC2_EStop_Latch" )
   END_RUNG
   // the same network as SCL:
   IF "HMI_Reset_Alarm" AND "HMI_Cho_Phep_Sua_Thong_So" AND NOT "Nut_EStop_Nhan_Eff" THEN
       "PLC2_EStop_Latch" := FALSE;
   END_IF;
END_REGION

REGION Network 68: Mất truyền thông PLC2 - Giả lập HMI
   RUNG wire#powerrail
      Contact( "Gia_Lap_Mat_Ket_Noi_HMI" )
      I_Contact( "HMI_Sim_Mode" )
      S_Coil( "PLC2_Loi_Truyen_Thong" )
   END_RUNG
   // the same network as SCL:
   IF "Gia_Lap_Mat_Ket_Noi_HMI" AND NOT "HMI_Sim_Mode" THEN "PLC2_Loi_Truyen_Thong" := TRUE; END_IF;
END_REGION

REGION Network 69: Mất truyền thông PLC2 - Heartbeat Timeout
   RUNG wire#powerrail
      Contact( "PLC2_Heartbeat_Timeout" )
      I_Contact( "HMI_Sim_Mode" )
      S_Coil( "PLC2_Loi_Truyen_Thong" )
   END_RUNG
   // the same network as SCL:
   IF "PLC2_Heartbeat_Timeout" AND NOT "HMI_Sim_Mode" THEN "PLC2_Loi_Truyen_Thong" := TRUE; END_IF;
END_REGION

REGION Network 70: Mất truyền thông PLC2 - Modbus TCP Server Error
   RUNG wire#powerrail
      Contact( "MB_TCP_Server_Error" )
      I_Contact( "HMI_Sim_Mode" )
      S_Coil( "PLC2_Loi_Truyen_Thong" )
   END_RUNG
   // the same network as SCL:
   IF "MB_TCP_Server_Error" AND NOT "HMI_Sim_Mode" THEN "PLC2_Loi_Truyen_Thong" := TRUE; END_IF;
END_REGION

REGION Network 71: Dry Run bơm Nhánh 2
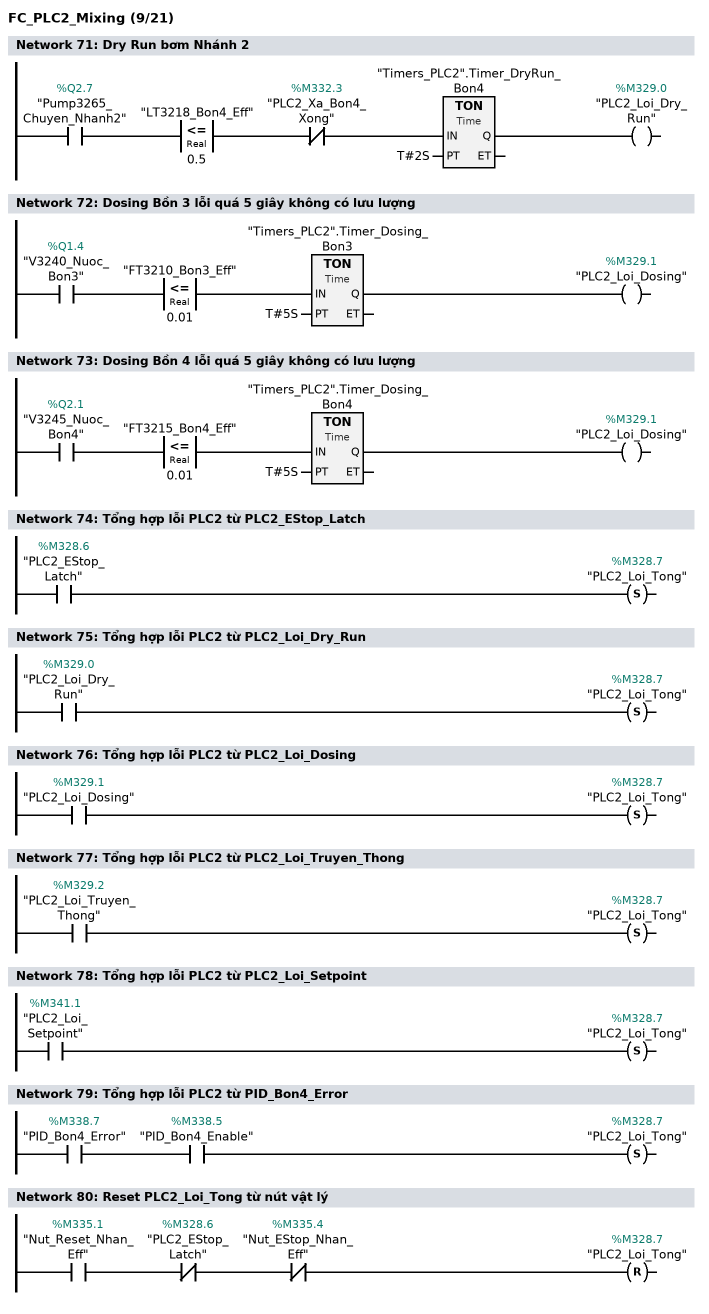
   RUNG wire#powerrail
      Contact( "Pump3265_Chuyen_Nhanh2" )
      { S7_Templates := "SrcType := Real" } LE_Contact(in1 := "LT3218_Bon4_Eff", in2 := 0.5)
      I_Contact( "PLC2_Xa_Bon4_Xong" )
      { S7_Templates := "time_type := Time" } "Timers_PLC2".Timer_DryRun_Bon4.TON(pt := T#2S, et =>)
      Coil( "PLC2_Loi_Dry_Run" )
   END_RUNG
   // the same network as SCL:
   "Timers_PLC2".Timer_DryRun_Bon4.TON(IN := "Pump3265_Chuyen_Nhanh2" AND ("LT3218_Bon4_Eff" <= 0.5) AND NOT "PLC2_Xa_Bon4_Xong",
                           PT := T#2S);
   "PLC2_Loi_Dry_Run" := "Timers_PLC2".Timer_DryRun_Bon4.Q;
END_REGION

REGION Network 72: Dosing Bồn 3 lỗi quá 5 giây không có lưu lượng
   RUNG wire#powerrail
      Contact( "V3240_Nuoc_Bon3" )
      { S7_Templates := "SrcType := Real" } LE_Contact(in1 := "FT3210_Bon3_Eff", in2 := 0.01)
      { S7_Templates := "time_type := Time" } "Timers_PLC2".Timer_Dosing_Bon3.TON(pt := T#5S, et =>)
      Coil( "PLC2_Loi_Dosing" )
   END_RUNG
   // the same network as SCL:
   "Timers_PLC2".Timer_Dosing_Bon3.TON(IN := "V3240_Nuoc_Bon3" AND ("FT3210_Bon3_Eff" <= 0.01), PT := T#5S);
   "PLC2_Loi_Dosing" := "Timers_PLC2".Timer_Dosing_Bon3.Q;
END_REGION

REGION Network 73: Dosing Bồn 4 lỗi quá 5 giây không có lưu lượng
   RUNG wire#powerrail
      Contact( "V3245_Nuoc_Bon4" )
      { S7_Templates := "SrcType := Real" } LE_Contact(in1 := "FT3215_Bon4_Eff", in2 := 0.01)
      { S7_Templates := "time_type := Time" } "Timers_PLC2".Timer_Dosing_Bon4.TON(pt := T#5S, et =>)
      Coil( "PLC2_Loi_Dosing" )
   END_RUNG
   // the same network as SCL:
   "Timers_PLC2".Timer_Dosing_Bon4.TON(IN := "V3245_Nuoc_Bon4" AND ("FT3215_Bon4_Eff" <= 0.01), PT := T#5S);
   "PLC2_Loi_Dosing" := "Timers_PLC2".Timer_Dosing_Bon4.Q;
END_REGION

REGION Network 74: Tổng hợp lỗi PLC2 từ PLC2_EStop_Latch
   RUNG wire#powerrail
      Contact( "PLC2_EStop_Latch" )
      S_Coil( "PLC2_Loi_Tong" )
   END_RUNG
   // the same network as SCL:
   IF "PLC2_EStop_Latch" THEN "PLC2_Loi_Tong" := TRUE; END_IF;
END_REGION

REGION Network 75: Tổng hợp lỗi PLC2 từ PLC2_Loi_Dry_Run
   RUNG wire#powerrail
      Contact( "PLC2_Loi_Dry_Run" )
      S_Coil( "PLC2_Loi_Tong" )
   END_RUNG
   // the same network as SCL:
   IF "PLC2_Loi_Dry_Run" THEN "PLC2_Loi_Tong" := TRUE; END_IF;
END_REGION

REGION Network 76: Tổng hợp lỗi PLC2 từ PLC2_Loi_Dosing
   RUNG wire#powerrail
      Contact( "PLC2_Loi_Dosing" )
      S_Coil( "PLC2_Loi_Tong" )
   END_RUNG
   // the same network as SCL:
   IF "PLC2_Loi_Dosing" THEN "PLC2_Loi_Tong" := TRUE; END_IF;
END_REGION

REGION Network 77: Tổng hợp lỗi PLC2 từ PLC2_Loi_Truyen_Thong
   RUNG wire#powerrail
      Contact( "PLC2_Loi_Truyen_Thong" )
      S_Coil( "PLC2_Loi_Tong" )
   END_RUNG
   // the same network as SCL:
   IF "PLC2_Loi_Truyen_Thong" THEN "PLC2_Loi_Tong" := TRUE; END_IF;
END_REGION

REGION Network 78: Tổng hợp lỗi PLC2 từ PLC2_Loi_Setpoint
   RUNG wire#powerrail
      Contact( "PLC2_Loi_Setpoint" )
      S_Coil( "PLC2_Loi_Tong" )
   END_RUNG
   // the same network as SCL:
   IF "PLC2_Loi_Setpoint" THEN "PLC2_Loi_Tong" := TRUE; END_IF;
END_REGION

REGION Network 79: Tổng hợp lỗi PLC2 từ PID_Bon4_Error
   RUNG wire#powerrail
      Contact( "PID_Bon4_Error" )
      Contact( "PID_Bon4_Enable" )
      S_Coil( "PLC2_Loi_Tong" )
   END_RUNG
   // the same network as SCL:
   IF "PID_Bon4_Error" AND "PID_Bon4_Enable" THEN "PLC2_Loi_Tong" := TRUE; END_IF;
END_REGION

REGION Network 80: Reset PLC2_Loi_Tong từ nút vật lý
   RUNG wire#powerrail
      Contact( "Nut_Reset_Nhan_Eff" )
      I_Contact( "PLC2_EStop_Latch" )
      I_Contact( "Nut_EStop_Nhan_Eff" )
      R_Coil( "PLC2_Loi_Tong" )
   END_RUNG
   // the same network as SCL:
   IF "Nut_Reset_Nhan_Eff" AND NOT "PLC2_EStop_Latch" AND NOT "Nut_EStop_Nhan_Eff" THEN
       "PLC2_Loi_Tong" := FALSE;
   END_IF;
END_REGION

REGION Network 81: Reset PLC2_Loi_Dry_Run từ nút vật lý
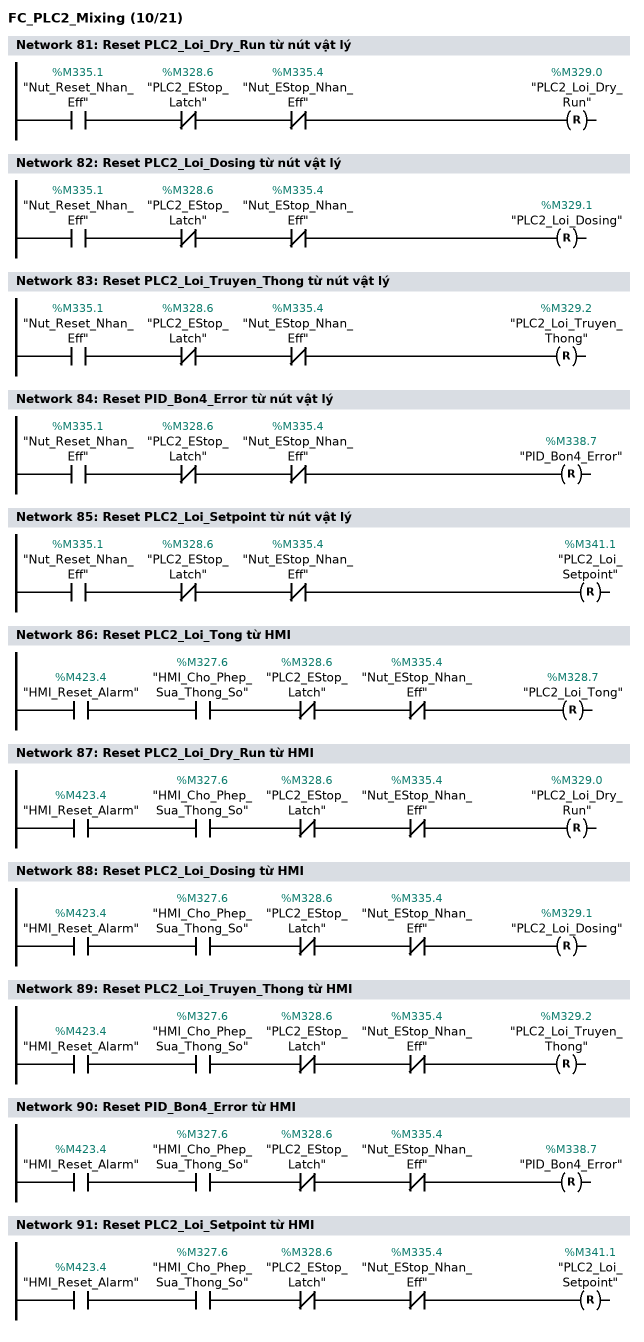
   RUNG wire#powerrail
      Contact( "Nut_Reset_Nhan_Eff" )
      I_Contact( "PLC2_EStop_Latch" )
      I_Contact( "Nut_EStop_Nhan_Eff" )
      R_Coil( "PLC2_Loi_Dry_Run" )
   END_RUNG
   // the same network as SCL:
   IF "Nut_Reset_Nhan_Eff" AND NOT "PLC2_EStop_Latch" AND NOT "Nut_EStop_Nhan_Eff" THEN
       "PLC2_Loi_Dry_Run" := FALSE;
   END_IF;
END_REGION

REGION Network 82: Reset PLC2_Loi_Dosing từ nút vật lý
   RUNG wire#powerrail
      Contact( "Nut_Reset_Nhan_Eff" )
      I_Contact( "PLC2_EStop_Latch" )
      I_Contact( "Nut_EStop_Nhan_Eff" )
      R_Coil( "PLC2_Loi_Dosing" )
   END_RUNG
   // the same network as SCL:
   IF "Nut_Reset_Nhan_Eff" AND NOT "PLC2_EStop_Latch" AND NOT "Nut_EStop_Nhan_Eff" THEN
       "PLC2_Loi_Dosing" := FALSE;
   END_IF;
END_REGION

REGION Network 83: Reset PLC2_Loi_Truyen_Thong từ nút vật lý
   RUNG wire#powerrail
      Contact( "Nut_Reset_Nhan_Eff" )
      I_Contact( "PLC2_EStop_Latch" )
      I_Contact( "Nut_EStop_Nhan_Eff" )
      R_Coil( "PLC2_Loi_Truyen_Thong" )
   END_RUNG
   // the same network as SCL:
   IF "Nut_Reset_Nhan_Eff" AND NOT "PLC2_EStop_Latch" AND NOT "Nut_EStop_Nhan_Eff" THEN
       "PLC2_Loi_Truyen_Thong" := FALSE;
   END_IF;
END_REGION

REGION Network 84: Reset PID_Bon4_Error từ nút vật lý
   RUNG wire#powerrail
      Contact( "Nut_Reset_Nhan_Eff" )
      I_Contact( "PLC2_EStop_Latch" )
      I_Contact( "Nut_EStop_Nhan_Eff" )
      R_Coil( "PID_Bon4_Error" )
   END_RUNG
   // the same network as SCL:
   IF "Nut_Reset_Nhan_Eff" AND NOT "PLC2_EStop_Latch" AND NOT "Nut_EStop_Nhan_Eff" THEN
       "PID_Bon4_Error" := FALSE;
   END_IF;
END_REGION

REGION Network 85: Reset PLC2_Loi_Setpoint từ nút vật lý
   RUNG wire#powerrail
      Contact( "Nut_Reset_Nhan_Eff" )
      I_Contact( "PLC2_EStop_Latch" )
      I_Contact( "Nut_EStop_Nhan_Eff" )
      R_Coil( "PLC2_Loi_Setpoint" )
   END_RUNG
   // the same network as SCL:
   IF "Nut_Reset_Nhan_Eff" AND NOT "PLC2_EStop_Latch" AND NOT "Nut_EStop_Nhan_Eff" THEN
       "PLC2_Loi_Setpoint" := FALSE;
   END_IF;
END_REGION

REGION Network 86: Reset PLC2_Loi_Tong từ HMI
   RUNG wire#powerrail
      Contact( "HMI_Reset_Alarm" )
      Contact( "HMI_Cho_Phep_Sua_Thong_So" )
      I_Contact( "PLC2_EStop_Latch" )
      I_Contact( "Nut_EStop_Nhan_Eff" )
      R_Coil( "PLC2_Loi_Tong" )
   END_RUNG
   // the same network as SCL:
   IF "HMI_Reset_Alarm" AND "HMI_Cho_Phep_Sua_Thong_So" AND NOT "PLC2_EStop_Latch" AND NOT "Nut_EStop_Nhan_Eff" THEN
       "PLC2_Loi_Tong" := FALSE;
   END_IF;
END_REGION

REGION Network 87: Reset PLC2_Loi_Dry_Run từ HMI
   RUNG wire#powerrail
      Contact( "HMI_Reset_Alarm" )
      Contact( "HMI_Cho_Phep_Sua_Thong_So" )
      I_Contact( "PLC2_EStop_Latch" )
      I_Contact( "Nut_EStop_Nhan_Eff" )
      R_Coil( "PLC2_Loi_Dry_Run" )
   END_RUNG
   // the same network as SCL:
   IF "HMI_Reset_Alarm" AND "HMI_Cho_Phep_Sua_Thong_So" AND NOT "PLC2_EStop_Latch" AND NOT "Nut_EStop_Nhan_Eff" THEN
       "PLC2_Loi_Dry_Run" := FALSE;
   END_IF;
END_REGION

REGION Network 88: Reset PLC2_Loi_Dosing từ HMI
   RUNG wire#powerrail
      Contact( "HMI_Reset_Alarm" )
      Contact( "HMI_Cho_Phep_Sua_Thong_So" )
      I_Contact( "PLC2_EStop_Latch" )
      I_Contact( "Nut_EStop_Nhan_Eff" )
      R_Coil( "PLC2_Loi_Dosing" )
   END_RUNG
   // the same network as SCL:
   IF "HMI_Reset_Alarm" AND "HMI_Cho_Phep_Sua_Thong_So" AND NOT "PLC2_EStop_Latch" AND NOT "Nut_EStop_Nhan_Eff" THEN
       "PLC2_Loi_Dosing" := FALSE;
   END_IF;
END_REGION

REGION Network 89: Reset PLC2_Loi_Truyen_Thong từ HMI
   RUNG wire#powerrail
      Contact( "HMI_Reset_Alarm" )
      Contact( "HMI_Cho_Phep_Sua_Thong_So" )
      I_Contact( "PLC2_EStop_Latch" )
      I_Contact( "Nut_EStop_Nhan_Eff" )
      R_Coil( "PLC2_Loi_Truyen_Thong" )
   END_RUNG
   // the same network as SCL:
   IF "HMI_Reset_Alarm" AND "HMI_Cho_Phep_Sua_Thong_So" AND NOT "PLC2_EStop_Latch" AND NOT "Nut_EStop_Nhan_Eff" THEN
       "PLC2_Loi_Truyen_Thong" := FALSE;
   END_IF;
END_REGION

REGION Network 90: Reset PID_Bon4_Error từ HMI
   RUNG wire#powerrail
      Contact( "HMI_Reset_Alarm" )
      Contact( "HMI_Cho_Phep_Sua_Thong_So" )
      I_Contact( "PLC2_EStop_Latch" )
      I_Contact( "Nut_EStop_Nhan_Eff" )
      R_Coil( "PID_Bon4_Error" )
   END_RUNG
   // the same network as SCL:
   IF "HMI_Reset_Alarm" AND "HMI_Cho_Phep_Sua_Thong_So" AND NOT "PLC2_EStop_Latch" AND NOT "Nut_EStop_Nhan_Eff" THEN
       "PID_Bon4_Error" := FALSE;
   END_IF;
END_REGION

REGION Network 91: Reset PLC2_Loi_Setpoint từ HMI
   RUNG wire#powerrail
      Contact( "HMI_Reset_Alarm" )
      Contact( "HMI_Cho_Phep_Sua_Thong_So" )
      I_Contact( "PLC2_EStop_Latch" )
      I_Contact( "Nut_EStop_Nhan_Eff" )
      R_Coil( "PLC2_Loi_Setpoint" )
   END_RUNG
   // the same network as SCL:
   IF "HMI_Reset_Alarm" AND "HMI_Cho_Phep_Sua_Thong_So" AND NOT "PLC2_EStop_Latch" AND NOT "Nut_EStop_Nhan_Eff" THEN
       "PLC2_Loi_Setpoint" := FALSE;
   END_IF;
END_REGION

REGION Network 92: Lỗi PLC2 - Dừng State về 0
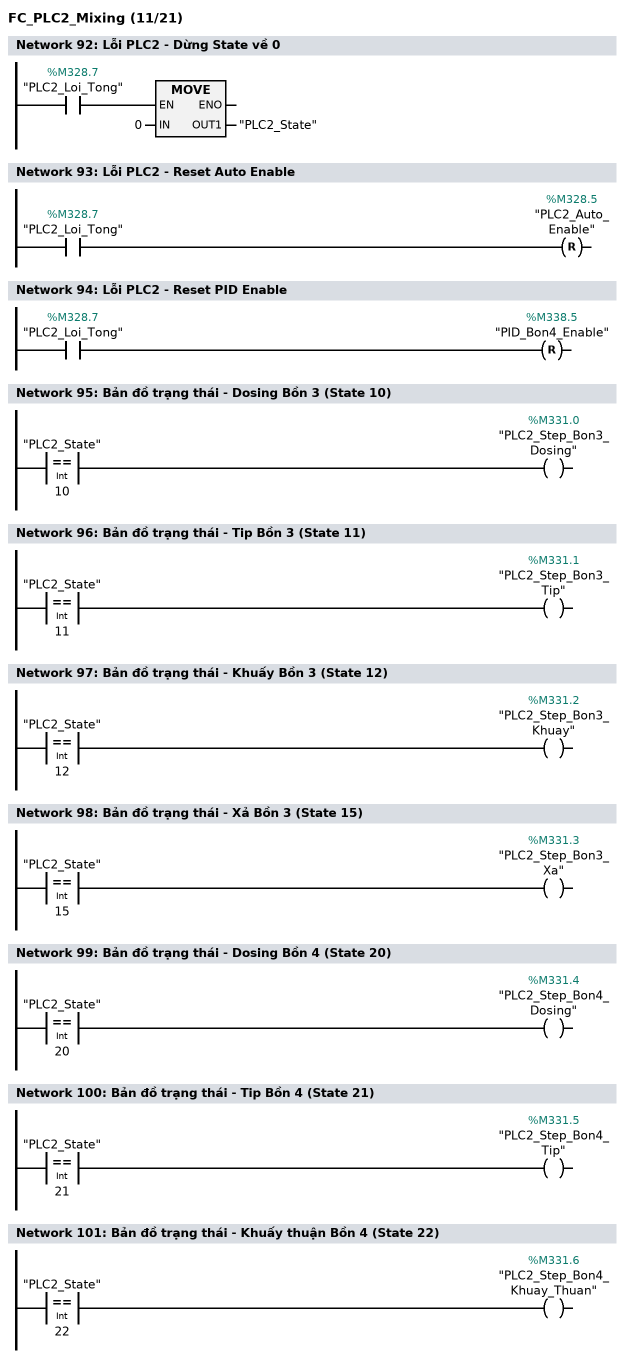
   RUNG wire#powerrail
      Contact( "PLC2_Loi_Tong" )
      { S7_GenerateENO := "TRUE" } Move(in := 0, out1 => "PLC2_State")
   END_RUNG
   // the same network as SCL:
   IF "PLC2_Loi_Tong" THEN "PLC2_State" := 0; END_IF;
END_REGION

REGION Network 93: Lỗi PLC2 - Reset Auto Enable
   RUNG wire#powerrail
      Contact( "PLC2_Loi_Tong" )
      R_Coil( "PLC2_Auto_Enable" )
   END_RUNG
   // the same network as SCL:
   IF "PLC2_Loi_Tong" THEN "PLC2_Auto_Enable" := FALSE; END_IF;
END_REGION

REGION Network 94: Lỗi PLC2 - Reset PID Enable
   RUNG wire#powerrail
      Contact( "PLC2_Loi_Tong" )
      R_Coil( "PID_Bon4_Enable" )
   END_RUNG
   // the same network as SCL:
   IF "PLC2_Loi_Tong" THEN "PID_Bon4_Enable" := FALSE; END_IF;
END_REGION

REGION Network 95: Bản đồ trạng thái - Dosing Bồn 3 (State 10)
   RUNG wire#powerrail
      { S7_Templates := "SrcType := Int" } EQ_Contact(in1 := "PLC2_State", in2 := 10)
      Coil( "PLC2_Step_Bon3_Dosing" )
   END_RUNG
   // the same network as SCL:
   "PLC2_Step_Bon3_Dosing" := "PLC2_State" = 10;
END_REGION

REGION Network 96: Bản đồ trạng thái - Tip Bồn 3 (State 11)
   RUNG wire#powerrail
      { S7_Templates := "SrcType := Int" } EQ_Contact(in1 := "PLC2_State", in2 := 11)
      Coil( "PLC2_Step_Bon3_Tip" )
   END_RUNG
   // the same network as SCL:
   "PLC2_Step_Bon3_Tip" := "PLC2_State" = 11;
END_REGION

REGION Network 97: Bản đồ trạng thái - Khuấy Bồn 3 (State 12)
   RUNG wire#powerrail
      { S7_Templates := "SrcType := Int" } EQ_Contact(in1 := "PLC2_State", in2 := 12)
      Coil( "PLC2_Step_Bon3_Khuay" )
   END_RUNG
   // the same network as SCL:
   "PLC2_Step_Bon3_Khuay" := "PLC2_State" = 12;
END_REGION

REGION Network 98: Bản đồ trạng thái - Xả Bồn 3 (State 15)
   RUNG wire#powerrail
      { S7_Templates := "SrcType := Int" } EQ_Contact(in1 := "PLC2_State", in2 := 15)
      Coil( "PLC2_Step_Bon3_Xa" )
   END_RUNG
   // the same network as SCL:
   "PLC2_Step_Bon3_Xa" := "PLC2_State" = 15;
END_REGION

REGION Network 99: Bản đồ trạng thái - Dosing Bồn 4 (State 20)
   RUNG wire#powerrail
      { S7_Templates := "SrcType := Int" } EQ_Contact(in1 := "PLC2_State", in2 := 20)
      Coil( "PLC2_Step_Bon4_Dosing" )
   END_RUNG
   // the same network as SCL:
   "PLC2_Step_Bon4_Dosing" := "PLC2_State" = 20;
END_REGION

REGION Network 100: Bản đồ trạng thái - Tip Bồn 4 (State 21)
   RUNG wire#powerrail
      { S7_Templates := "SrcType := Int" } EQ_Contact(in1 := "PLC2_State", in2 := 21)
      Coil( "PLC2_Step_Bon4_Tip" )
   END_RUNG
   // the same network as SCL:
   "PLC2_Step_Bon4_Tip" := "PLC2_State" = 21;
END_REGION

REGION Network 101: Bản đồ trạng thái - Khuấy thuận Bồn 4 (State 22)
   RUNG wire#powerrail
      { S7_Templates := "SrcType := Int" } EQ_Contact(in1 := "PLC2_State", in2 := 22)
      Coil( "PLC2_Step_Bon4_Khuay_Thuan" )
   END_RUNG
   // the same network as SCL:
   "PLC2_Step_Bon4_Khuay_Thuan" := "PLC2_State" = 22;
END_REGION

REGION Network 102: Bản đồ trạng thái - Khuấy nghịch Bồn 4 (State 23)
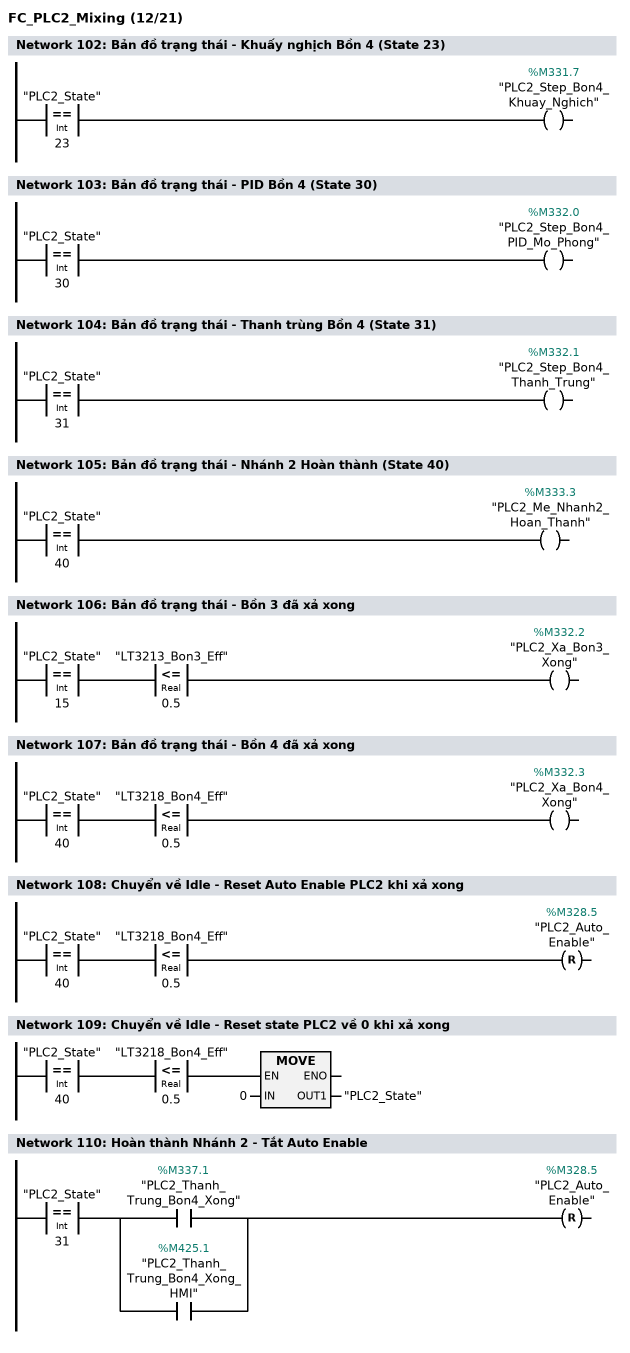
   RUNG wire#powerrail
      { S7_Templates := "SrcType := Int" } EQ_Contact(in1 := "PLC2_State", in2 := 23)
      Coil( "PLC2_Step_Bon4_Khuay_Nghich" )
   END_RUNG
   // the same network as SCL:
   "PLC2_Step_Bon4_Khuay_Nghich" := "PLC2_State" = 23;
END_REGION

REGION Network 103: Bản đồ trạng thái - PID Bồn 4 (State 30)
   RUNG wire#powerrail
      { S7_Templates := "SrcType := Int" } EQ_Contact(in1 := "PLC2_State", in2 := 30)
      Coil( "PLC2_Step_Bon4_PID_Mo_Phong" )
   END_RUNG
   // the same network as SCL:
   "PLC2_Step_Bon4_PID_Mo_Phong" := "PLC2_State" = 30;
END_REGION

REGION Network 104: Bản đồ trạng thái - Thanh trùng Bồn 4 (State 31)
   RUNG wire#powerrail
      { S7_Templates := "SrcType := Int" } EQ_Contact(in1 := "PLC2_State", in2 := 31)
      Coil( "PLC2_Step_Bon4_Thanh_Trung" )
   END_RUNG
   // the same network as SCL:
   "PLC2_Step_Bon4_Thanh_Trung" := "PLC2_State" = 31;
END_REGION

REGION Network 105: Bản đồ trạng thái - Nhánh 2 Hoàn thành (State 40)
   RUNG wire#powerrail
      { S7_Templates := "SrcType := Int" } EQ_Contact(in1 := "PLC2_State", in2 := 40)
      Coil( "PLC2_Me_Nhanh2_Hoan_Thanh" )
   END_RUNG
   // the same network as SCL:
   "PLC2_Me_Nhanh2_Hoan_Thanh" := "PLC2_State" = 40;
END_REGION

REGION Network 106: Bản đồ trạng thái - Bồn 3 đã xả xong
   RUNG wire#powerrail
      { S7_Templates := "SrcType := Int" } EQ_Contact(in1 := "PLC2_State", in2 := 15)
      { S7_Templates := "SrcType := Real" } LE_Contact(in1 := "LT3213_Bon3_Eff", in2 := 0.5)
      Coil( "PLC2_Xa_Bon3_Xong" )
   END_RUNG
   // the same network as SCL:
   "PLC2_Xa_Bon3_Xong" := ("PLC2_State" = 15) AND ("LT3213_Bon3_Eff" <= 0.5);
END_REGION

REGION Network 107: Bản đồ trạng thái - Bồn 4 đã xả xong
   RUNG wire#powerrail
      { S7_Templates := "SrcType := Int" } EQ_Contact(in1 := "PLC2_State", in2 := 40)
      { S7_Templates := "SrcType := Real" } LE_Contact(in1 := "LT3218_Bon4_Eff", in2 := 0.5)
      Coil( "PLC2_Xa_Bon4_Xong" )
   END_RUNG
   // the same network as SCL:
   "PLC2_Xa_Bon4_Xong" := ("PLC2_State" = 40) AND ("LT3218_Bon4_Eff" <= 0.5);
END_REGION

REGION Network 108: Chuyển về Idle - Reset Auto Enable PLC2 khi xả xong
   RUNG wire#powerrail
      { S7_Templates := "SrcType := Int" } EQ_Contact(in1 := "PLC2_State", in2 := 40)
      { S7_Templates := "SrcType := Real" } LE_Contact(in1 := "LT3218_Bon4_Eff", in2 := 0.5)
      R_Coil( "PLC2_Auto_Enable" )
   END_RUNG
   // the same network as SCL:
   IF ("PLC2_State" = 40) AND ("LT3218_Bon4_Eff" <= 0.5) THEN "PLC2_Auto_Enable" := FALSE; END_IF;
END_REGION

REGION Network 109: Chuyển về Idle - Reset state PLC2 về 0 khi xả xong
   RUNG wire#powerrail
      { S7_Templates := "SrcType := Int" } EQ_Contact(in1 := "PLC2_State", in2 := 40)
      { S7_Templates := "SrcType := Real" } LE_Contact(in1 := "LT3218_Bon4_Eff", in2 := 0.5)
      { S7_GenerateENO := "TRUE" } Move(in := 0, out1 => "PLC2_State")
   END_RUNG
   // the same network as SCL:
   IF ("PLC2_State" = 40) AND ("LT3218_Bon4_Eff" <= 0.5) THEN "PLC2_State" := 0; END_IF;
END_REGION

REGION Network 110: Hoàn thành Nhánh 2 - Tắt Auto Enable
   RUNG wire#powerrail
      { S7_Templates := "SrcType := Int" } EQ_Contact(in1 := "PLC2_State", in2 := 31)
      wire#w1
      Contact( "PLC2_Thanh_Trung_Bon4_Xong" )
      wire#w2
      R_Coil( "PLC2_Auto_Enable" )
   END_RUNG
   RUNG wire#w1
      Contact( "PLC2_Thanh_Trung_Bon4_Xong_HMI" )
   END_RUNG wire#w2
   // the same network as SCL:
   IF ("PLC2_State" = 31) AND ("PLC2_Thanh_Trung_Bon4_Xong" OR "PLC2_Thanh_Trung_Bon4_Xong_HMI") THEN
       "PLC2_Auto_Enable" := FALSE;
   END_IF;
END_REGION

REGION Network 111: Hoàn thành Nhánh 2 - Tắt PID Enable
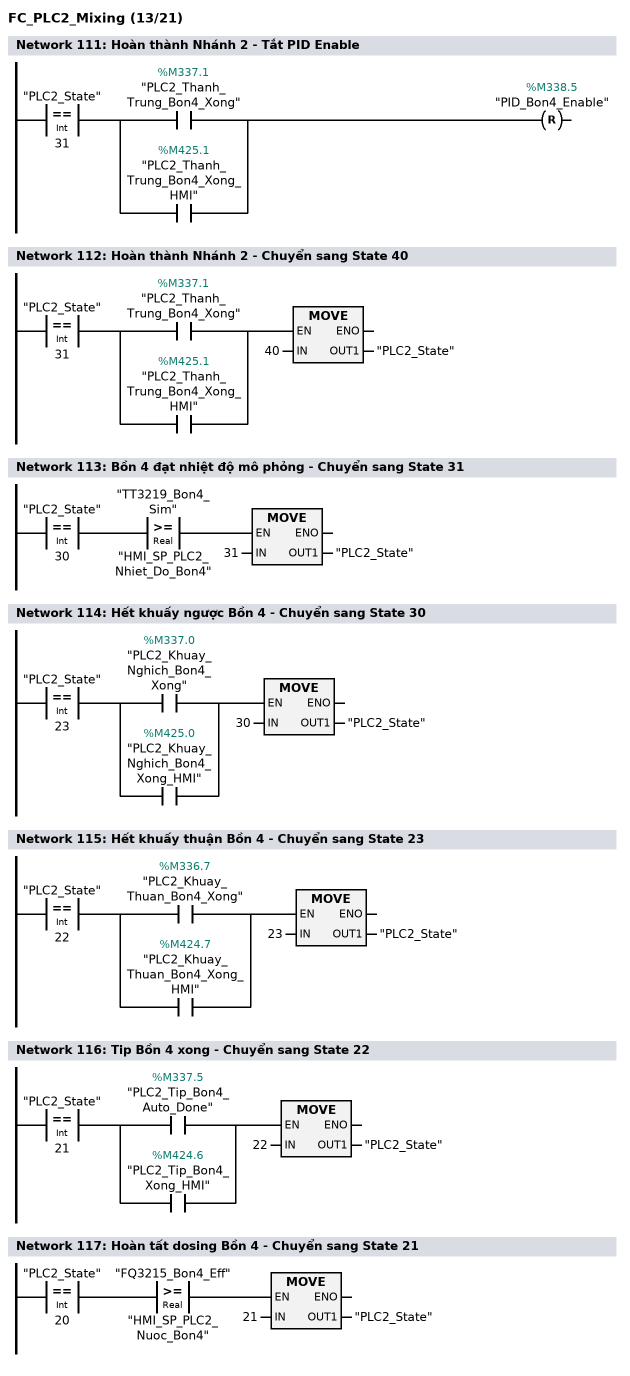
   RUNG wire#powerrail
      { S7_Templates := "SrcType := Int" } EQ_Contact(in1 := "PLC2_State", in2 := 31)
      wire#w1
      Contact( "PLC2_Thanh_Trung_Bon4_Xong" )
      wire#w2
      R_Coil( "PID_Bon4_Enable" )
   END_RUNG
   RUNG wire#w1
      Contact( "PLC2_Thanh_Trung_Bon4_Xong_HMI" )
   END_RUNG wire#w2
   // the same network as SCL:
   IF ("PLC2_State" = 31) AND ("PLC2_Thanh_Trung_Bon4_Xong" OR "PLC2_Thanh_Trung_Bon4_Xong_HMI") THEN
       "PID_Bon4_Enable" := FALSE;
   END_IF;
END_REGION

REGION Network 112: Hoàn thành Nhánh 2 - Chuyển sang State 40
   RUNG wire#powerrail
      { S7_Templates := "SrcType := Int" } EQ_Contact(in1 := "PLC2_State", in2 := 31)
      wire#w1
      Contact( "PLC2_Thanh_Trung_Bon4_Xong" )
      wire#w2
      { S7_GenerateENO := "TRUE" } Move(in := 40, out1 => "PLC2_State")
   END_RUNG
   RUNG wire#w1
      Contact( "PLC2_Thanh_Trung_Bon4_Xong_HMI" )
   END_RUNG wire#w2
   // the same network as SCL:
   IF ("PLC2_State" = 31) AND ("PLC2_Thanh_Trung_Bon4_Xong" OR "PLC2_Thanh_Trung_Bon4_Xong_HMI") THEN
       "PLC2_State" := 40;
   END_IF;
END_REGION

REGION Network 113: Bồn 4 đạt nhiệt độ mô phỏng - Chuyển sang State 31
   RUNG wire#powerrail
      { S7_Templates := "SrcType := Int" } EQ_Contact(in1 := "PLC2_State", in2 := 30)
      { S7_Templates := "SrcType := Real" } GE_Contact(in1 := "TT3219_Bon4_Sim", in2 := "HMI_SP_PLC2_Nhiet_Do_Bon4")
      { S7_GenerateENO := "TRUE" } Move(in := 31, out1 => "PLC2_State")
   END_RUNG
   // the same network as SCL:
   IF ("PLC2_State" = 30) AND ("TT3219_Bon4_Sim" >= "HMI_SP_PLC2_Nhiet_Do_Bon4") THEN
       "PLC2_State" := 31;
   END_IF;
END_REGION

REGION Network 114: Hết khuấy ngược Bồn 4 - Chuyển sang State 30
   RUNG wire#powerrail
      { S7_Templates := "SrcType := Int" } EQ_Contact(in1 := "PLC2_State", in2 := 23)
      wire#w1
      Contact( "PLC2_Khuay_Nghich_Bon4_Xong" )
      wire#w2
      { S7_GenerateENO := "TRUE" } Move(in := 30, out1 => "PLC2_State")
   END_RUNG
   RUNG wire#w1
      Contact( "PLC2_Khuay_Nghich_Bon4_Xong_HMI" )
   END_RUNG wire#w2
   // the same network as SCL:
   IF ("PLC2_State" = 23) AND ("PLC2_Khuay_Nghich_Bon4_Xong" OR "PLC2_Khuay_Nghich_Bon4_Xong_HMI") THEN
       "PLC2_State" := 30;
   END_IF;
END_REGION

REGION Network 115: Hết khuấy thuận Bồn 4 - Chuyển sang State 23
   RUNG wire#powerrail
      { S7_Templates := "SrcType := Int" } EQ_Contact(in1 := "PLC2_State", in2 := 22)
      wire#w1
      Contact( "PLC2_Khuay_Thuan_Bon4_Xong" )
      wire#w2
      { S7_GenerateENO := "TRUE" } Move(in := 23, out1 => "PLC2_State")
   END_RUNG
   RUNG wire#w1
      Contact( "PLC2_Khuay_Thuan_Bon4_Xong_HMI" )
   END_RUNG wire#w2
   // the same network as SCL:
   IF ("PLC2_State" = 22) AND ("PLC2_Khuay_Thuan_Bon4_Xong" OR "PLC2_Khuay_Thuan_Bon4_Xong_HMI") THEN
       "PLC2_State" := 23;
   END_IF;
END_REGION

REGION Network 116: Tip Bồn 4 xong - Chuyển sang State 22
   RUNG wire#powerrail
      { S7_Templates := "SrcType := Int" } EQ_Contact(in1 := "PLC2_State", in2 := 21)
      wire#w1
      Contact( "PLC2_Tip_Bon4_Auto_Done" )
      wire#w2
      { S7_GenerateENO := "TRUE" } Move(in := 22, out1 => "PLC2_State")
   END_RUNG
   RUNG wire#w1
      Contact( "PLC2_Tip_Bon4_Xong_HMI" )
   END_RUNG wire#w2
   // the same network as SCL:
   IF ("PLC2_State" = 21) AND ("PLC2_Tip_Bon4_Auto_Done" OR "PLC2_Tip_Bon4_Xong_HMI") THEN
       "PLC2_State" := 22;
   END_IF;
END_REGION

REGION Network 117: Hoàn tất dosing Bồn 4 - Chuyển sang State 21
   RUNG wire#powerrail
      { S7_Templates := "SrcType := Int" } EQ_Contact(in1 := "PLC2_State", in2 := 20)
      { S7_Templates := "SrcType := Real" } GE_Contact(in1 := "FQ3215_Bon4_Eff", in2 := "HMI_SP_PLC2_Nuoc_Bon4")
      { S7_GenerateENO := "TRUE" } Move(in := 21, out1 => "PLC2_State")
   END_RUNG
   // the same network as SCL:
   IF ("PLC2_State" = 20) AND ("FQ3215_Bon4_Eff" >= "HMI_SP_PLC2_Nuoc_Bon4") THEN "PLC2_State" := 21; END_IF;
END_REGION

REGION Network 118: Xả Bồn 3 xong - Chuyển sang State 20
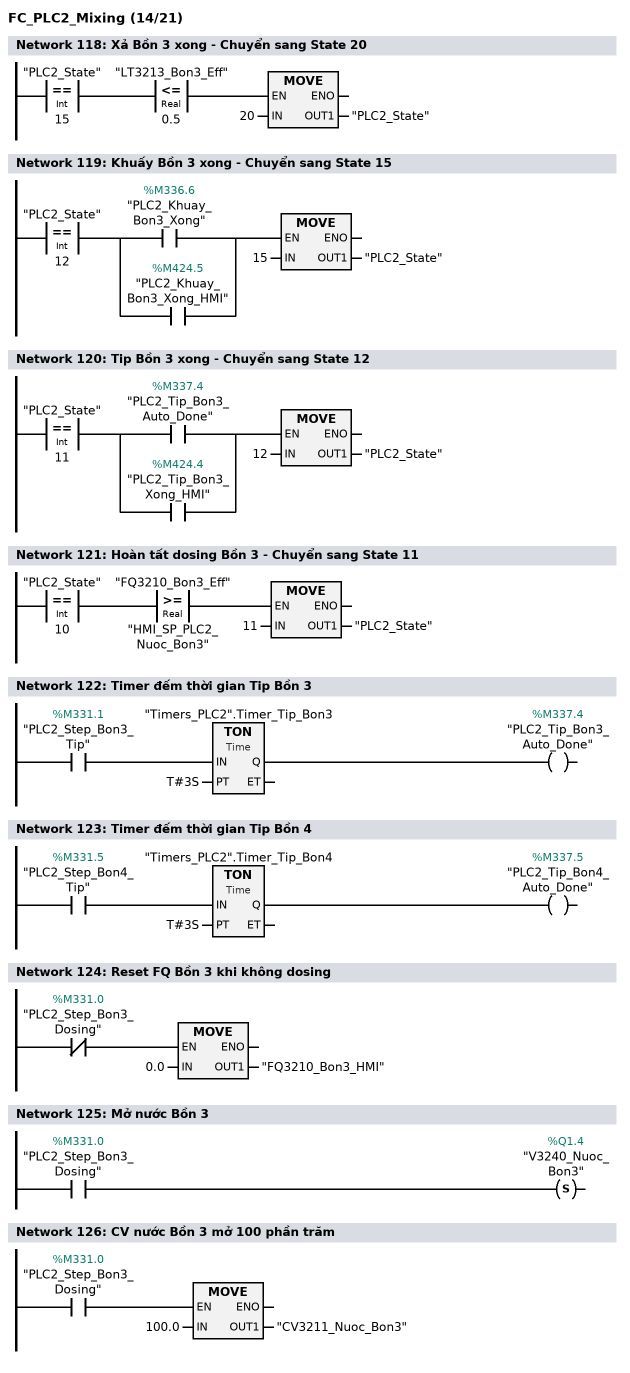
   RUNG wire#powerrail
      { S7_Templates := "SrcType := Int" } EQ_Contact(in1 := "PLC2_State", in2 := 15)
      { S7_Templates := "SrcType := Real" } LE_Contact(in1 := "LT3213_Bon3_Eff", in2 := 0.5)
      { S7_GenerateENO := "TRUE" } Move(in := 20, out1 => "PLC2_State")
   END_RUNG
   // the same network as SCL:
   IF ("PLC2_State" = 15) AND ("LT3213_Bon3_Eff" <= 0.5) THEN "PLC2_State" := 20; END_IF;
END_REGION

REGION Network 119: Khuấy Bồn 3 xong - Chuyển sang State 15
   RUNG wire#powerrail
      { S7_Templates := "SrcType := Int" } EQ_Contact(in1 := "PLC2_State", in2 := 12)
      wire#w1
      Contact( "PLC2_Khuay_Bon3_Xong" )
      wire#w2
      { S7_GenerateENO := "TRUE" } Move(in := 15, out1 => "PLC2_State")
   END_RUNG
   RUNG wire#w1
      Contact( "PLC2_Khuay_Bon3_Xong_HMI" )
   END_RUNG wire#w2
   // the same network as SCL:
   IF ("PLC2_State" = 12) AND ("PLC2_Khuay_Bon3_Xong" OR "PLC2_Khuay_Bon3_Xong_HMI") THEN
       "PLC2_State" := 15;
   END_IF;
END_REGION

REGION Network 120: Tip Bồn 3 xong - Chuyển sang State 12
   RUNG wire#powerrail
      { S7_Templates := "SrcType := Int" } EQ_Contact(in1 := "PLC2_State", in2 := 11)
      wire#w1
      Contact( "PLC2_Tip_Bon3_Auto_Done" )
      wire#w2
      { S7_GenerateENO := "TRUE" } Move(in := 12, out1 => "PLC2_State")
   END_RUNG
   RUNG wire#w1
      Contact( "PLC2_Tip_Bon3_Xong_HMI" )
   END_RUNG wire#w2
   // the same network as SCL:
   IF ("PLC2_State" = 11) AND ("PLC2_Tip_Bon3_Auto_Done" OR "PLC2_Tip_Bon3_Xong_HMI") THEN
       "PLC2_State" := 12;
   END_IF;
END_REGION

REGION Network 121: Hoàn tất dosing Bồn 3 - Chuyển sang State 11
   RUNG wire#powerrail
      { S7_Templates := "SrcType := Int" } EQ_Contact(in1 := "PLC2_State", in2 := 10)
      { S7_Templates := "SrcType := Real" } GE_Contact(in1 := "FQ3210_Bon3_Eff", in2 := "HMI_SP_PLC2_Nuoc_Bon3")
      { S7_GenerateENO := "TRUE" } Move(in := 11, out1 => "PLC2_State")
   END_RUNG
   // the same network as SCL:
   IF ("PLC2_State" = 10) AND ("FQ3210_Bon3_Eff" >= "HMI_SP_PLC2_Nuoc_Bon3") THEN "PLC2_State" := 11; END_IF;
END_REGION

REGION Network 122: Timer đếm thời gian Tip Bồn 3
   RUNG wire#powerrail
      Contact( "PLC2_Step_Bon3_Tip" )
      { S7_Templates := "time_type := Time" } "Timers_PLC2".Timer_Tip_Bon3.TON(pt := T#3S, et =>)
      Coil( "PLC2_Tip_Bon3_Auto_Done" )
   END_RUNG
   // the same network as SCL:
   "Timers_PLC2".Timer_Tip_Bon3.TON(IN := "PLC2_Step_Bon3_Tip", PT := T#3S);
   "PLC2_Tip_Bon3_Auto_Done" := "Timers_PLC2".Timer_Tip_Bon3.Q;
END_REGION

REGION Network 123: Timer đếm thời gian Tip Bồn 4
   RUNG wire#powerrail
      Contact( "PLC2_Step_Bon4_Tip" )
      { S7_Templates := "time_type := Time" } "Timers_PLC2".Timer_Tip_Bon4.TON(pt := T#3S, et =>)
      Coil( "PLC2_Tip_Bon4_Auto_Done" )
   END_RUNG
   // the same network as SCL:
   "Timers_PLC2".Timer_Tip_Bon4.TON(IN := "PLC2_Step_Bon4_Tip", PT := T#3S);
   "PLC2_Tip_Bon4_Auto_Done" := "Timers_PLC2".Timer_Tip_Bon4.Q;
END_REGION

REGION Network 124: Reset FQ Bồn 3 khi không dosing
   RUNG wire#powerrail
      I_Contact( "PLC2_Step_Bon3_Dosing" )
      { S7_GenerateENO := "TRUE" } Move(in := 0.0, out1 => "FQ3210_Bon3_HMI")
   END_RUNG
   // the same network as SCL:
   IF NOT "PLC2_Step_Bon3_Dosing" THEN "FQ3210_Bon3_HMI" := 0.0; END_IF;
END_REGION

REGION Network 125: Mở nước Bồn 3
   RUNG wire#powerrail
      Contact( "PLC2_Step_Bon3_Dosing" )
      S_Coil( "V3240_Nuoc_Bon3" )
   END_RUNG
   // the same network as SCL:
   IF "PLC2_Step_Bon3_Dosing" THEN "V3240_Nuoc_Bon3" := TRUE; END_IF;
END_REGION

REGION Network 126: CV nước Bồn 3 mở 100 phần trăm
   RUNG wire#powerrail
      Contact( "PLC2_Step_Bon3_Dosing" )
      { S7_GenerateENO := "TRUE" } Move(in := 100.0, out1 => "CV3211_Nuoc_Bon3")
   END_RUNG
   // the same network as SCL:
   IF "PLC2_Step_Bon3_Dosing" THEN "CV3211_Nuoc_Bon3" := 100.0; END_IF;
END_REGION

REGION Network 127: Đóng nước Bồn 3 sau dosing
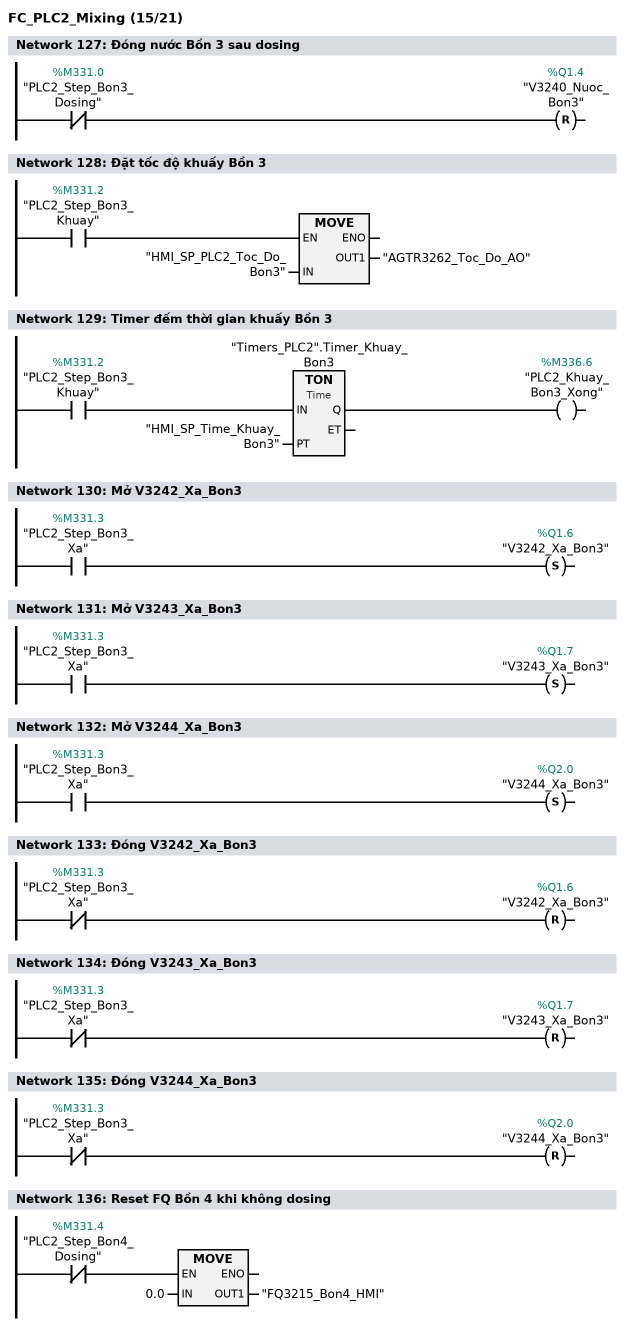
   RUNG wire#powerrail
      I_Contact( "PLC2_Step_Bon3_Dosing" )
      R_Coil( "V3240_Nuoc_Bon3" )
   END_RUNG
   // the same network as SCL:
   IF NOT "PLC2_Step_Bon3_Dosing" THEN "V3240_Nuoc_Bon3" := FALSE; END_IF;
END_REGION

REGION Network 128: Đặt tốc độ khuấy Bồn 3
   RUNG wire#powerrail
      Contact( "PLC2_Step_Bon3_Khuay" )
      { S7_GenerateENO := "TRUE" } Move(in := "HMI_SP_PLC2_Toc_Do_Bon3", out1 => "AGTR3262_Toc_Do_AO")
   END_RUNG
   // the same network as SCL:
   IF "PLC2_Step_Bon3_Khuay" THEN "AGTR3262_Toc_Do_AO" := "HMI_SP_PLC2_Toc_Do_Bon3"; END_IF;
END_REGION

REGION Network 129: Timer đếm thời gian khuấy Bồn 3
   RUNG wire#powerrail
      Contact( "PLC2_Step_Bon3_Khuay" )
      { S7_Templates := "time_type := Time" } "Timers_PLC2".Timer_Khuay_Bon3.TON(pt := "HMI_SP_Time_Khuay_Bon3", et =>)
      Coil( "PLC2_Khuay_Bon3_Xong" )
   END_RUNG
   // the same network as SCL:
   "Timers_PLC2".Timer_Khuay_Bon3.TON(IN := "PLC2_Step_Bon3_Khuay", PT := "HMI_SP_Time_Khuay_Bon3");
   "PLC2_Khuay_Bon3_Xong" := "Timers_PLC2".Timer_Khuay_Bon3.Q;
END_REGION

REGION Network 130: Mở V3242_Xa_Bon3
   RUNG wire#powerrail
      Contact( "PLC2_Step_Bon3_Xa" )
      S_Coil( "V3242_Xa_Bon3" )
   END_RUNG
   // the same network as SCL:
   IF "PLC2_Step_Bon3_Xa" THEN "V3242_Xa_Bon3" := TRUE; END_IF;
END_REGION

REGION Network 131: Mở V3243_Xa_Bon3
   RUNG wire#powerrail
      Contact( "PLC2_Step_Bon3_Xa" )
      S_Coil( "V3243_Xa_Bon3" )
   END_RUNG
   // the same network as SCL:
   IF "PLC2_Step_Bon3_Xa" THEN "V3243_Xa_Bon3" := TRUE; END_IF;
END_REGION

REGION Network 132: Mở V3244_Xa_Bon3
   RUNG wire#powerrail
      Contact( "PLC2_Step_Bon3_Xa" )
      S_Coil( "V3244_Xa_Bon3" )
   END_RUNG
   // the same network as SCL:
   IF "PLC2_Step_Bon3_Xa" THEN "V3244_Xa_Bon3" := TRUE; END_IF;
END_REGION

REGION Network 133: Đóng V3242_Xa_Bon3
   RUNG wire#powerrail
      I_Contact( "PLC2_Step_Bon3_Xa" )
      R_Coil( "V3242_Xa_Bon3" )
   END_RUNG
   // the same network as SCL:
   IF NOT "PLC2_Step_Bon3_Xa" THEN "V3242_Xa_Bon3" := FALSE; END_IF;
END_REGION

REGION Network 134: Đóng V3243_Xa_Bon3
   RUNG wire#powerrail
      I_Contact( "PLC2_Step_Bon3_Xa" )
      R_Coil( "V3243_Xa_Bon3" )
   END_RUNG
   // the same network as SCL:
   IF NOT "PLC2_Step_Bon3_Xa" THEN "V3243_Xa_Bon3" := FALSE; END_IF;
END_REGION

REGION Network 135: Đóng V3244_Xa_Bon3
   RUNG wire#powerrail
      I_Contact( "PLC2_Step_Bon3_Xa" )
      R_Coil( "V3244_Xa_Bon3" )
   END_RUNG
   // the same network as SCL:
   IF NOT "PLC2_Step_Bon3_Xa" THEN "V3244_Xa_Bon3" := FALSE; END_IF;
END_REGION

REGION Network 136: Reset FQ Bồn 4 khi không dosing
   RUNG wire#powerrail
      I_Contact( "PLC2_Step_Bon4_Dosing" )
      { S7_GenerateENO := "TRUE" } Move(in := 0.0, out1 => "FQ3215_Bon4_HMI")
   END_RUNG
   // the same network as SCL:
   IF NOT "PLC2_Step_Bon4_Dosing" THEN "FQ3215_Bon4_HMI" := 0.0; END_IF;
END_REGION

REGION Network 137: Mở nước Bồn 4
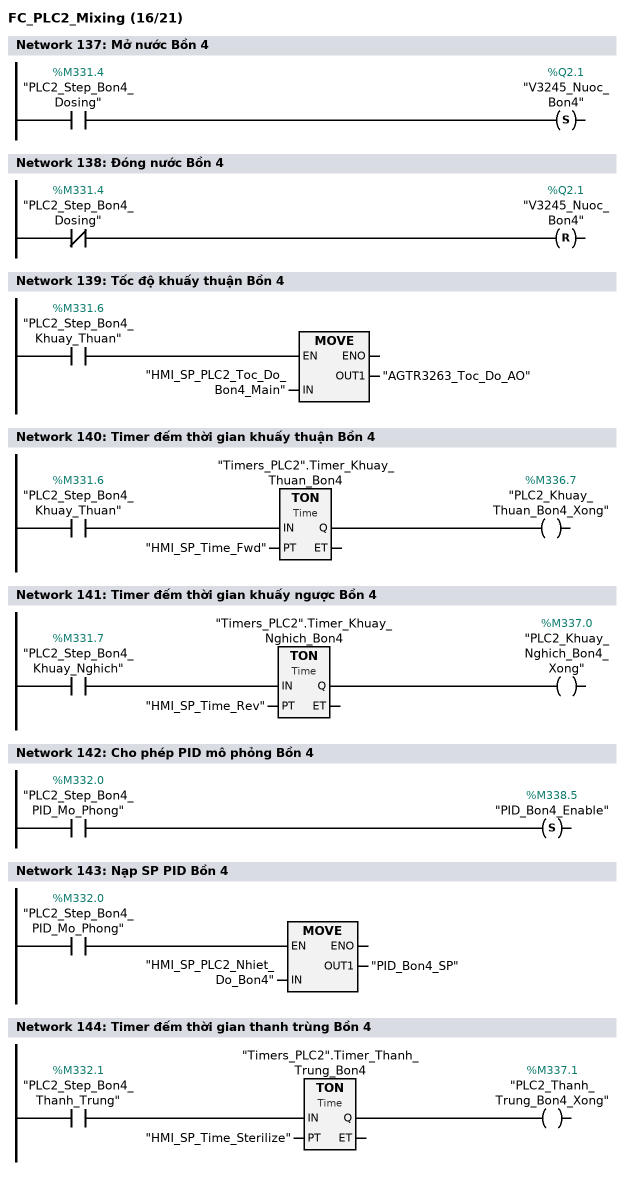
   RUNG wire#powerrail
      Contact( "PLC2_Step_Bon4_Dosing" )
      S_Coil( "V3245_Nuoc_Bon4" )
   END_RUNG
   // the same network as SCL:
   IF "PLC2_Step_Bon4_Dosing" THEN "V3245_Nuoc_Bon4" := TRUE; END_IF;
END_REGION

REGION Network 138: Đóng nước Bồn 4
   RUNG wire#powerrail
      I_Contact( "PLC2_Step_Bon4_Dosing" )
      R_Coil( "V3245_Nuoc_Bon4" )
   END_RUNG
   // the same network as SCL:
   IF NOT "PLC2_Step_Bon4_Dosing" THEN "V3245_Nuoc_Bon4" := FALSE; END_IF;
END_REGION

REGION Network 139: Tốc độ khuấy thuận Bồn 4
   RUNG wire#powerrail
      Contact( "PLC2_Step_Bon4_Khuay_Thuan" )
      { S7_GenerateENO := "TRUE" } Move(in := "HMI_SP_PLC2_Toc_Do_Bon4_Main", out1 => "AGTR3263_Toc_Do_AO")
   END_RUNG
   // the same network as SCL:
   IF "PLC2_Step_Bon4_Khuay_Thuan" THEN "AGTR3263_Toc_Do_AO" := "HMI_SP_PLC2_Toc_Do_Bon4_Main"; END_IF;
END_REGION

REGION Network 140: Timer đếm thời gian khuấy thuận Bồn 4
   RUNG wire#powerrail
      Contact( "PLC2_Step_Bon4_Khuay_Thuan" )
      { S7_Templates := "time_type := Time" } "Timers_PLC2".Timer_Khuay_Thuan_Bon4.TON(pt := "HMI_SP_Time_Fwd", et =>)
      Coil( "PLC2_Khuay_Thuan_Bon4_Xong" )
   END_RUNG
   // the same network as SCL:
   "Timers_PLC2".Timer_Khuay_Thuan_Bon4.TON(IN := "PLC2_Step_Bon4_Khuay_Thuan", PT := "HMI_SP_Time_Fwd");
   "PLC2_Khuay_Thuan_Bon4_Xong" := "Timers_PLC2".Timer_Khuay_Thuan_Bon4.Q;
END_REGION

REGION Network 141: Timer đếm thời gian khuấy ngược Bồn 4
   RUNG wire#powerrail
      Contact( "PLC2_Step_Bon4_Khuay_Nghich" )
      { S7_Templates := "time_type := Time" } "Timers_PLC2".Timer_Khuay_Nghich_Bon4.TON(pt := "HMI_SP_Time_Rev", et =>)
      Coil( "PLC2_Khuay_Nghich_Bon4_Xong" )
   END_RUNG
   // the same network as SCL:
   "Timers_PLC2".Timer_Khuay_Nghich_Bon4.TON(IN := "PLC2_Step_Bon4_Khuay_Nghich", PT := "HMI_SP_Time_Rev");
   "PLC2_Khuay_Nghich_Bon4_Xong" := "Timers_PLC2".Timer_Khuay_Nghich_Bon4.Q;
END_REGION

REGION Network 142: Cho phép PID mô phỏng Bồn 4
   RUNG wire#powerrail
      Contact( "PLC2_Step_Bon4_PID_Mo_Phong" )
      S_Coil( "PID_Bon4_Enable" )
   END_RUNG
   // the same network as SCL:
   IF "PLC2_Step_Bon4_PID_Mo_Phong" THEN "PID_Bon4_Enable" := TRUE; END_IF;
END_REGION

REGION Network 143: Nạp SP PID Bồn 4
   RUNG wire#powerrail
      Contact( "PLC2_Step_Bon4_PID_Mo_Phong" )
      { S7_GenerateENO := "TRUE" } Move(in := "HMI_SP_PLC2_Nhiet_Do_Bon4", out1 => "PID_Bon4_SP")
   END_RUNG
   // the same network as SCL:
   IF "PLC2_Step_Bon4_PID_Mo_Phong" THEN "PID_Bon4_SP" := "HMI_SP_PLC2_Nhiet_Do_Bon4"; END_IF;
END_REGION

REGION Network 144: Timer đếm thời gian thanh trùng Bồn 4
   RUNG wire#powerrail
      Contact( "PLC2_Step_Bon4_Thanh_Trung" )
      { S7_Templates := "time_type := Time" } "Timers_PLC2".Timer_Thanh_Trung_Bon4.TON(pt := "HMI_SP_Time_Sterilize", et =>)
      Coil( "PLC2_Thanh_Trung_Bon4_Xong" )
   END_RUNG
   // the same network as SCL:
   "Timers_PLC2".Timer_Thanh_Trung_Bon4.TON(IN := "PLC2_Step_Bon4_Thanh_Trung", PT := "HMI_SP_Time_Sterilize");
   "PLC2_Thanh_Trung_Bon4_Xong" := "Timers_PLC2".Timer_Thanh_Trung_Bon4.Q;
END_REGION

REGION Network 145: Bơm chuyển Nhánh 2 chạy khi có lệnh
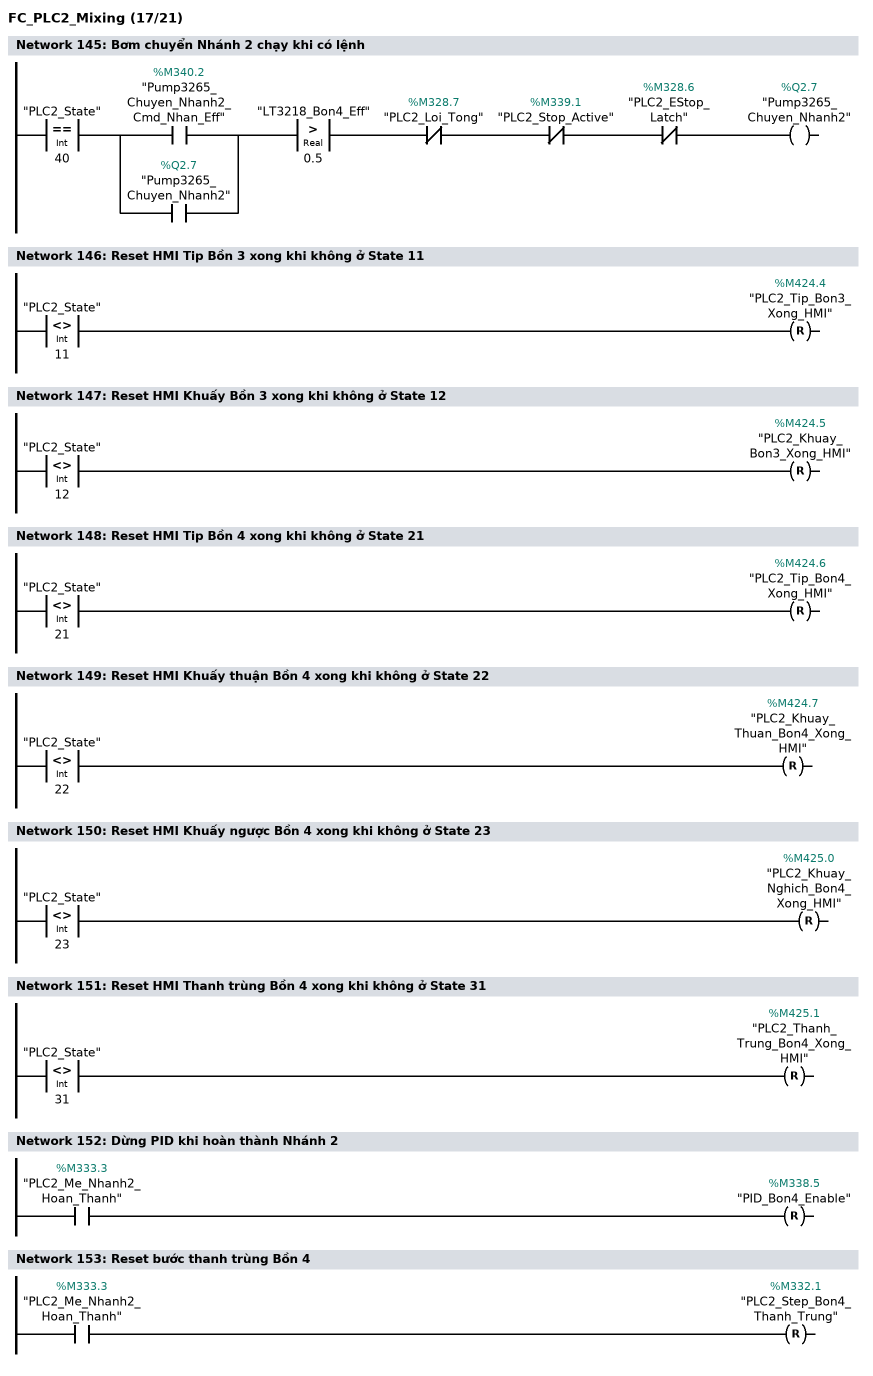
   RUNG wire#powerrail
      { S7_Templates := "SrcType := Int" } EQ_Contact(in1 := "PLC2_State", in2 := 40)
      wire#w1
      Contact( "Pump3265_Chuyen_Nhanh2_Cmd_Nhan_Eff" )
      wire#w2
      { S7_Templates := "SrcType := Real" } GT_Contact(in1 := "LT3218_Bon4_Eff", in2 := 0.5)
      I_Contact( "PLC2_Loi_Tong" )
      I_Contact( "PLC2_Stop_Active" )
      I_Contact( "PLC2_EStop_Latch" )
      Coil( "Pump3265_Chuyen_Nhanh2" )
   END_RUNG
   RUNG wire#w1
      Contact( "Pump3265_Chuyen_Nhanh2" )
   END_RUNG wire#w2
   // the same network as SCL:
   "Pump3265_Chuyen_Nhanh2" := ("PLC2_State" = 40) AND ("Pump3265_Chuyen_Nhanh2_Cmd_Nhan_Eff" OR "Pump3265_Chuyen_Nhanh2") AND ("LT3218_Bon4_Eff" > 0.5) AND NOT "PLC2_Loi_Tong" AND NOT "PLC2_Stop_Active" AND NOT "PLC2_EStop_Latch";
END_REGION

REGION Network 146: Reset HMI Tip Bồn 3 xong khi không ở State 11
   RUNG wire#powerrail
      { S7_Templates := "SrcType := Int" } NE_Contact(in1 := "PLC2_State", in2 := 11)
      R_Coil( "PLC2_Tip_Bon3_Xong_HMI" )
   END_RUNG
   // the same network as SCL:
   IF "PLC2_State" <> 11 THEN "PLC2_Tip_Bon3_Xong_HMI" := FALSE; END_IF;
END_REGION

REGION Network 147: Reset HMI Khuấy Bồn 3 xong khi không ở State 12
   RUNG wire#powerrail
      { S7_Templates := "SrcType := Int" } NE_Contact(in1 := "PLC2_State", in2 := 12)
      R_Coil( "PLC2_Khuay_Bon3_Xong_HMI" )
   END_RUNG
   // the same network as SCL:
   IF "PLC2_State" <> 12 THEN "PLC2_Khuay_Bon3_Xong_HMI" := FALSE; END_IF;
END_REGION

REGION Network 148: Reset HMI Tip Bồn 4 xong khi không ở State 21
   RUNG wire#powerrail
      { S7_Templates := "SrcType := Int" } NE_Contact(in1 := "PLC2_State", in2 := 21)
      R_Coil( "PLC2_Tip_Bon4_Xong_HMI" )
   END_RUNG
   // the same network as SCL:
   IF "PLC2_State" <> 21 THEN "PLC2_Tip_Bon4_Xong_HMI" := FALSE; END_IF;
END_REGION

REGION Network 149: Reset HMI Khuấy thuận Bồn 4 xong khi không ở State 22
   RUNG wire#powerrail
      { S7_Templates := "SrcType := Int" } NE_Contact(in1 := "PLC2_State", in2 := 22)
      R_Coil( "PLC2_Khuay_Thuan_Bon4_Xong_HMI" )
   END_RUNG
   // the same network as SCL:
   IF "PLC2_State" <> 22 THEN "PLC2_Khuay_Thuan_Bon4_Xong_HMI" := FALSE; END_IF;
END_REGION

REGION Network 150: Reset HMI Khuấy ngược Bồn 4 xong khi không ở State 23
   RUNG wire#powerrail
      { S7_Templates := "SrcType := Int" } NE_Contact(in1 := "PLC2_State", in2 := 23)
      R_Coil( "PLC2_Khuay_Nghich_Bon4_Xong_HMI" )
   END_RUNG
   // the same network as SCL:
   IF "PLC2_State" <> 23 THEN "PLC2_Khuay_Nghich_Bon4_Xong_HMI" := FALSE; END_IF;
END_REGION

REGION Network 151: Reset HMI Thanh trùng Bồn 4 xong khi không ở State 31
   RUNG wire#powerrail
      { S7_Templates := "SrcType := Int" } NE_Contact(in1 := "PLC2_State", in2 := 31)
      R_Coil( "PLC2_Thanh_Trung_Bon4_Xong_HMI" )
   END_RUNG
   // the same network as SCL:
   IF "PLC2_State" <> 31 THEN "PLC2_Thanh_Trung_Bon4_Xong_HMI" := FALSE; END_IF;
END_REGION

REGION Network 152: Dừng PID khi hoàn thành Nhánh 2
   RUNG wire#powerrail
      Contact( "PLC2_Me_Nhanh2_Hoan_Thanh" )
      R_Coil( "PID_Bon4_Enable" )
   END_RUNG
   // the same network as SCL:
   IF "PLC2_Me_Nhanh2_Hoan_Thanh" THEN "PID_Bon4_Enable" := FALSE; END_IF;
END_REGION

REGION Network 153: Reset bước thanh trùng Bồn 4
   RUNG wire#powerrail
      Contact( "PLC2_Me_Nhanh2_Hoan_Thanh" )
      R_Coil( "PLC2_Step_Bon4_Thanh_Trung" )
   END_RUNG
   // the same network as SCL:
   IF "PLC2_Me_Nhanh2_Hoan_Thanh" THEN "PLC2_Step_Bon4_Thanh_Trung" := FALSE; END_IF;
END_REGION

REGION Network 154: Chạy cánh khuấy Bồn 3 (Coil thường)
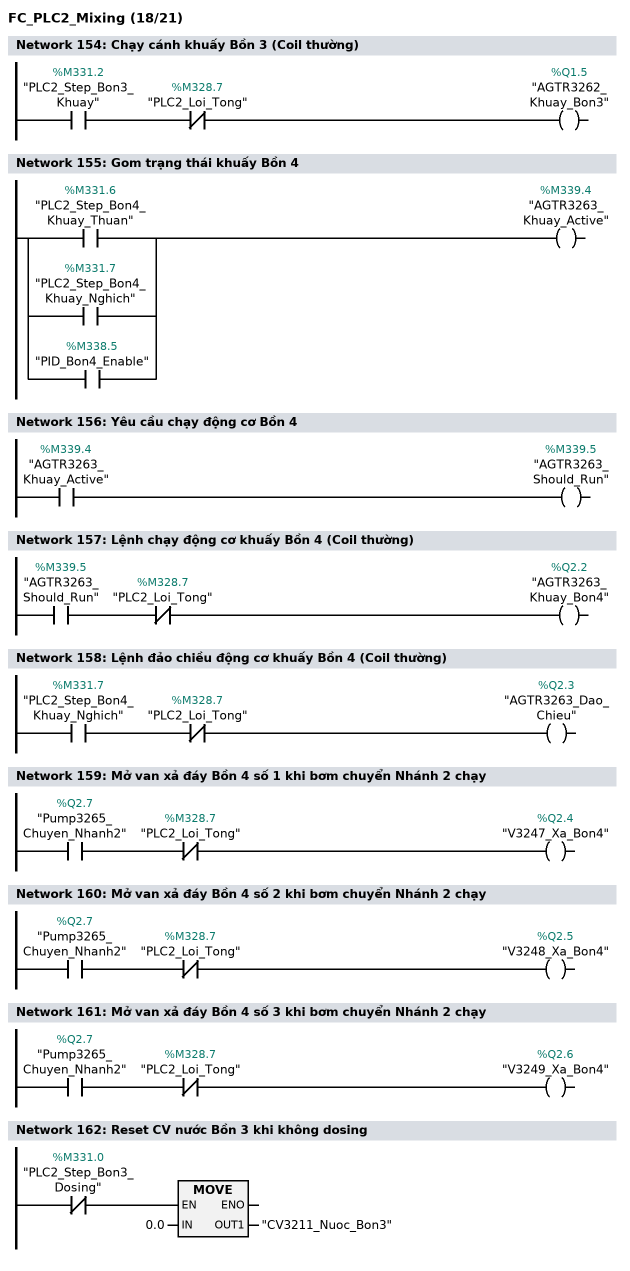
   RUNG wire#powerrail
      Contact( "PLC2_Step_Bon3_Khuay" )
      I_Contact( "PLC2_Loi_Tong" )
      Coil( "AGTR3262_Khuay_Bon3" )
   END_RUNG
   // the same network as SCL:
   "AGTR3262_Khuay_Bon3" := "PLC2_Step_Bon3_Khuay" AND NOT "PLC2_Loi_Tong";
END_REGION

REGION Network 155: Gom trạng thái khuấy Bồn 4
   RUNG wire#powerrail
      Contact( "PLC2_Step_Bon4_Khuay_Thuan" )
      wire#w1
      Coil( "AGTR3263_Khuay_Active" )
   END_RUNG
   RUNG wire#powerrail
      Contact( "PLC2_Step_Bon4_Khuay_Nghich" )
   END_RUNG wire#w1
   RUNG wire#powerrail
      Contact( "PID_Bon4_Enable" )
   END_RUNG wire#w1
   // the same network as SCL:
   "AGTR3263_Khuay_Active" := "PLC2_Step_Bon4_Khuay_Thuan" OR "PLC2_Step_Bon4_Khuay_Nghich" OR "PID_Bon4_Enable";
END_REGION

REGION Network 156: Yêu cầu chạy động cơ Bồn 4
   RUNG wire#powerrail
      Contact( "AGTR3263_Khuay_Active" )
      Coil( "AGTR3263_Should_Run" )
   END_RUNG
   // the same network as SCL:
   "AGTR3263_Should_Run" := "AGTR3263_Khuay_Active";
END_REGION

REGION Network 157: Lệnh chạy động cơ khuấy Bồn 4 (Coil thường)
   RUNG wire#powerrail
      Contact( "AGTR3263_Should_Run" )
      I_Contact( "PLC2_Loi_Tong" )
      Coil( "AGTR3263_Khuay_Bon4" )
   END_RUNG
   // the same network as SCL:
   "AGTR3263_Khuay_Bon4" := "AGTR3263_Should_Run" AND NOT "PLC2_Loi_Tong";
END_REGION

REGION Network 158: Lệnh đảo chiều động cơ khuấy Bồn 4 (Coil thường)
   RUNG wire#powerrail
      Contact( "PLC2_Step_Bon4_Khuay_Nghich" )
      I_Contact( "PLC2_Loi_Tong" )
      Coil( "AGTR3263_Dao_Chieu" )
   END_RUNG
   // the same network as SCL:
   "AGTR3263_Dao_Chieu" := "PLC2_Step_Bon4_Khuay_Nghich" AND NOT "PLC2_Loi_Tong";
END_REGION

REGION Network 159: Mở van xả đáy Bồn 4 số 1 khi bơm chuyển Nhánh 2 chạy
   RUNG wire#powerrail
      Contact( "Pump3265_Chuyen_Nhanh2" )
      I_Contact( "PLC2_Loi_Tong" )
      Coil( "V3247_Xa_Bon4" )
   END_RUNG
   // the same network as SCL:
   "V3247_Xa_Bon4" := "Pump3265_Chuyen_Nhanh2" AND NOT "PLC2_Loi_Tong";
END_REGION

REGION Network 160: Mở van xả đáy Bồn 4 số 2 khi bơm chuyển Nhánh 2 chạy
   RUNG wire#powerrail
      Contact( "Pump3265_Chuyen_Nhanh2" )
      I_Contact( "PLC2_Loi_Tong" )
      Coil( "V3248_Xa_Bon4" )
   END_RUNG
   // the same network as SCL:
   "V3248_Xa_Bon4" := "Pump3265_Chuyen_Nhanh2" AND NOT "PLC2_Loi_Tong";
END_REGION

REGION Network 161: Mở van xả đáy Bồn 4 số 3 khi bơm chuyển Nhánh 2 chạy
   RUNG wire#powerrail
      Contact( "Pump3265_Chuyen_Nhanh2" )
      I_Contact( "PLC2_Loi_Tong" )
      Coil( "V3249_Xa_Bon4" )
   END_RUNG
   // the same network as SCL:
   "V3249_Xa_Bon4" := "Pump3265_Chuyen_Nhanh2" AND NOT "PLC2_Loi_Tong";
END_REGION

